REGION Network 4: Znacznik błedu komunikacji modbus
   RUNG wire#powerrail
      { S7_Templates := "SrcType := USInt" } EQ_Contact(in1 := "dbTags_master_Fal_1"."step", in2 := 1)
      wire#w1
      "MB_MASTER_DB".MB_MASTER(REQ := "dbTags_master_Fal_1".modbusMaster.req, MB_ADDR := "dbTags_master_Fal_1".modbusMaster.mbAddr, MODE := "dbTags_master_Fal_1".modbusMaster.mode, DATA_ADDR := "dbTags_master_Fal_1".modbusMaster.dataAddr, DATA_LEN := "dbTags_master_Fal_1".modbusMaster.dataLen, DATA_PTR := "dbMasterData".ID26_Inver_Control_word_416000_Fal, DONE => "dbTags_master_Fal_1".modbusMaster.done, BUSY => "dbTags_master_Fal_1".modbusMaster.busy, ERROR => "dbTags_master_Fal_1".modbusMaster.error, STATUS => "dbTags_master_Fal_1".modbusMaster.status)
   END_RUNG
   RUNG wire#powerrail
      { S7_Templates := "SrcType := USInt" } EQ_Contact(in1 := "dbTags_master_Fal_1"."step", in2 := 2)
   END_RUNG wire#w1
   RUNG wire#powerrail
      Contact( "dbTags_master_Fal_1".modbusMaster.error )
      wire#w2
      { S7_GenerateENO := "TRUE" } Move(in := "dbTags_master_Fal_1".modbusMaster.status, out1 => "dbTags_master_Fal_1".modbusMaster.errorStatus)
   END_RUNG
   RUNG wire#w2
      { S7_GenerateENO := "TRUE" } Move(in := 0, out1 => "dbModbusRTU_Reg".receivede26_Inver_Control_word_416000.typeDataInverter_int[0])
   END_RUNG
   // the same network as SCL:
   IF ("dbTags_master_Fal_1"."step" = 1) OR ("dbTags_master_Fal_1"."step" = 2) THEN
       "MB_MASTER_DB"(REQ := "dbTags_master_Fal_1".modbusMaster.req,   // MB_MASTER
                      MB_ADDR := "dbTags_master_Fal_1".modbusMaster.mbAddr,
                      MODE := "dbTags_master_Fal_1".modbusMaster.mode,
                      DATA_ADDR := "dbTags_master_Fal_1".modbusMaster.dataAddr,
                      DATA_LEN := "dbTags_master_Fal_1".modbusMaster.dataLen,
                      DATA_PTR := "dbMasterData".ID26_Inver_Control_word_416000_Fal,
                      DONE => "dbTags_master_Fal_1".modbusMaster.done,
                      BUSY => "dbTags_master_Fal_1".modbusMaster.busy,
                      ERROR => "dbTags_master_Fal_1".modbusMaster.error,
                      STATUS => "dbTags_master_Fal_1".modbusMaster.status);
   END_IF;
   IF "dbTags_master_Fal_1".modbusMaster.error THEN
       "dbTags_master_Fal_1".modbusMaster.errorStatus := "dbTags_master_Fal_1".modbusMaster.status;
       "dbModbusRTU_Reg".receivede26_Inver_Control_word_416000.typeDataInverter_int[0] := 0;
   END_IF;
END_REGION

REGION Network 5: step1: save received data 416000
   RUNG wire#powerrail
      { S7_Templates := "SrcType := USInt" } EQ_Contact(in1 := "dbTags_master_Fal_1"."step", in2 := 2)
      Contact( "dbTags_master_Fal_1".modbusMaster.done )
      wire#w1
      { S7_GenerateENO := "TRUE" } Move(in := "dbMasterData".ID26_Inver_Control_word_416000_Fal.typeDataInverter_int[0], out1 => "dbModbusRTU_Reg".receivede26_Inver_Control_word_416000.typeDataInverter_int[0])
      R_Coil( "dbTags_master_Fal_1".modbusMaster.req )
   END_RUNG
   RUNG wire#w1
      { S7_GenerateENO := "TRUE" } Move(in := 3, out1 => "dbTags_master_Fal_1"."step")
   END_RUNG
   // the same network as SCL:
   // ENO of a box is taken as its EN; it also drops when the box reports an error
   IF ("dbTags_master_Fal_1"."step" = 2) AND "dbTags_master_Fal_1".modbusMaster.done THEN
       "dbModbusRTU_Reg".receivede26_Inver_Control_word_416000.typeDataInverter_int[0] := "dbMasterData".ID26_Inver_Control_word_416000_Fal.typeDataInverter_int[0];
       "dbTags_master_Fal_1".modbusMaster.req := FALSE;
       "dbTags_master_Fal_1"."step" := 3;
   END_IF;
END_REGION

REGION Network 6: MODBUS RTU adress 26*****step 2: read from slave Inverter setpoint
   // Pobieranie wartości zadanej Hz
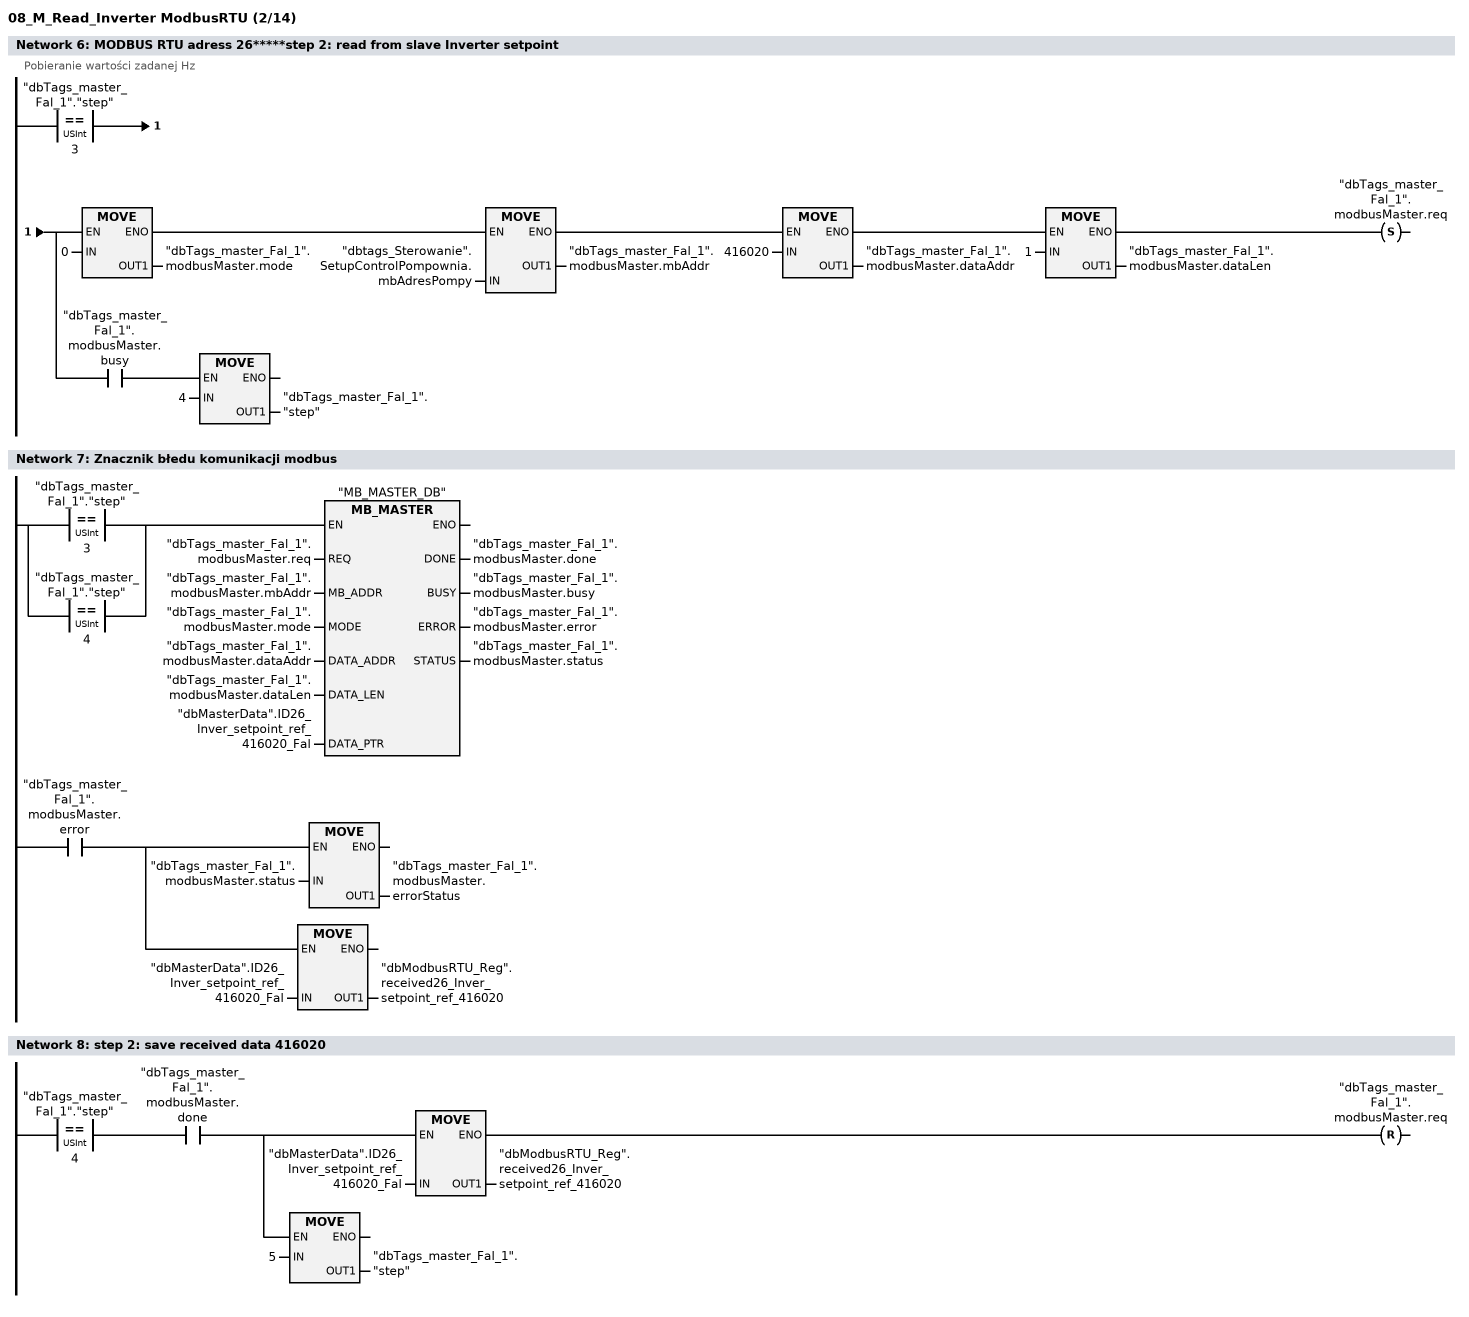
   RUNG wire#powerrail
      { S7_Templates := "SrcType := USInt" } EQ_Contact(in1 := "dbTags_master_Fal_1"."step", in2 := 3)
      wire#w1
      { S7_GenerateENO := "TRUE" } Move(in := 0, out1 => "dbTags_master_Fal_1".modbusMaster.mode)
      Move(in := "dbtags_Sterowanie".SetupControlPompownia.mbAdresPompy, out1 => "dbTags_master_Fal_1".modbusMaster.mbAddr)
      { S7_GenerateENO := "TRUE" } Move(in := 416020, out1 => "dbTags_master_Fal_1".modbusMaster.dataAddr)
      Move(in := 1, out1 => "dbTags_master_Fal_1".modbusMaster.dataLen)
      S_Coil( "dbTags_master_Fal_1".modbusMaster.req )
   END_RUNG
   RUNG wire#w1
      Contact( "dbTags_master_Fal_1".modbusMaster.busy )
      { S7_GenerateENO := "TRUE" } Move(in := 4, out1 => "dbTags_master_Fal_1"."step")
   END_RUNG
   // the same network as SCL:
   // ENO of a box is taken as its EN; it also drops when the box reports an error
   #_w1 := "dbTags_master_Fal_1"."step" = 3;
   IF #_w1 THEN
       "dbTags_master_Fal_1".modbusMaster.mode := 0;
       "dbTags_master_Fal_1".modbusMaster.mbAddr := "dbtags_Sterowanie".SetupControlPompownia.mbAdresPompy;
       "dbTags_master_Fal_1".modbusMaster.dataAddr := 416020;
       "dbTags_master_Fal_1".modbusMaster.dataLen := 1;
       "dbTags_master_Fal_1".modbusMaster.req := TRUE;
   END_IF;
   IF #_w1 AND "dbTags_master_Fal_1".modbusMaster.busy THEN "dbTags_master_Fal_1"."step" := 4; END_IF;
END_REGION

REGION Network 7: Znacznik błedu komunikacji modbus
   RUNG wire#powerrail
      { S7_Templates := "SrcType := USInt" } EQ_Contact(in1 := "dbTags_master_Fal_1"."step", in2 := 3)
      wire#w1
      "MB_MASTER_DB".MB_MASTER(REQ := "dbTags_master_Fal_1".modbusMaster.req, MB_ADDR := "dbTags_master_Fal_1".modbusMaster.mbAddr, MODE := "dbTags_master_Fal_1".modbusMaster.mode, DATA_ADDR := "dbTags_master_Fal_1".modbusMaster.dataAddr, DATA_LEN := "dbTags_master_Fal_1".modbusMaster.dataLen, DATA_PTR := "dbMasterData".ID26_Inver_setpoint_ref_416020_Fal, DONE => "dbTags_master_Fal_1".modbusMaster.done, BUSY => "dbTags_master_Fal_1".modbusMaster.busy, ERROR => "dbTags_master_Fal_1".modbusMaster.error, STATUS => "dbTags_master_Fal_1".modbusMaster.status)
   END_RUNG
   RUNG wire#powerrail
      { S7_Templates := "SrcType := USInt" } EQ_Contact(in1 := "dbTags_master_Fal_1"."step", in2 := 4)
   END_RUNG wire#w1
   RUNG wire#powerrail
      Contact( "dbTags_master_Fal_1".modbusMaster.error )
      wire#w2
      { S7_GenerateENO := "TRUE" } Move(in := "dbTags_master_Fal_1".modbusMaster.status, out1 => "dbTags_master_Fal_1".modbusMaster.errorStatus)
   END_RUNG
   RUNG wire#w2
      { S7_GenerateENO := "TRUE" } Move(in := "dbMasterData".ID26_Inver_setpoint_ref_416020_Fal, out1 => "dbModbusRTU_Reg".received26_Inver_setpoint_ref_416020)
   END_RUNG
   // the same network as SCL:
   IF ("dbTags_master_Fal_1"."step" = 3) OR ("dbTags_master_Fal_1"."step" = 4) THEN
       "MB_MASTER_DB"(REQ := "dbTags_master_Fal_1".modbusMaster.req,   // MB_MASTER
                      MB_ADDR := "dbTags_master_Fal_1".modbusMaster.mbAddr,
                      MODE := "dbTags_master_Fal_1".modbusMaster.mode,
                      DATA_ADDR := "dbTags_master_Fal_1".modbusMaster.dataAddr,
                      DATA_LEN := "dbTags_master_Fal_1".modbusMaster.dataLen,
                      DATA_PTR := "dbMasterData".ID26_Inver_setpoint_ref_416020_Fal,
                      DONE => "dbTags_master_Fal_1".modbusMaster.done,
                      BUSY => "dbTags_master_Fal_1".modbusMaster.busy,
                      ERROR => "dbTags_master_Fal_1".modbusMaster.error,
                      STATUS => "dbTags_master_Fal_1".modbusMaster.status);
   END_IF;
   IF "dbTags_master_Fal_1".modbusMaster.error THEN
       "dbTags_master_Fal_1".modbusMaster.errorStatus := "dbTags_master_Fal_1".modbusMaster.status;
       "dbModbusRTU_Reg".received26_Inver_setpoint_ref_416020 := "dbMasterData".ID26_Inver_setpoint_ref_416020_Fal;
   END_IF;
END_REGION

REGION Network 8: step 2: save received data 416020
   RUNG wire#powerrail
      { S7_Templates := "SrcType := USInt" } EQ_Contact(in1 := "dbTags_master_Fal_1"."step", in2 := 4)
      Contact( "dbTags_master_Fal_1".modbusMaster.done )
      wire#w1
      { S7_GenerateENO := "TRUE" } Move(in := "dbMasterData".ID26_Inver_setpoint_ref_416020_Fal, out1 => "dbModbusRTU_Reg".received26_Inver_setpoint_ref_416020)
      R_Coil( "dbTags_master_Fal_1".modbusMaster.req )
   END_RUNG
   RUNG wire#w1
      { S7_GenerateENO := "TRUE" } Move(in := 5, out1 => "dbTags_master_Fal_1"."step")
   END_RUNG
   // the same network as SCL:
   // ENO of a box is taken as its EN; it also drops when the box reports an error
   IF ("dbTags_master_Fal_1"."step" = 4) AND "dbTags_master_Fal_1".modbusMaster.done THEN
       "dbModbusRTU_Reg".received26_Inver_setpoint_ref_416020 := "dbMasterData".ID26_Inver_setpoint_ref_416020_Fal;
       "dbTags_master_Fal_1".modbusMaster.req := FALSE;
       "dbTags_master_Fal_1"."step" := 5;
   END_IF;
END_REGION

REGION Network 9: MODBUS RTU adress 26*****step 3: read from slave Inverter status word
   // Pobieramy status falownika
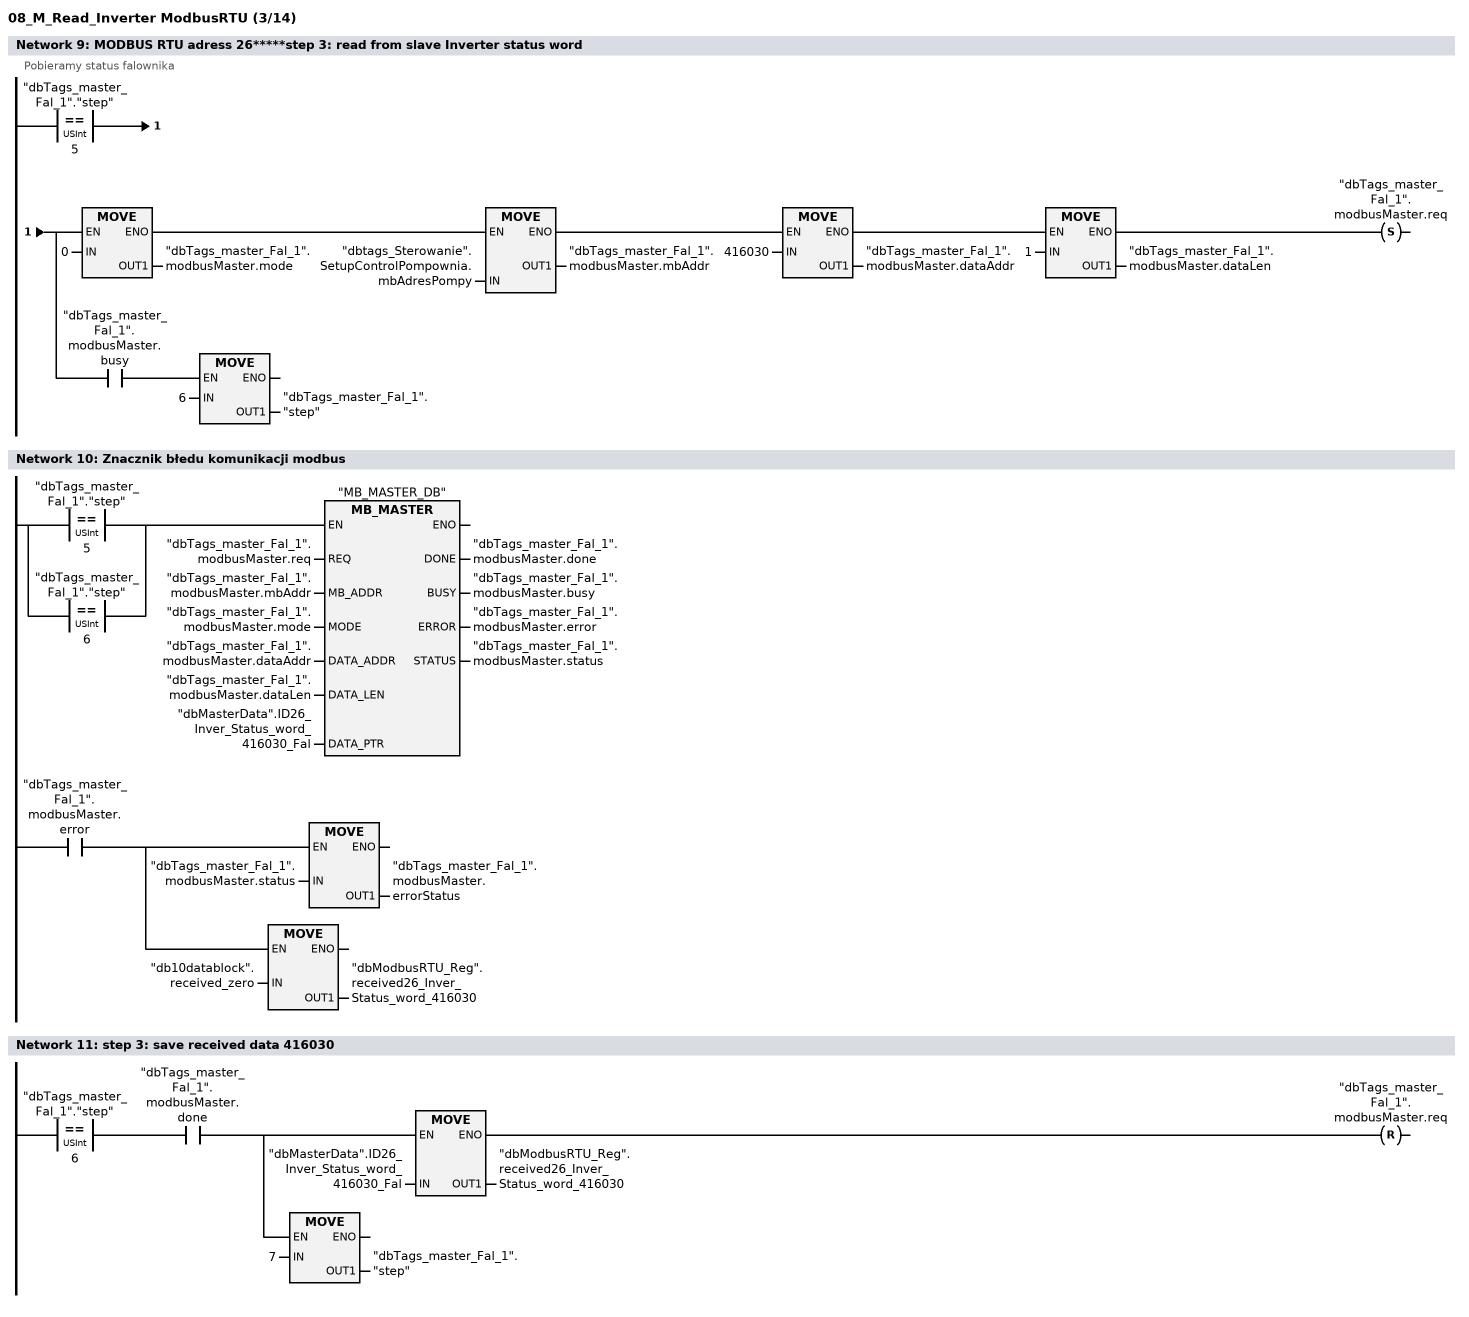
   RUNG wire#powerrail
      { S7_Templates := "SrcType := USInt" } EQ_Contact(in1 := "dbTags_master_Fal_1"."step", in2 := 5)
      wire#w1
      { S7_GenerateENO := "TRUE" } Move(in := 0, out1 => "dbTags_master_Fal_1".modbusMaster.mode)
      Move(in := "dbtags_Sterowanie".SetupControlPompownia.mbAdresPompy, out1 => "dbTags_master_Fal_1".modbusMaster.mbAddr)
      { S7_GenerateENO := "TRUE" } Move(in := 416030, out1 => "dbTags_master_Fal_1".modbusMaster.dataAddr)
      Move(in := 1, out1 => "dbTags_master_Fal_1".modbusMaster.dataLen)
      S_Coil( "dbTags_master_Fal_1".modbusMaster.req )
   END_RUNG
   RUNG wire#w1
      Contact( "dbTags_master_Fal_1".modbusMaster.busy )
      { S7_GenerateENO := "TRUE" } Move(in := 6, out1 => "dbTags_master_Fal_1"."step")
   END_RUNG
   // the same network as SCL:
   // ENO of a box is taken as its EN; it also drops when the box reports an error
   #_w1 := "dbTags_master_Fal_1"."step" = 5;
   IF #_w1 THEN
       "dbTags_master_Fal_1".modbusMaster.mode := 0;
       "dbTags_master_Fal_1".modbusMaster.mbAddr := "dbtags_Sterowanie".SetupControlPompownia.mbAdresPompy;
       "dbTags_master_Fal_1".modbusMaster.dataAddr := 416030;
       "dbTags_master_Fal_1".modbusMaster.dataLen := 1;
       "dbTags_master_Fal_1".modbusMaster.req := TRUE;
   END_IF;
   IF #_w1 AND "dbTags_master_Fal_1".modbusMaster.busy THEN "dbTags_master_Fal_1"."step" := 6; END_IF;
END_REGION

REGION Network 10: Znacznik błedu komunikacji modbus
   RUNG wire#powerrail
      { S7_Templates := "SrcType := USInt" } EQ_Contact(in1 := "dbTags_master_Fal_1"."step", in2 := 5)
      wire#w1
      "MB_MASTER_DB".MB_MASTER(REQ := "dbTags_master_Fal_1".modbusMaster.req, MB_ADDR := "dbTags_master_Fal_1".modbusMaster.mbAddr, MODE := "dbTags_master_Fal_1".modbusMaster.mode, DATA_ADDR := "dbTags_master_Fal_1".modbusMaster.dataAddr, DATA_LEN := "dbTags_master_Fal_1".modbusMaster.dataLen, DATA_PTR := "dbMasterData".ID26_Inver_Status_word_416030_Fal, DONE => "dbTags_master_Fal_1".modbusMaster.done, BUSY => "dbTags_master_Fal_1".modbusMaster.busy, ERROR => "dbTags_master_Fal_1".modbusMaster.error, STATUS => "dbTags_master_Fal_1".modbusMaster.status)
   END_RUNG
   RUNG wire#powerrail
      { S7_Templates := "SrcType := USInt" } EQ_Contact(in1 := "dbTags_master_Fal_1"."step", in2 := 6)
   END_RUNG wire#w1
   RUNG wire#powerrail
      Contact( "dbTags_master_Fal_1".modbusMaster.error )
      wire#w2
      { S7_GenerateENO := "TRUE" } Move(in := "dbTags_master_Fal_1".modbusMaster.status, out1 => "dbTags_master_Fal_1".modbusMaster.errorStatus)
   END_RUNG
   RUNG wire#w2
      { S7_GenerateENO := "TRUE" } Move(in := "db10datablock".received_zero, out1 => "dbModbusRTU_Reg".received26_Inver_Status_word_416030)
   END_RUNG
   // the same network as SCL:
   IF ("dbTags_master_Fal_1"."step" = 5) OR ("dbTags_master_Fal_1"."step" = 6) THEN
       "MB_MASTER_DB"(REQ := "dbTags_master_Fal_1".modbusMaster.req,   // MB_MASTER
                      MB_ADDR := "dbTags_master_Fal_1".modbusMaster.mbAddr,
                      MODE := "dbTags_master_Fal_1".modbusMaster.mode,
                      DATA_ADDR := "dbTags_master_Fal_1".modbusMaster.dataAddr,
                      DATA_LEN := "dbTags_master_Fal_1".modbusMaster.dataLen,
                      DATA_PTR := "dbMasterData".ID26_Inver_Status_word_416030_Fal,
                      DONE => "dbTags_master_Fal_1".modbusMaster.done,
                      BUSY => "dbTags_master_Fal_1".modbusMaster.busy,
                      ERROR => "dbTags_master_Fal_1".modbusMaster.error,
                      STATUS => "dbTags_master_Fal_1".modbusMaster.status);
   END_IF;
   IF "dbTags_master_Fal_1".modbusMaster.error THEN
       "dbTags_master_Fal_1".modbusMaster.errorStatus := "dbTags_master_Fal_1".modbusMaster.status;
       "dbModbusRTU_Reg".received26_Inver_Status_word_416030 := "db10datablock".received_zero;
   END_IF;
END_REGION

REGION Network 11: step 3: save received data 416030
   RUNG wire#powerrail
      { S7_Templates := "SrcType := USInt" } EQ_Contact(in1 := "dbTags_master_Fal_1"."step", in2 := 6)
      Contact( "dbTags_master_Fal_1".modbusMaster.done )
      wire#w1
      { S7_GenerateENO := "TRUE" } Move(in := "dbMasterData".ID26_Inver_Status_word_416030_Fal, out1 => "dbModbusRTU_Reg".received26_Inver_Status_word_416030)
      R_Coil( "dbTags_master_Fal_1".modbusMaster.req )
   END_RUNG
   RUNG wire#w1
      { S7_GenerateENO := "TRUE" } Move(in := 7, out1 => "dbTags_master_Fal_1"."step")
   END_RUNG
   // the same network as SCL:
   // ENO of a box is taken as its EN; it also drops when the box reports an error
   IF ("dbTags_master_Fal_1"."step" = 6) AND "dbTags_master_Fal_1".modbusMaster.done THEN
       "dbModbusRTU_Reg".received26_Inver_Status_word_416030 := "dbMasterData".ID26_Inver_Status_word_416030_Fal;
       "dbTags_master_Fal_1".modbusMaster.req := FALSE;
       "dbTags_master_Fal_1"."step" := 7;
   END_IF;
END_REGION

REGION Network 13: MODBUS RTU adress 26*****step 4: read from slave Inverter frequency
   // Pobieramy częstotliwość na silniku
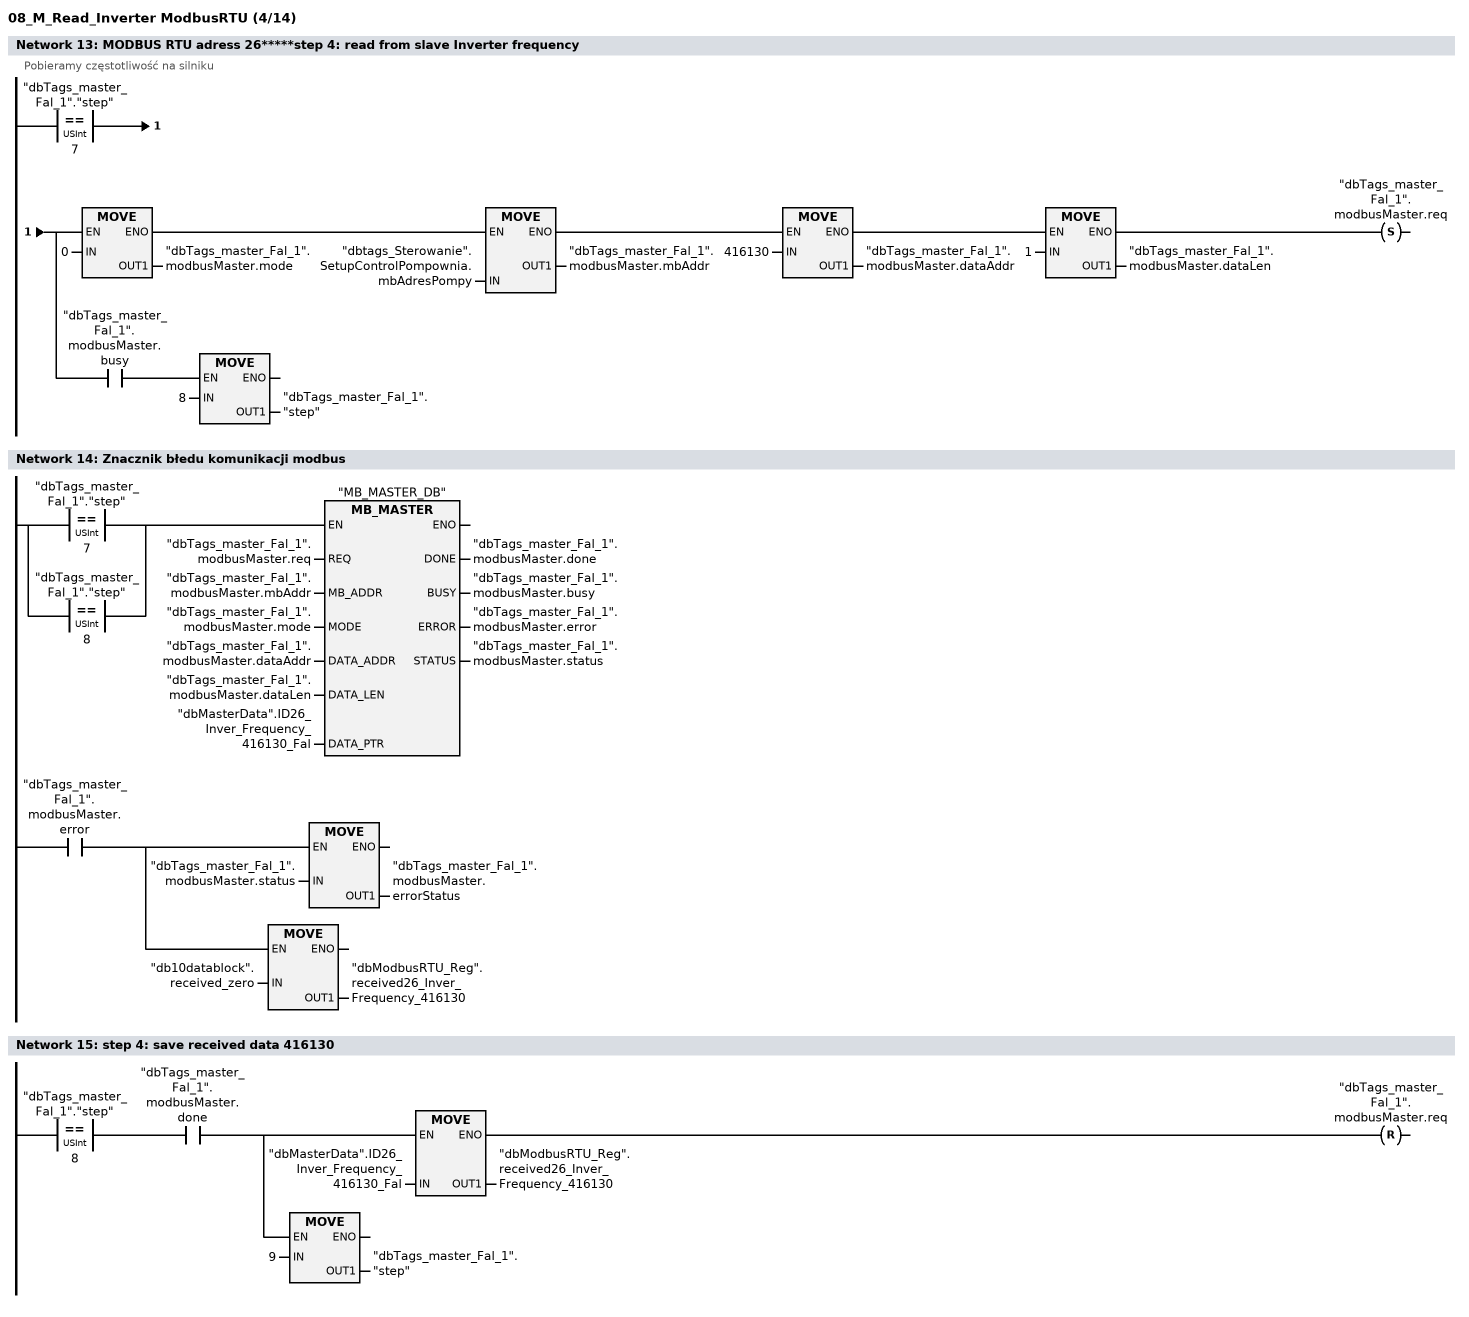
   RUNG wire#powerrail
      { S7_Templates := "SrcType := USInt" } EQ_Contact(in1 := "dbTags_master_Fal_1"."step", in2 := 7)
      wire#w1
      { S7_GenerateENO := "TRUE" } Move(in := 0, out1 => "dbTags_master_Fal_1".modbusMaster.mode)
      Move(in := "dbtags_Sterowanie".SetupControlPompownia.mbAdresPompy, out1 => "dbTags_master_Fal_1".modbusMaster.mbAddr)
      { S7_GenerateENO := "TRUE" } Move(in := 416130, out1 => "dbTags_master_Fal_1".modbusMaster.dataAddr)
      Move(in := 1, out1 => "dbTags_master_Fal_1".modbusMaster.dataLen)
      S_Coil( "dbTags_master_Fal_1".modbusMaster.req )
   END_RUNG
   RUNG wire#w1
      Contact( "dbTags_master_Fal_1".modbusMaster.busy )
      { S7_GenerateENO := "TRUE" } Move(in := 8, out1 => "dbTags_master_Fal_1"."step")
   END_RUNG
   // the same network as SCL:
   // ENO of a box is taken as its EN; it also drops when the box reports an error
   #_w1 := "dbTags_master_Fal_1"."step" = 7;
   IF #_w1 THEN
       "dbTags_master_Fal_1".modbusMaster.mode := 0;
       "dbTags_master_Fal_1".modbusMaster.mbAddr := "dbtags_Sterowanie".SetupControlPompownia.mbAdresPompy;
       "dbTags_master_Fal_1".modbusMaster.dataAddr := 416130;
       "dbTags_master_Fal_1".modbusMaster.dataLen := 1;
       "dbTags_master_Fal_1".modbusMaster.req := TRUE;
   END_IF;
   IF #_w1 AND "dbTags_master_Fal_1".modbusMaster.busy THEN "dbTags_master_Fal_1"."step" := 8; END_IF;
END_REGION

REGION Network 14: Znacznik błedu komunikacji modbus
   RUNG wire#powerrail
      { S7_Templates := "SrcType := USInt" } EQ_Contact(in1 := "dbTags_master_Fal_1"."step", in2 := 7)
      wire#w1
      "MB_MASTER_DB".MB_MASTER(REQ := "dbTags_master_Fal_1".modbusMaster.req, MB_ADDR := "dbTags_master_Fal_1".modbusMaster.mbAddr, MODE := "dbTags_master_Fal_1".modbusMaster.mode, DATA_ADDR := "dbTags_master_Fal_1".modbusMaster.dataAddr, DATA_LEN := "dbTags_master_Fal_1".modbusMaster.dataLen, DATA_PTR := "dbMasterData".ID26_Inver_Frequency_416130_Fal, DONE => "dbTags_master_Fal_1".modbusMaster.done, BUSY => "dbTags_master_Fal_1".modbusMaster.busy, ERROR => "dbTags_master_Fal_1".modbusMaster.error, STATUS => "dbTags_master_Fal_1".modbusMaster.status)
   END_RUNG
   RUNG wire#powerrail
      { S7_Templates := "SrcType := USInt" } EQ_Contact(in1 := "dbTags_master_Fal_1"."step", in2 := 8)
   END_RUNG wire#w1
   RUNG wire#powerrail
      Contact( "dbTags_master_Fal_1".modbusMaster.error )
      wire#w2
      { S7_GenerateENO := "TRUE" } Move(in := "dbTags_master_Fal_1".modbusMaster.status, out1 => "dbTags_master_Fal_1".modbusMaster.errorStatus)
   END_RUNG
   RUNG wire#w2
      { S7_GenerateENO := "TRUE" } Move(in := "db10datablock".received_zero, out1 => "dbModbusRTU_Reg".received26_Inver_Frequency_416130)
   END_RUNG
   // the same network as SCL:
   IF ("dbTags_master_Fal_1"."step" = 7) OR ("dbTags_master_Fal_1"."step" = 8) THEN
       "MB_MASTER_DB"(REQ := "dbTags_master_Fal_1".modbusMaster.req,   // MB_MASTER
                      MB_ADDR := "dbTags_master_Fal_1".modbusMaster.mbAddr,
                      MODE := "dbTags_master_Fal_1".modbusMaster.mode,
                      DATA_ADDR := "dbTags_master_Fal_1".modbusMaster.dataAddr,
                      DATA_LEN := "dbTags_master_Fal_1".modbusMaster.dataLen,
                      DATA_PTR := "dbMasterData".ID26_Inver_Frequency_416130_Fal,
                      DONE => "dbTags_master_Fal_1".modbusMaster.done,
                      BUSY => "dbTags_master_Fal_1".modbusMaster.busy,
                      ERROR => "dbTags_master_Fal_1".modbusMaster.error,
                      STATUS => "dbTags_master_Fal_1".modbusMaster.status);
   END_IF;
   IF "dbTags_master_Fal_1".modbusMaster.error THEN
       "dbTags_master_Fal_1".modbusMaster.errorStatus := "dbTags_master_Fal_1".modbusMaster.status;
       "dbModbusRTU_Reg".received26_Inver_Frequency_416130 := "db10datablock".received_zero;
   END_IF;
END_REGION

REGION Network 15: step 4: save received data 416130
   RUNG wire#powerrail
      { S7_Templates := "SrcType := USInt" } EQ_Contact(in1 := "dbTags_master_Fal_1"."step", in2 := 8)
      Contact( "dbTags_master_Fal_1".modbusMaster.done )
      wire#w1
      { S7_GenerateENO := "TRUE" } Move(in := "dbMasterData".ID26_Inver_Frequency_416130_Fal, out1 => "dbModbusRTU_Reg".received26_Inver_Frequency_416130)
      R_Coil( "dbTags_master_Fal_1".modbusMaster.req )
   END_RUNG
   RUNG wire#w1
      { S7_GenerateENO := "TRUE" } Move(in := 9, out1 => "dbTags_master_Fal_1"."step")
   END_RUNG
   // the same network as SCL:
   // ENO of a box is taken as its EN; it also drops when the box reports an error
   IF ("dbTags_master_Fal_1"."step" = 8) AND "dbTags_master_Fal_1".modbusMaster.done THEN
       "dbModbusRTU_Reg".received26_Inver_Frequency_416130 := "dbMasterData".ID26_Inver_Frequency_416130_Fal;
       "dbTags_master_Fal_1".modbusMaster.req := FALSE;
       "dbTags_master_Fal_1"."step" := 9;
   END_IF;
END_REGION

REGION Network 17: MODBUS RTU adress 26*****step 5: read from slave Motor Current
   // Pobieramy prąd silnika
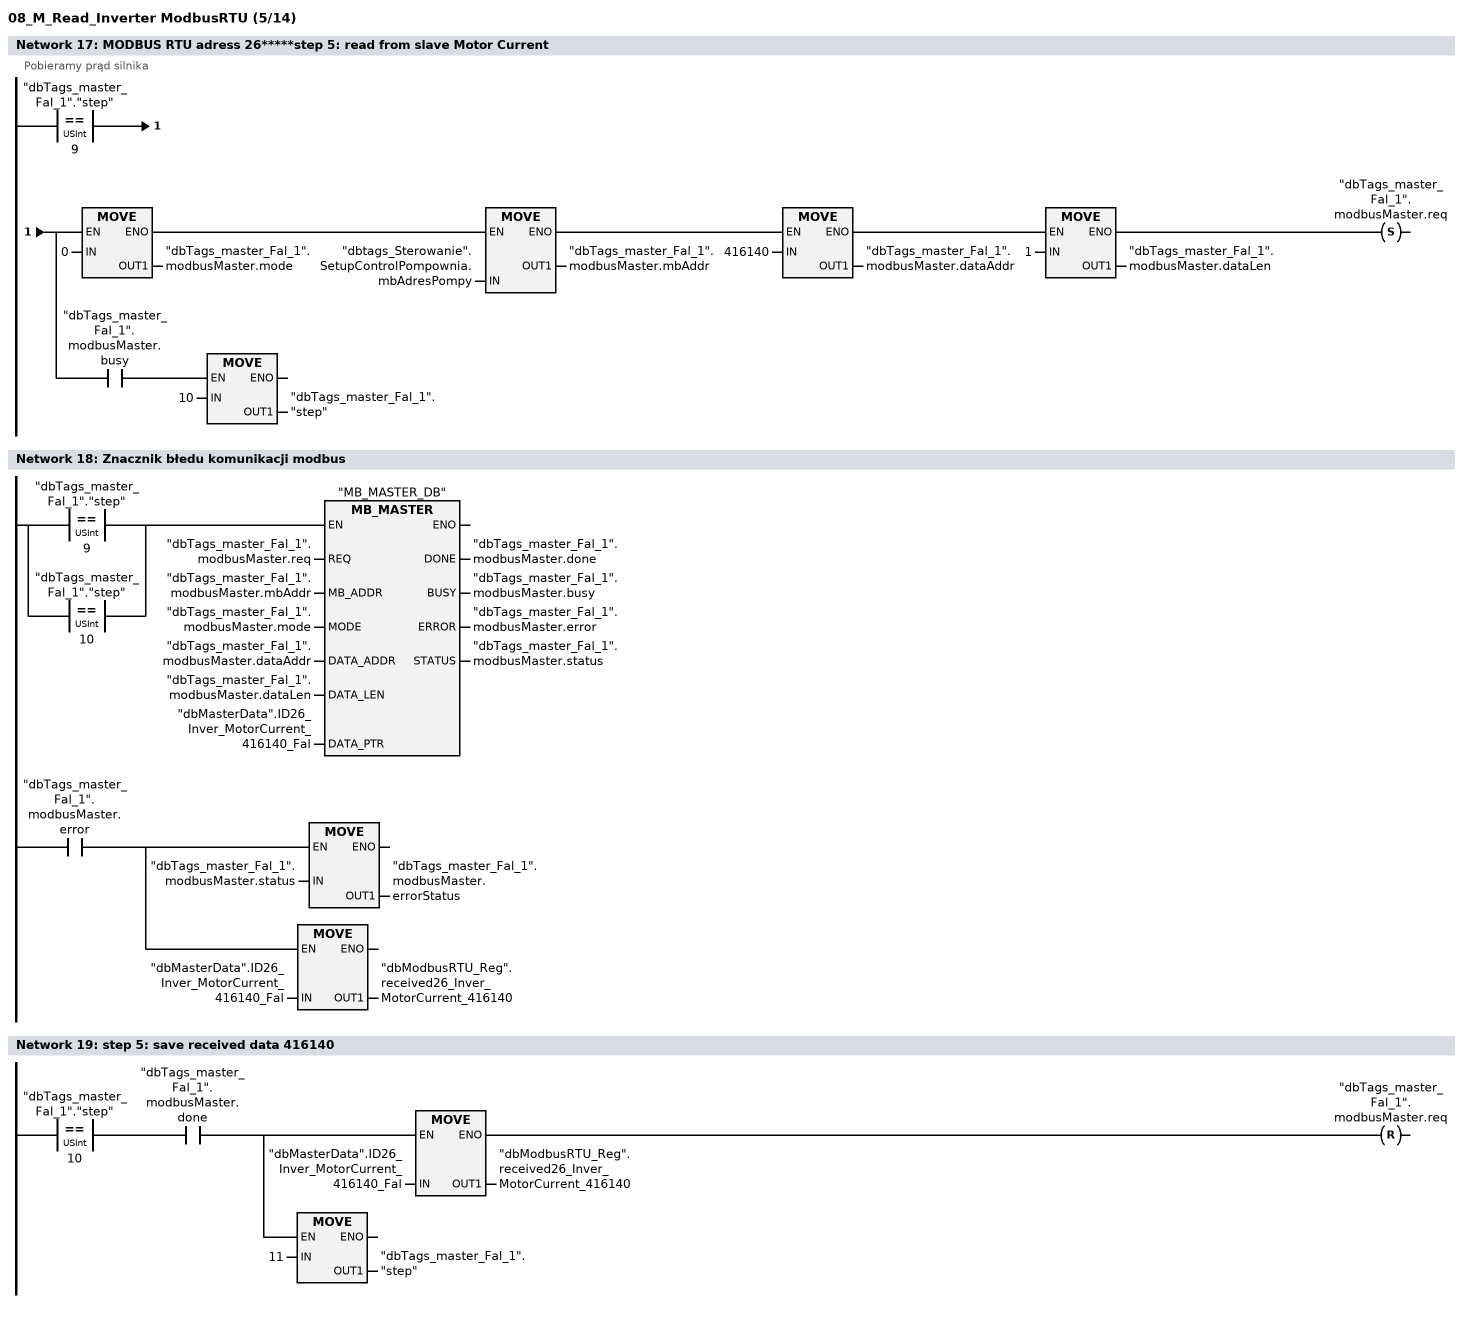
   RUNG wire#powerrail
      { S7_Templates := "SrcType := USInt" } EQ_Contact(in1 := "dbTags_master_Fal_1"."step", in2 := 9)
      wire#w1
      { S7_GenerateENO := "TRUE" } Move(in := 0, out1 => "dbTags_master_Fal_1".modbusMaster.mode)
      Move(in := "dbtags_Sterowanie".SetupControlPompownia.mbAdresPompy, out1 => "dbTags_master_Fal_1".modbusMaster.mbAddr)
      { S7_GenerateENO := "TRUE" } Move(in := 416140, out1 => "dbTags_master_Fal_1".modbusMaster.dataAddr)
      Move(in := 1, out1 => "dbTags_master_Fal_1".modbusMaster.dataLen)
      S_Coil( "dbTags_master_Fal_1".modbusMaster.req )
   END_RUNG
   RUNG wire#w1
      Contact( "dbTags_master_Fal_1".modbusMaster.busy )
      { S7_GenerateENO := "TRUE" } Move(in := 10, out1 => "dbTags_master_Fal_1"."step")
   END_RUNG
   // the same network as SCL:
   // ENO of a box is taken as its EN; it also drops when the box reports an error
   #_w1 := "dbTags_master_Fal_1"."step" = 9;
   IF #_w1 THEN
       "dbTags_master_Fal_1".modbusMaster.mode := 0;
       "dbTags_master_Fal_1".modbusMaster.mbAddr := "dbtags_Sterowanie".SetupControlPompownia.mbAdresPompy;
       "dbTags_master_Fal_1".modbusMaster.dataAddr := 416140;
       "dbTags_master_Fal_1".modbusMaster.dataLen := 1;
       "dbTags_master_Fal_1".modbusMaster.req := TRUE;
   END_IF;
   IF #_w1 AND "dbTags_master_Fal_1".modbusMaster.busy THEN "dbTags_master_Fal_1"."step" := 10; END_IF;
END_REGION

REGION Network 18: Znacznik błedu komunikacji modbus
   RUNG wire#powerrail
      { S7_Templates := "SrcType := USInt" } EQ_Contact(in1 := "dbTags_master_Fal_1"."step", in2 := 9)
      wire#w1
      "MB_MASTER_DB".MB_MASTER(REQ := "dbTags_master_Fal_1".modbusMaster.req, MB_ADDR := "dbTags_master_Fal_1".modbusMaster.mbAddr, MODE := "dbTags_master_Fal_1".modbusMaster.mode, DATA_ADDR := "dbTags_master_Fal_1".modbusMaster.dataAddr, DATA_LEN := "dbTags_master_Fal_1".modbusMaster.dataLen, DATA_PTR := "dbMasterData".ID26_Inver_MotorCurrent_416140_Fal, DONE => "dbTags_master_Fal_1".modbusMaster.done, BUSY => "dbTags_master_Fal_1".modbusMaster.busy, ERROR => "dbTags_master_Fal_1".modbusMaster.error, STATUS => "dbTags_master_Fal_1".modbusMaster.status)
   END_RUNG
   RUNG wire#powerrail
      { S7_Templates := "SrcType := USInt" } EQ_Contact(in1 := "dbTags_master_Fal_1"."step", in2 := 10)
   END_RUNG wire#w1
   RUNG wire#powerrail
      Contact( "dbTags_master_Fal_1".modbusMaster.error )
      wire#w2
      { S7_GenerateENO := "TRUE" } Move(in := "dbTags_master_Fal_1".modbusMaster.status, out1 => "dbTags_master_Fal_1".modbusMaster.errorStatus)
   END_RUNG
   RUNG wire#w2
      { S7_GenerateENO := "TRUE" } Move(in := "dbMasterData".ID26_Inver_MotorCurrent_416140_Fal, out1 => "dbModbusRTU_Reg".received26_Inver_MotorCurrent_416140)
   END_RUNG
   // the same network as SCL:
   IF ("dbTags_master_Fal_1"."step" = 9) OR ("dbTags_master_Fal_1"."step" = 10) THEN
       "MB_MASTER_DB"(REQ := "dbTags_master_Fal_1".modbusMaster.req,   // MB_MASTER
                      MB_ADDR := "dbTags_master_Fal_1".modbusMaster.mbAddr,
                      MODE := "dbTags_master_Fal_1".modbusMaster.mode,
                      DATA_ADDR := "dbTags_master_Fal_1".modbusMaster.dataAddr,
                      DATA_LEN := "dbTags_master_Fal_1".modbusMaster.dataLen,
                      DATA_PTR := "dbMasterData".ID26_Inver_MotorCurrent_416140_Fal,
                      DONE => "dbTags_master_Fal_1".modbusMaster.done,
                      BUSY => "dbTags_master_Fal_1".modbusMaster.busy,
                      ERROR => "dbTags_master_Fal_1".modbusMaster.error,
                      STATUS => "dbTags_master_Fal_1".modbusMaster.status);
   END_IF;
   IF "dbTags_master_Fal_1".modbusMaster.error THEN
       "dbTags_master_Fal_1".modbusMaster.errorStatus := "dbTags_master_Fal_1".modbusMaster.status;
       "dbModbusRTU_Reg".received26_Inver_MotorCurrent_416140 := "dbMasterData".ID26_Inver_MotorCurrent_416140_Fal;
   END_IF;
END_REGION

REGION Network 19: step 5: save received data 416140
   RUNG wire#powerrail
      { S7_Templates := "SrcType := USInt" } EQ_Contact(in1 := "dbTags_master_Fal_1"."step", in2 := 10)
      Contact( "dbTags_master_Fal_1".modbusMaster.done )
      wire#w1
      { S7_GenerateENO := "TRUE" } Move(in := "dbMasterData".ID26_Inver_MotorCurrent_416140_Fal, out1 => "dbModbusRTU_Reg".received26_Inver_MotorCurrent_416140)
      R_Coil( "dbTags_master_Fal_1".modbusMaster.req )
   END_RUNG
   RUNG wire#w1
      { S7_GenerateENO := "TRUE" } Move(in := 11, out1 => "dbTags_master_Fal_1"."step")
   END_RUNG
   // the same network as SCL:
   // ENO of a box is taken as its EN; it also drops when the box reports an error
   IF ("dbTags_master_Fal_1"."step" = 10) AND "dbTags_master_Fal_1".modbusMaster.done THEN
       "dbModbusRTU_Reg".received26_Inver_MotorCurrent_416140 := "dbMasterData".ID26_Inver_MotorCurrent_416140_Fal;
       "dbTags_master_Fal_1".modbusMaster.req := FALSE;
       "dbTags_master_Fal_1"."step" := 11;
   END_IF;
END_REGION

REGION Network 21: MODBUS RTU adress 26*****step 6: read from slave DC Voltage
   // Pobieramy napięcie na szynie DC
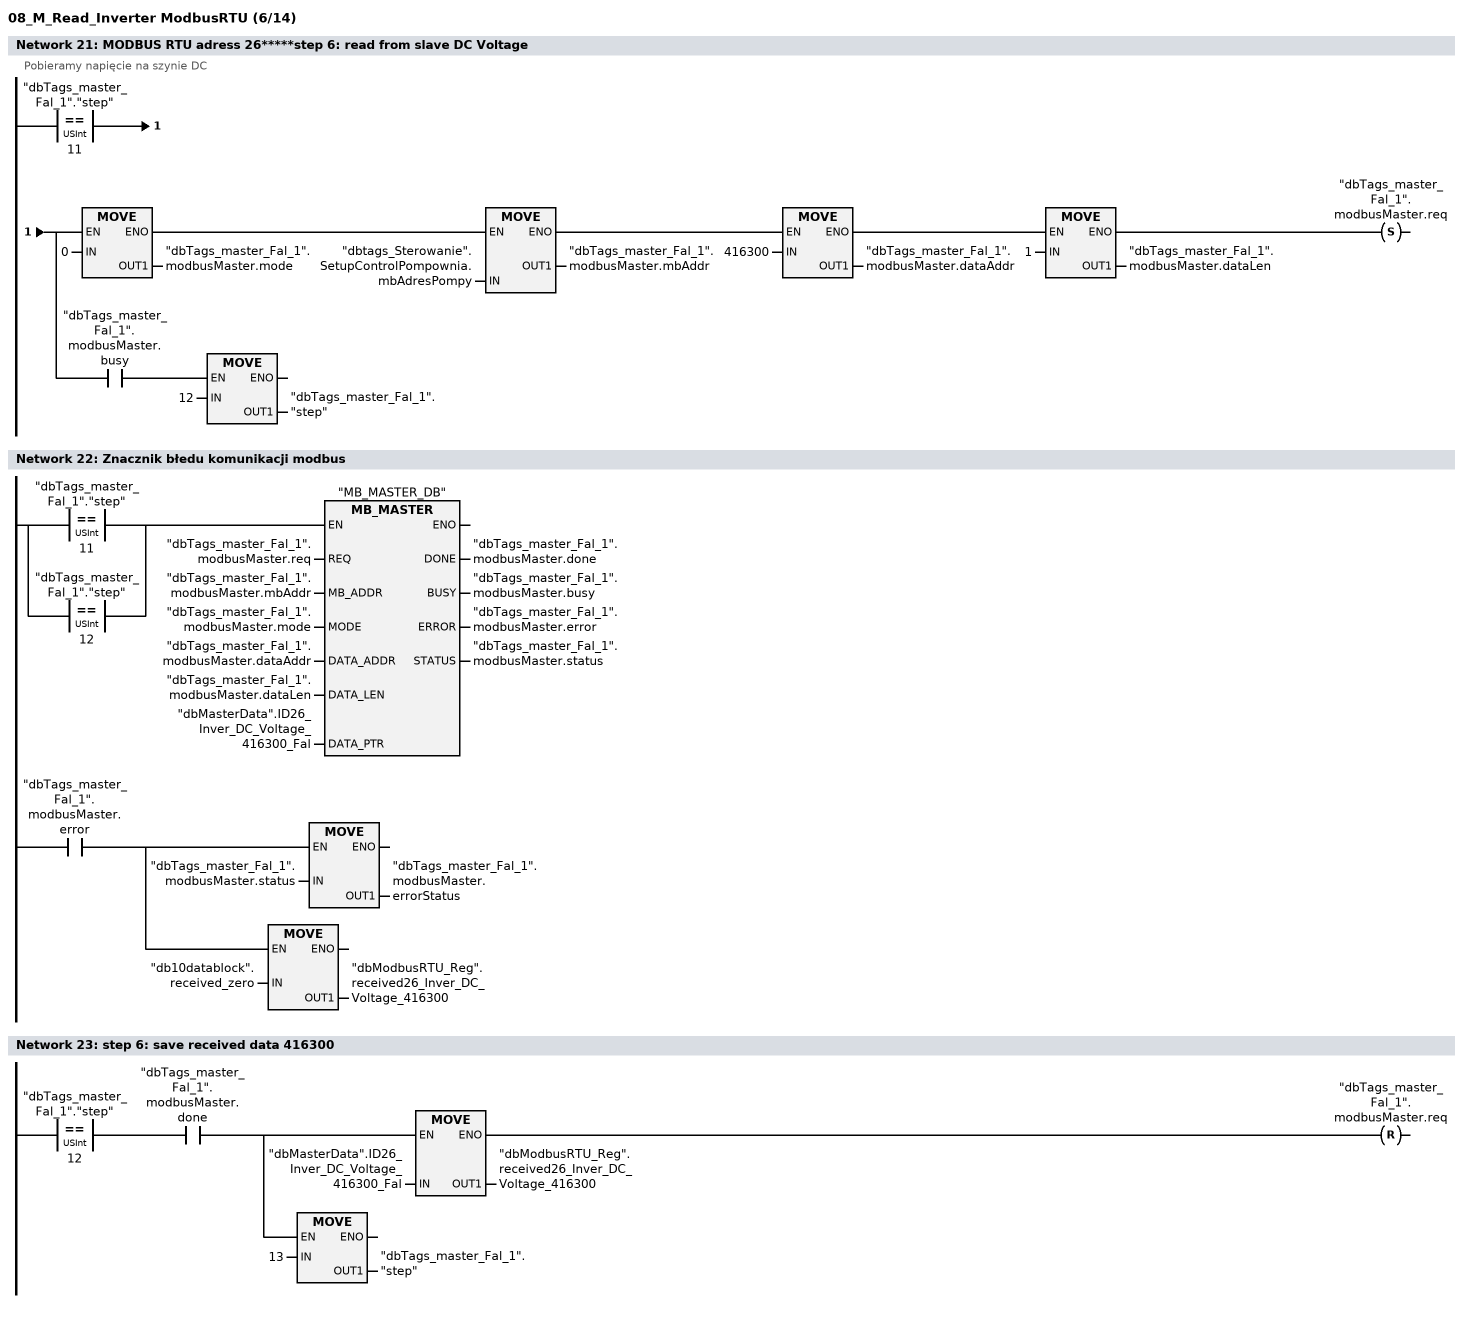
   RUNG wire#powerrail
      { S7_Templates := "SrcType := USInt" } EQ_Contact(in1 := "dbTags_master_Fal_1"."step", in2 := 11)
      wire#w1
      { S7_GenerateENO := "TRUE" } Move(in := 0, out1 => "dbTags_master_Fal_1".modbusMaster.mode)
      Move(in := "dbtags_Sterowanie".SetupControlPompownia.mbAdresPompy, out1 => "dbTags_master_Fal_1".modbusMaster.mbAddr)
      { S7_GenerateENO := "TRUE" } Move(in := 416300, out1 => "dbTags_master_Fal_1".modbusMaster.dataAddr)
      Move(in := 1, out1 => "dbTags_master_Fal_1".modbusMaster.dataLen)
      S_Coil( "dbTags_master_Fal_1".modbusMaster.req )
   END_RUNG
   RUNG wire#w1
      Contact( "dbTags_master_Fal_1".modbusMaster.busy )
      { S7_GenerateENO := "TRUE" } Move(in := 12, out1 => "dbTags_master_Fal_1"."step")
   END_RUNG
   // the same network as SCL:
   // ENO of a box is taken as its EN; it also drops when the box reports an error
   #_w1 := "dbTags_master_Fal_1"."step" = 11;
   IF #_w1 THEN
       "dbTags_master_Fal_1".modbusMaster.mode := 0;
       "dbTags_master_Fal_1".modbusMaster.mbAddr := "dbtags_Sterowanie".SetupControlPompownia.mbAdresPompy;
       "dbTags_master_Fal_1".modbusMaster.dataAddr := 416300;
       "dbTags_master_Fal_1".modbusMaster.dataLen := 1;
       "dbTags_master_Fal_1".modbusMaster.req := TRUE;
   END_IF;
   IF #_w1 AND "dbTags_master_Fal_1".modbusMaster.busy THEN "dbTags_master_Fal_1"."step" := 12; END_IF;
END_REGION

REGION Network 22: Znacznik błedu komunikacji modbus
   RUNG wire#powerrail
      { S7_Templates := "SrcType := USInt" } EQ_Contact(in1 := "dbTags_master_Fal_1"."step", in2 := 11)
      wire#w1
      "MB_MASTER_DB".MB_MASTER(REQ := "dbTags_master_Fal_1".modbusMaster.req, MB_ADDR := "dbTags_master_Fal_1".modbusMaster.mbAddr, MODE := "dbTags_master_Fal_1".modbusMaster.mode, DATA_ADDR := "dbTags_master_Fal_1".modbusMaster.dataAddr, DATA_LEN := "dbTags_master_Fal_1".modbusMaster.dataLen, DATA_PTR := "dbMasterData".ID26_Inver_DC_Voltage_416300_Fal, DONE => "dbTags_master_Fal_1".modbusMaster.done, BUSY => "dbTags_master_Fal_1".modbusMaster.busy, ERROR => "dbTags_master_Fal_1".modbusMaster.error, STATUS => "dbTags_master_Fal_1".modbusMaster.status)
   END_RUNG
   RUNG wire#powerrail
      { S7_Templates := "SrcType := USInt" } EQ_Contact(in1 := "dbTags_master_Fal_1"."step", in2 := 12)
   END_RUNG wire#w1
   RUNG wire#powerrail
      Contact( "dbTags_master_Fal_1".modbusMaster.error )
      wire#w2
      { S7_GenerateENO := "TRUE" } Move(in := "dbTags_master_Fal_1".modbusMaster.status, out1 => "dbTags_master_Fal_1".modbusMaster.errorStatus)
   END_RUNG
   RUNG wire#w2
      { S7_GenerateENO := "TRUE" } Move(in := "db10datablock".received_zero, out1 => "dbModbusRTU_Reg".received26_Inver_DC_Voltage_416300)
   END_RUNG
   // the same network as SCL:
   IF ("dbTags_master_Fal_1"."step" = 11) OR ("dbTags_master_Fal_1"."step" = 12) THEN
       "MB_MASTER_DB"(REQ := "dbTags_master_Fal_1".modbusMaster.req,   // MB_MASTER
                      MB_ADDR := "dbTags_master_Fal_1".modbusMaster.mbAddr,
                      MODE := "dbTags_master_Fal_1".modbusMaster.mode,
                      DATA_ADDR := "dbTags_master_Fal_1".modbusMaster.dataAddr,
                      DATA_LEN := "dbTags_master_Fal_1".modbusMaster.dataLen,
                      DATA_PTR := "dbMasterData".ID26_Inver_DC_Voltage_416300_Fal,
                      DONE => "dbTags_master_Fal_1".modbusMaster.done,
                      BUSY => "dbTags_master_Fal_1".modbusMaster.busy,
                      ERROR => "dbTags_master_Fal_1".modbusMaster.error,
                      STATUS => "dbTags_master_Fal_1".modbusMaster.status);
   END_IF;
   IF "dbTags_master_Fal_1".modbusMaster.error THEN
       "dbTags_master_Fal_1".modbusMaster.errorStatus := "dbTags_master_Fal_1".modbusMaster.status;
       "dbModbusRTU_Reg".received26_Inver_DC_Voltage_416300 := "db10datablock".received_zero;
   END_IF;
END_REGION

REGION Network 23: step 6: save received data 416300
   RUNG wire#powerrail
      { S7_Templates := "SrcType := USInt" } EQ_Contact(in1 := "dbTags_master_Fal_1"."step", in2 := 12)
      Contact( "dbTags_master_Fal_1".modbusMaster.done )
      wire#w1
      { S7_GenerateENO := "TRUE" } Move(in := "dbMasterData".ID26_Inver_DC_Voltage_416300_Fal, out1 => "dbModbusRTU_Reg".received26_Inver_DC_Voltage_416300)
      R_Coil( "dbTags_master_Fal_1".modbusMaster.req )
   END_RUNG
   RUNG wire#w1
      { S7_GenerateENO := "TRUE" } Move(in := 13, out1 => "dbTags_master_Fal_1"."step")
   END_RUNG
   // the same network as SCL:
   // ENO of a box is taken as its EN; it also drops when the box reports an error
   IF ("dbTags_master_Fal_1"."step" = 12) AND "dbTags_master_Fal_1".modbusMaster.done THEN
       "dbModbusRTU_Reg".received26_Inver_DC_Voltage_416300 := "dbMasterData".ID26_Inver_DC_Voltage_416300_Fal;
       "dbTags_master_Fal_1".modbusMaster.req := FALSE;
       "dbTags_master_Fal_1"."step" := 13;
   END_IF;
END_REGION

REGION Network 25: MODBUS RTU adress 26*****step 7: read from slave temperature inverter
   // Pobieramy tęperaturę falownika
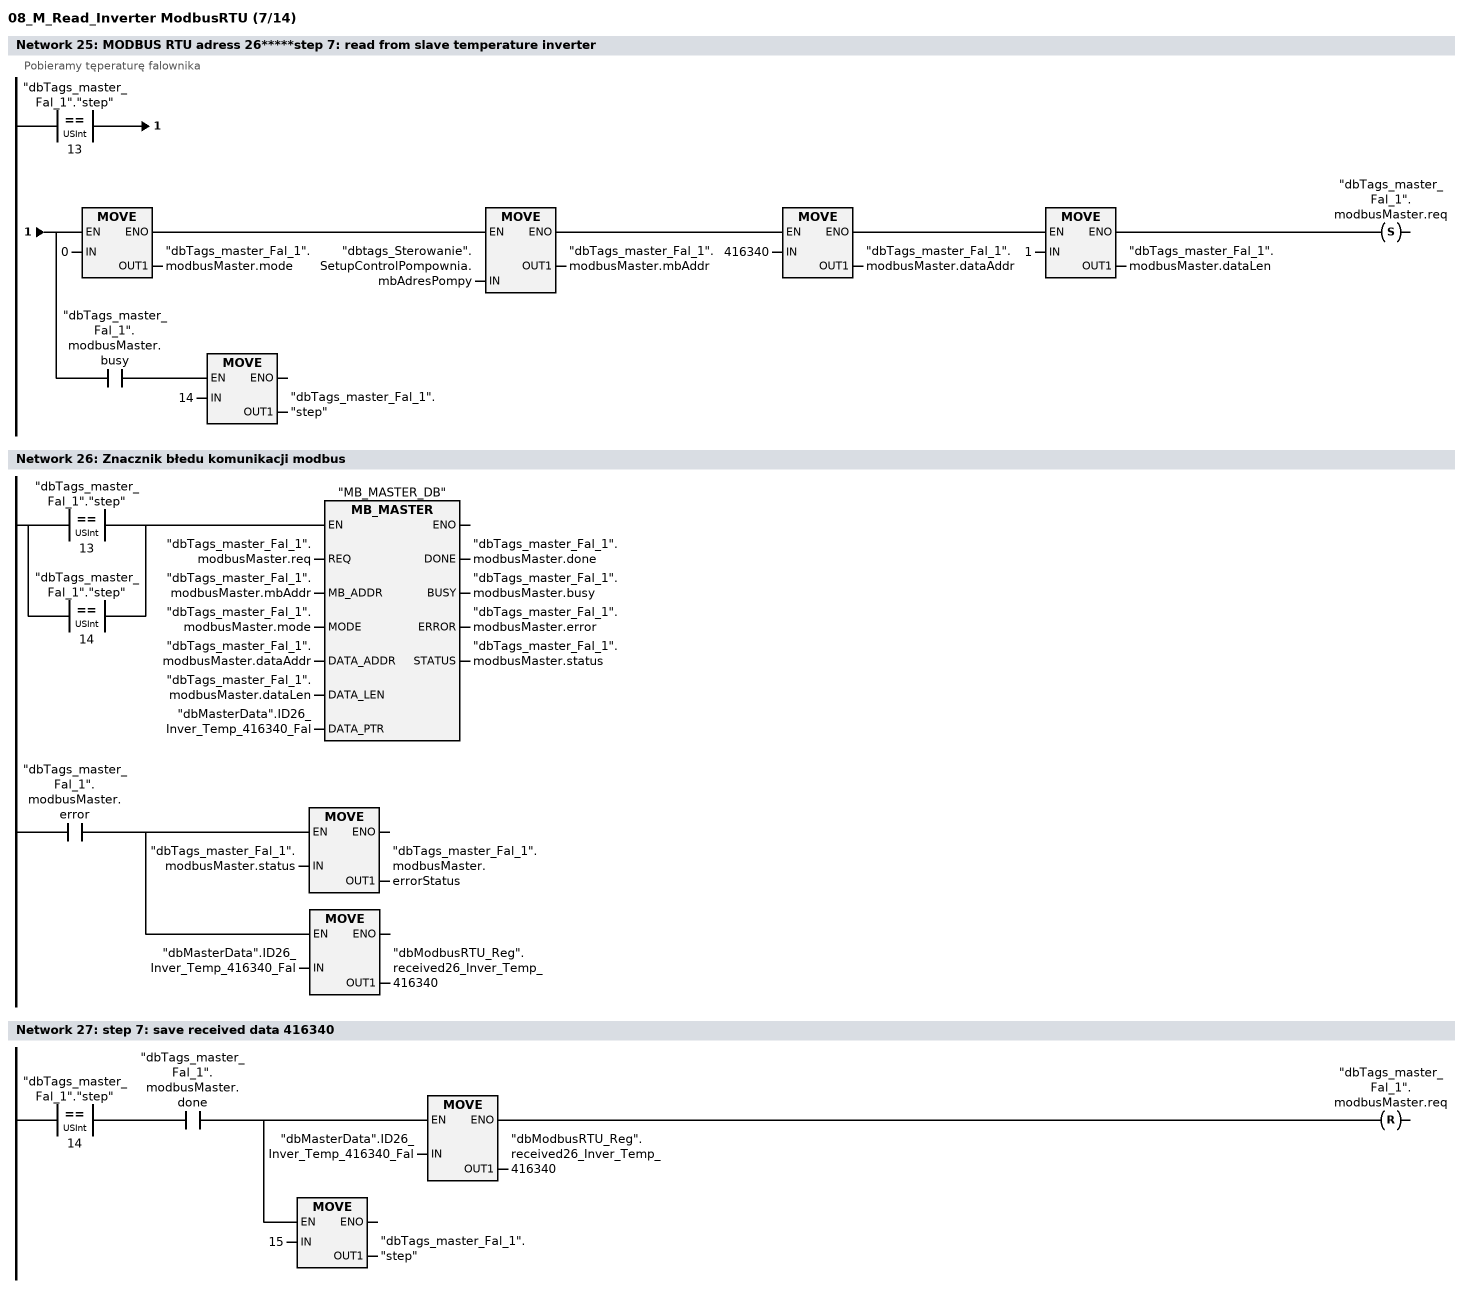
   RUNG wire#powerrail
      { S7_Templates := "SrcType := USInt" } EQ_Contact(in1 := "dbTags_master_Fal_1"."step", in2 := 13)
      wire#w1
      { S7_GenerateENO := "TRUE" } Move(in := 0, out1 => "dbTags_master_Fal_1".modbusMaster.mode)
      Move(in := "dbtags_Sterowanie".SetupControlPompownia.mbAdresPompy, out1 => "dbTags_master_Fal_1".modbusMaster.mbAddr)
      { S7_GenerateENO := "TRUE" } Move(in := 416340, out1 => "dbTags_master_Fal_1".modbusMaster.dataAddr)
      Move(in := 1, out1 => "dbTags_master_Fal_1".modbusMaster.dataLen)
      S_Coil( "dbTags_master_Fal_1".modbusMaster.req )
   END_RUNG
   RUNG wire#w1
      Contact( "dbTags_master_Fal_1".modbusMaster.busy )
      { S7_GenerateENO := "TRUE" } Move(in := 14, out1 => "dbTags_master_Fal_1"."step")
   END_RUNG
   // the same network as SCL:
   // ENO of a box is taken as its EN; it also drops when the box reports an error
   #_w1 := "dbTags_master_Fal_1"."step" = 13;
   IF #_w1 THEN
       "dbTags_master_Fal_1".modbusMaster.mode := 0;
       "dbTags_master_Fal_1".modbusMaster.mbAddr := "dbtags_Sterowanie".SetupControlPompownia.mbAdresPompy;
       "dbTags_master_Fal_1".modbusMaster.dataAddr := 416340;
       "dbTags_master_Fal_1".modbusMaster.dataLen := 1;
       "dbTags_master_Fal_1".modbusMaster.req := TRUE;
   END_IF;
   IF #_w1 AND "dbTags_master_Fal_1".modbusMaster.busy THEN "dbTags_master_Fal_1"."step" := 14; END_IF;
END_REGION

REGION Network 26: Znacznik błedu komunikacji modbus
   RUNG wire#powerrail
      { S7_Templates := "SrcType := USInt" } EQ_Contact(in1 := "dbTags_master_Fal_1"."step", in2 := 13)
      wire#w1
      "MB_MASTER_DB".MB_MASTER(REQ := "dbTags_master_Fal_1".modbusMaster.req, MB_ADDR := "dbTags_master_Fal_1".modbusMaster.mbAddr, MODE := "dbTags_master_Fal_1".modbusMaster.mode, DATA_ADDR := "dbTags_master_Fal_1".modbusMaster.dataAddr, DATA_LEN := "dbTags_master_Fal_1".modbusMaster.dataLen, DATA_PTR := "dbMasterData".ID26_Inver_Temp_416340_Fal, DONE => "dbTags_master_Fal_1".modbusMaster.done, BUSY => "dbTags_master_Fal_1".modbusMaster.busy, ERROR => "dbTags_master_Fal_1".modbusMaster.error, STATUS => "dbTags_master_Fal_1".modbusMaster.status)
   END_RUNG
   RUNG wire#powerrail
      { S7_Templates := "SrcType := USInt" } EQ_Contact(in1 := "dbTags_master_Fal_1"."step", in2 := 14)
   END_RUNG wire#w1
   RUNG wire#powerrail
      Contact( "dbTags_master_Fal_1".modbusMaster.error )
      wire#w2
      { S7_GenerateENO := "TRUE" } Move(in := "dbTags_master_Fal_1".modbusMaster.status, out1 => "dbTags_master_Fal_1".modbusMaster.errorStatus)
   END_RUNG
   RUNG wire#w2
      { S7_GenerateENO := "TRUE" } Move(in := "dbMasterData".ID26_Inver_Temp_416340_Fal, out1 => "dbModbusRTU_Reg".received26_Inver_Temp_416340)
   END_RUNG
   // the same network as SCL:
   IF ("dbTags_master_Fal_1"."step" = 13) OR ("dbTags_master_Fal_1"."step" = 14) THEN
       "MB_MASTER_DB"(REQ := "dbTags_master_Fal_1".modbusMaster.req,   // MB_MASTER
                      MB_ADDR := "dbTags_master_Fal_1".modbusMaster.mbAddr,
                      MODE := "dbTags_master_Fal_1".modbusMaster.mode,
                      DATA_ADDR := "dbTags_master_Fal_1".modbusMaster.dataAddr,
                      DATA_LEN := "dbTags_master_Fal_1".modbusMaster.dataLen,
                      DATA_PTR := "dbMasterData".ID26_Inver_Temp_416340_Fal,
                      DONE => "dbTags_master_Fal_1".modbusMaster.done,
                      BUSY => "dbTags_master_Fal_1".modbusMaster.busy,
                      ERROR => "dbTags_master_Fal_1".modbusMaster.error,
                      STATUS => "dbTags_master_Fal_1".modbusMaster.status);
   END_IF;
   IF "dbTags_master_Fal_1".modbusMaster.error THEN
       "dbTags_master_Fal_1".modbusMaster.errorStatus := "dbTags_master_Fal_1".modbusMaster.status;
       "dbModbusRTU_Reg".received26_Inver_Temp_416340 := "dbMasterData".ID26_Inver_Temp_416340_Fal;
   END_IF;
END_REGION

REGION Network 27: step 7: save received data 416340
   RUNG wire#powerrail
      { S7_Templates := "SrcType := USInt" } EQ_Contact(in1 := "dbTags_master_Fal_1"."step", in2 := 14)
      Contact( "dbTags_master_Fal_1".modbusMaster.done )
      wire#w1
      { S7_GenerateENO := "TRUE" } Move(in := "dbMasterData".ID26_Inver_Temp_416340_Fal, out1 => "dbModbusRTU_Reg".received26_Inver_Temp_416340)
      R_Coil( "dbTags_master_Fal_1".modbusMaster.req )
   END_RUNG
   RUNG wire#w1
      { S7_GenerateENO := "TRUE" } Move(in := 15, out1 => "dbTags_master_Fal_1"."step")
   END_RUNG
   // the same network as SCL:
   // ENO of a box is taken as its EN; it also drops when the box reports an error
   IF ("dbTags_master_Fal_1"."step" = 14) AND "dbTags_master_Fal_1".modbusMaster.done THEN
       "dbModbusRTU_Reg".received26_Inver_Temp_416340 := "dbMasterData".ID26_Inver_Temp_416340_Fal;
       "dbTags_master_Fal_1".modbusMaster.req := FALSE;
       "dbTags_master_Fal_1"."step" := 15;
   END_IF;
END_REGION

REGION Network 29: MODBUS RTU adress 26*****step 8: read from slave Normal Current
   // Pobieramy nominalną wartość prądu falownika (znamionowa ustawiona)
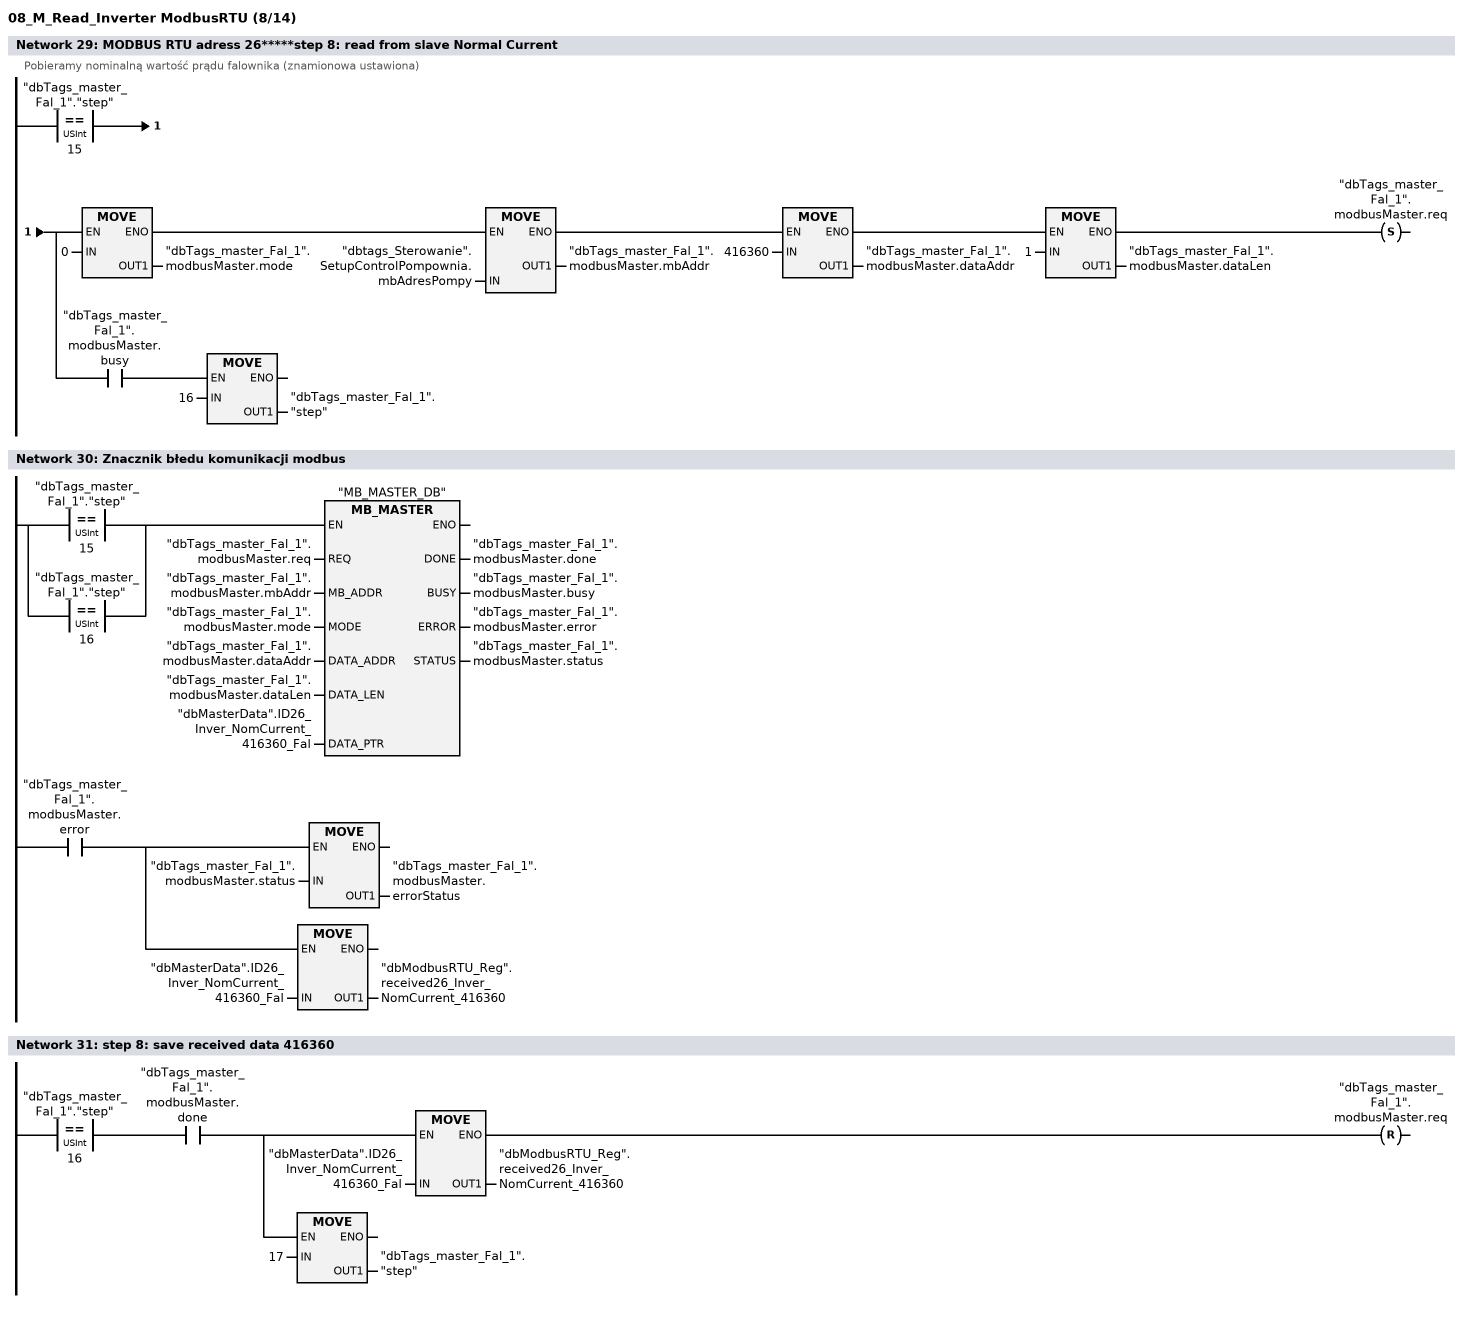
   RUNG wire#powerrail
      { S7_Templates := "SrcType := USInt" } EQ_Contact(in1 := "dbTags_master_Fal_1"."step", in2 := 15)
      wire#w1
      { S7_GenerateENO := "TRUE" } Move(in := 0, out1 => "dbTags_master_Fal_1".modbusMaster.mode)
      Move(in := "dbtags_Sterowanie".SetupControlPompownia.mbAdresPompy, out1 => "dbTags_master_Fal_1".modbusMaster.mbAddr)
      { S7_GenerateENO := "TRUE" } Move(in := 416360, out1 => "dbTags_master_Fal_1".modbusMaster.dataAddr)
      Move(in := 1, out1 => "dbTags_master_Fal_1".modbusMaster.dataLen)
      S_Coil( "dbTags_master_Fal_1".modbusMaster.req )
   END_RUNG
   RUNG wire#w1
      Contact( "dbTags_master_Fal_1".modbusMaster.busy )
      { S7_GenerateENO := "TRUE" } Move(in := 16, out1 => "dbTags_master_Fal_1"."step")
   END_RUNG
   // the same network as SCL:
   // ENO of a box is taken as its EN; it also drops when the box reports an error
   #_w1 := "dbTags_master_Fal_1"."step" = 15;
   IF #_w1 THEN
       "dbTags_master_Fal_1".modbusMaster.mode := 0;
       "dbTags_master_Fal_1".modbusMaster.mbAddr := "dbtags_Sterowanie".SetupControlPompownia.mbAdresPompy;
       "dbTags_master_Fal_1".modbusMaster.dataAddr := 416360;
       "dbTags_master_Fal_1".modbusMaster.dataLen := 1;
       "dbTags_master_Fal_1".modbusMaster.req := TRUE;
   END_IF;
   IF #_w1 AND "dbTags_master_Fal_1".modbusMaster.busy THEN "dbTags_master_Fal_1"."step" := 16; END_IF;
END_REGION

REGION Network 30: Znacznik błedu komunikacji modbus
   RUNG wire#powerrail
      { S7_Templates := "SrcType := USInt" } EQ_Contact(in1 := "dbTags_master_Fal_1"."step", in2 := 15)
      wire#w1
      "MB_MASTER_DB".MB_MASTER(REQ := "dbTags_master_Fal_1".modbusMaster.req, MB_ADDR := "dbTags_master_Fal_1".modbusMaster.mbAddr, MODE := "dbTags_master_Fal_1".modbusMaster.mode, DATA_ADDR := "dbTags_master_Fal_1".modbusMaster.dataAddr, DATA_LEN := "dbTags_master_Fal_1".modbusMaster.dataLen, DATA_PTR := "dbMasterData".ID26_Inver_NomCurrent_416360_Fal, DONE => "dbTags_master_Fal_1".modbusMaster.done, BUSY => "dbTags_master_Fal_1".modbusMaster.busy, ERROR => "dbTags_master_Fal_1".modbusMaster.error, STATUS => "dbTags_master_Fal_1".modbusMaster.status)
   END_RUNG
   RUNG wire#powerrail
      { S7_Templates := "SrcType := USInt" } EQ_Contact(in1 := "dbTags_master_Fal_1"."step", in2 := 16)
   END_RUNG wire#w1
   RUNG wire#powerrail
      Contact( "dbTags_master_Fal_1".modbusMaster.error )
      wire#w2
      { S7_GenerateENO := "TRUE" } Move(in := "dbTags_master_Fal_1".modbusMaster.status, out1 => "dbTags_master_Fal_1".modbusMaster.errorStatus)
   END_RUNG
   RUNG wire#w2
      { S7_GenerateENO := "TRUE" } Move(in := "dbMasterData".ID26_Inver_NomCurrent_416360_Fal, out1 => "dbModbusRTU_Reg".received26_Inver_NomCurrent_416360)
   END_RUNG
   // the same network as SCL:
   IF ("dbTags_master_Fal_1"."step" = 15) OR ("dbTags_master_Fal_1"."step" = 16) THEN
       "MB_MASTER_DB"(REQ := "dbTags_master_Fal_1".modbusMaster.req,   // MB_MASTER
                      MB_ADDR := "dbTags_master_Fal_1".modbusMaster.mbAddr,
                      MODE := "dbTags_master_Fal_1".modbusMaster.mode,
                      DATA_ADDR := "dbTags_master_Fal_1".modbusMaster.dataAddr,
                      DATA_LEN := "dbTags_master_Fal_1".modbusMaster.dataLen,
                      DATA_PTR := "dbMasterData".ID26_Inver_NomCurrent_416360_Fal,
                      DONE => "dbTags_master_Fal_1".modbusMaster.done,
                      BUSY => "dbTags_master_Fal_1".modbusMaster.busy,
                      ERROR => "dbTags_master_Fal_1".modbusMaster.error,
                      STATUS => "dbTags_master_Fal_1".modbusMaster.status);
   END_IF;
   IF "dbTags_master_Fal_1".modbusMaster.error THEN
       "dbTags_master_Fal_1".modbusMaster.errorStatus := "dbTags_master_Fal_1".modbusMaster.status;
       "dbModbusRTU_Reg".received26_Inver_NomCurrent_416360 := "dbMasterData".ID26_Inver_NomCurrent_416360_Fal;
   END_IF;
END_REGION

REGION Network 31: step 8: save received data 416360
   RUNG wire#powerrail
      { S7_Templates := "SrcType := USInt" } EQ_Contact(in1 := "dbTags_master_Fal_1"."step", in2 := 16)
      Contact( "dbTags_master_Fal_1".modbusMaster.done )
      wire#w1
      { S7_GenerateENO := "TRUE" } Move(in := "dbMasterData".ID26_Inver_NomCurrent_416360_Fal, out1 => "dbModbusRTU_Reg".received26_Inver_NomCurrent_416360)
      R_Coil( "dbTags_master_Fal_1".modbusMaster.req )
   END_RUNG
   RUNG wire#w1
      { S7_GenerateENO := "TRUE" } Move(in := 17, out1 => "dbTags_master_Fal_1"."step")
   END_RUNG
   // the same network as SCL:
   // ENO of a box is taken as its EN; it also drops when the box reports an error
   IF ("dbTags_master_Fal_1"."step" = 16) AND "dbTags_master_Fal_1".modbusMaster.done THEN
       "dbModbusRTU_Reg".received26_Inver_NomCurrent_416360 := "dbMasterData".ID26_Inver_NomCurrent_416360_Fal;
       "dbTags_master_Fal_1".modbusMaster.req := FALSE;
       "dbTags_master_Fal_1"."step" := 17;
   END_IF;
END_REGION

REGION Network 33: MODBUS RTU adress 26*****step 9: read from slave Max Current
   // Pobieramy dopuszczalnu maxymalny krótkotrwały
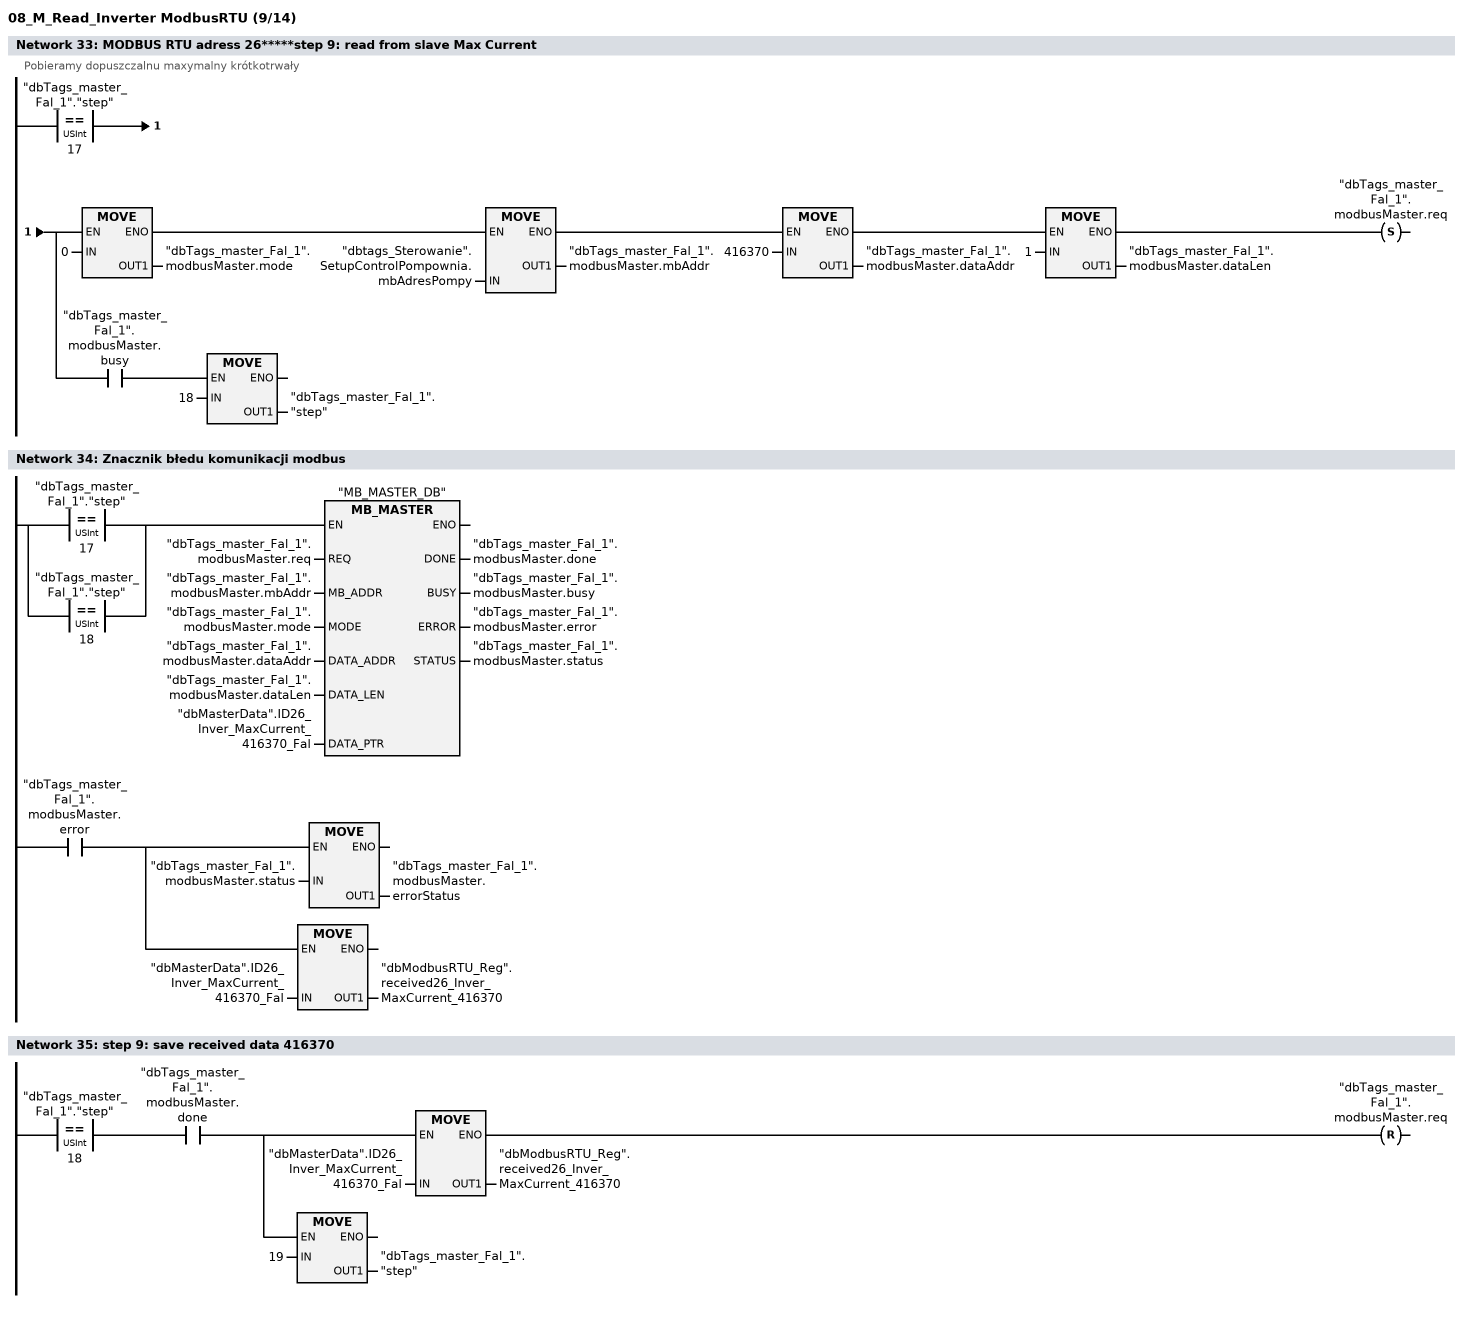
   RUNG wire#powerrail
      { S7_Templates := "SrcType := USInt" } EQ_Contact(in1 := "dbTags_master_Fal_1"."step", in2 := 17)
      wire#w1
      { S7_GenerateENO := "TRUE" } Move(in := 0, out1 => "dbTags_master_Fal_1".modbusMaster.mode)
      Move(in := "dbtags_Sterowanie".SetupControlPompownia.mbAdresPompy, out1 => "dbTags_master_Fal_1".modbusMaster.mbAddr)
      { S7_GenerateENO := "TRUE" } Move(in := 416370, out1 => "dbTags_master_Fal_1".modbusMaster.dataAddr)
      Move(in := 1, out1 => "dbTags_master_Fal_1".modbusMaster.dataLen)
      S_Coil( "dbTags_master_Fal_1".modbusMaster.req )
   END_RUNG
   RUNG wire#w1
      Contact( "dbTags_master_Fal_1".modbusMaster.busy )
      { S7_GenerateENO := "TRUE" } Move(in := 18, out1 => "dbTags_master_Fal_1"."step")
   END_RUNG
   // the same network as SCL:
   // ENO of a box is taken as its EN; it also drops when the box reports an error
   #_w1 := "dbTags_master_Fal_1"."step" = 17;
   IF #_w1 THEN
       "dbTags_master_Fal_1".modbusMaster.mode := 0;
       "dbTags_master_Fal_1".modbusMaster.mbAddr := "dbtags_Sterowanie".SetupControlPompownia.mbAdresPompy;
       "dbTags_master_Fal_1".modbusMaster.dataAddr := 416370;
       "dbTags_master_Fal_1".modbusMaster.dataLen := 1;
       "dbTags_master_Fal_1".modbusMaster.req := TRUE;
   END_IF;
   IF #_w1 AND "dbTags_master_Fal_1".modbusMaster.busy THEN "dbTags_master_Fal_1"."step" := 18; END_IF;
END_REGION

REGION Network 34: Znacznik błedu komunikacji modbus
   RUNG wire#powerrail
      { S7_Templates := "SrcType := USInt" } EQ_Contact(in1 := "dbTags_master_Fal_1"."step", in2 := 17)
      wire#w1
      "MB_MASTER_DB".MB_MASTER(REQ := "dbTags_master_Fal_1".modbusMaster.req, MB_ADDR := "dbTags_master_Fal_1".modbusMaster.mbAddr, MODE := "dbTags_master_Fal_1".modbusMaster.mode, DATA_ADDR := "dbTags_master_Fal_1".modbusMaster.dataAddr, DATA_LEN := "dbTags_master_Fal_1".modbusMaster.dataLen, DATA_PTR := "dbMasterData".ID26_Inver_MaxCurrent_416370_Fal, DONE => "dbTags_master_Fal_1".modbusMaster.done, BUSY => "dbTags_master_Fal_1".modbusMaster.busy, ERROR => "dbTags_master_Fal_1".modbusMaster.error, STATUS => "dbTags_master_Fal_1".modbusMaster.status)
   END_RUNG
   RUNG wire#powerrail
      { S7_Templates := "SrcType := USInt" } EQ_Contact(in1 := "dbTags_master_Fal_1"."step", in2 := 18)
   END_RUNG wire#w1
   RUNG wire#powerrail
      Contact( "dbTags_master_Fal_1".modbusMaster.error )
      wire#w2
      { S7_GenerateENO := "TRUE" } Move(in := "dbTags_master_Fal_1".modbusMaster.status, out1 => "dbTags_master_Fal_1".modbusMaster.errorStatus)
   END_RUNG
   RUNG wire#w2
      { S7_GenerateENO := "TRUE" } Move(in := "dbMasterData".ID26_Inver_MaxCurrent_416370_Fal, out1 => "dbModbusRTU_Reg".received26_Inver_MaxCurrent_416370)
   END_RUNG
   // the same network as SCL:
   IF ("dbTags_master_Fal_1"."step" = 17) OR ("dbTags_master_Fal_1"."step" = 18) THEN
       "MB_MASTER_DB"(REQ := "dbTags_master_Fal_1".modbusMaster.req,   // MB_MASTER
                      MB_ADDR := "dbTags_master_Fal_1".modbusMaster.mbAddr,
                      MODE := "dbTags_master_Fal_1".modbusMaster.mode,
                      DATA_ADDR := "dbTags_master_Fal_1".modbusMaster.dataAddr,
                      DATA_LEN := "dbTags_master_Fal_1".modbusMaster.dataLen,
                      DATA_PTR := "dbMasterData".ID26_Inver_MaxCurrent_416370_Fal,
                      DONE => "dbTags_master_Fal_1".modbusMaster.done,
                      BUSY => "dbTags_master_Fal_1".modbusMaster.busy,
                      ERROR => "dbTags_master_Fal_1".modbusMaster.error,
                      STATUS => "dbTags_master_Fal_1".modbusMaster.status);
   END_IF;
   IF "dbTags_master_Fal_1".modbusMaster.error THEN
       "dbTags_master_Fal_1".modbusMaster.errorStatus := "dbTags_master_Fal_1".modbusMaster.status;
       "dbModbusRTU_Reg".received26_Inver_MaxCurrent_416370 := "dbMasterData".ID26_Inver_MaxCurrent_416370_Fal;
   END_IF;
END_REGION

REGION Network 35: step 9: save received data 416370
   RUNG wire#powerrail
      { S7_Templates := "SrcType := USInt" } EQ_Contact(in1 := "dbTags_master_Fal_1"."step", in2 := 18)
      Contact( "dbTags_master_Fal_1".modbusMaster.done )
      wire#w1
      { S7_GenerateENO := "TRUE" } Move(in := "dbMasterData".ID26_Inver_MaxCurrent_416370_Fal, out1 => "dbModbusRTU_Reg".received26_Inver_MaxCurrent_416370)
      R_Coil( "dbTags_master_Fal_1".modbusMaster.req )
   END_RUNG
   RUNG wire#w1
      { S7_GenerateENO := "TRUE" } Move(in := 19, out1 => "dbTags_master_Fal_1"."step")
   END_RUNG
   // the same network as SCL:
   // ENO of a box is taken as its EN; it also drops when the box reports an error
   IF ("dbTags_master_Fal_1"."step" = 18) AND "dbTags_master_Fal_1".modbusMaster.done THEN
       "dbModbusRTU_Reg".received26_Inver_MaxCurrent_416370 := "dbMasterData".ID26_Inver_MaxCurrent_416370_Fal;
       "dbTags_master_Fal_1".modbusMaster.req := FALSE;
       "dbTags_master_Fal_1"."step" := 19;
   END_IF;
END_REGION

REGION Network 37: MODBUS RTU adress 26*****step 10: read from slave Input digital 18, 19,27,33
   // Pobieramy sygnał z wejść cyfrowych wej 18 Strat inverter =1
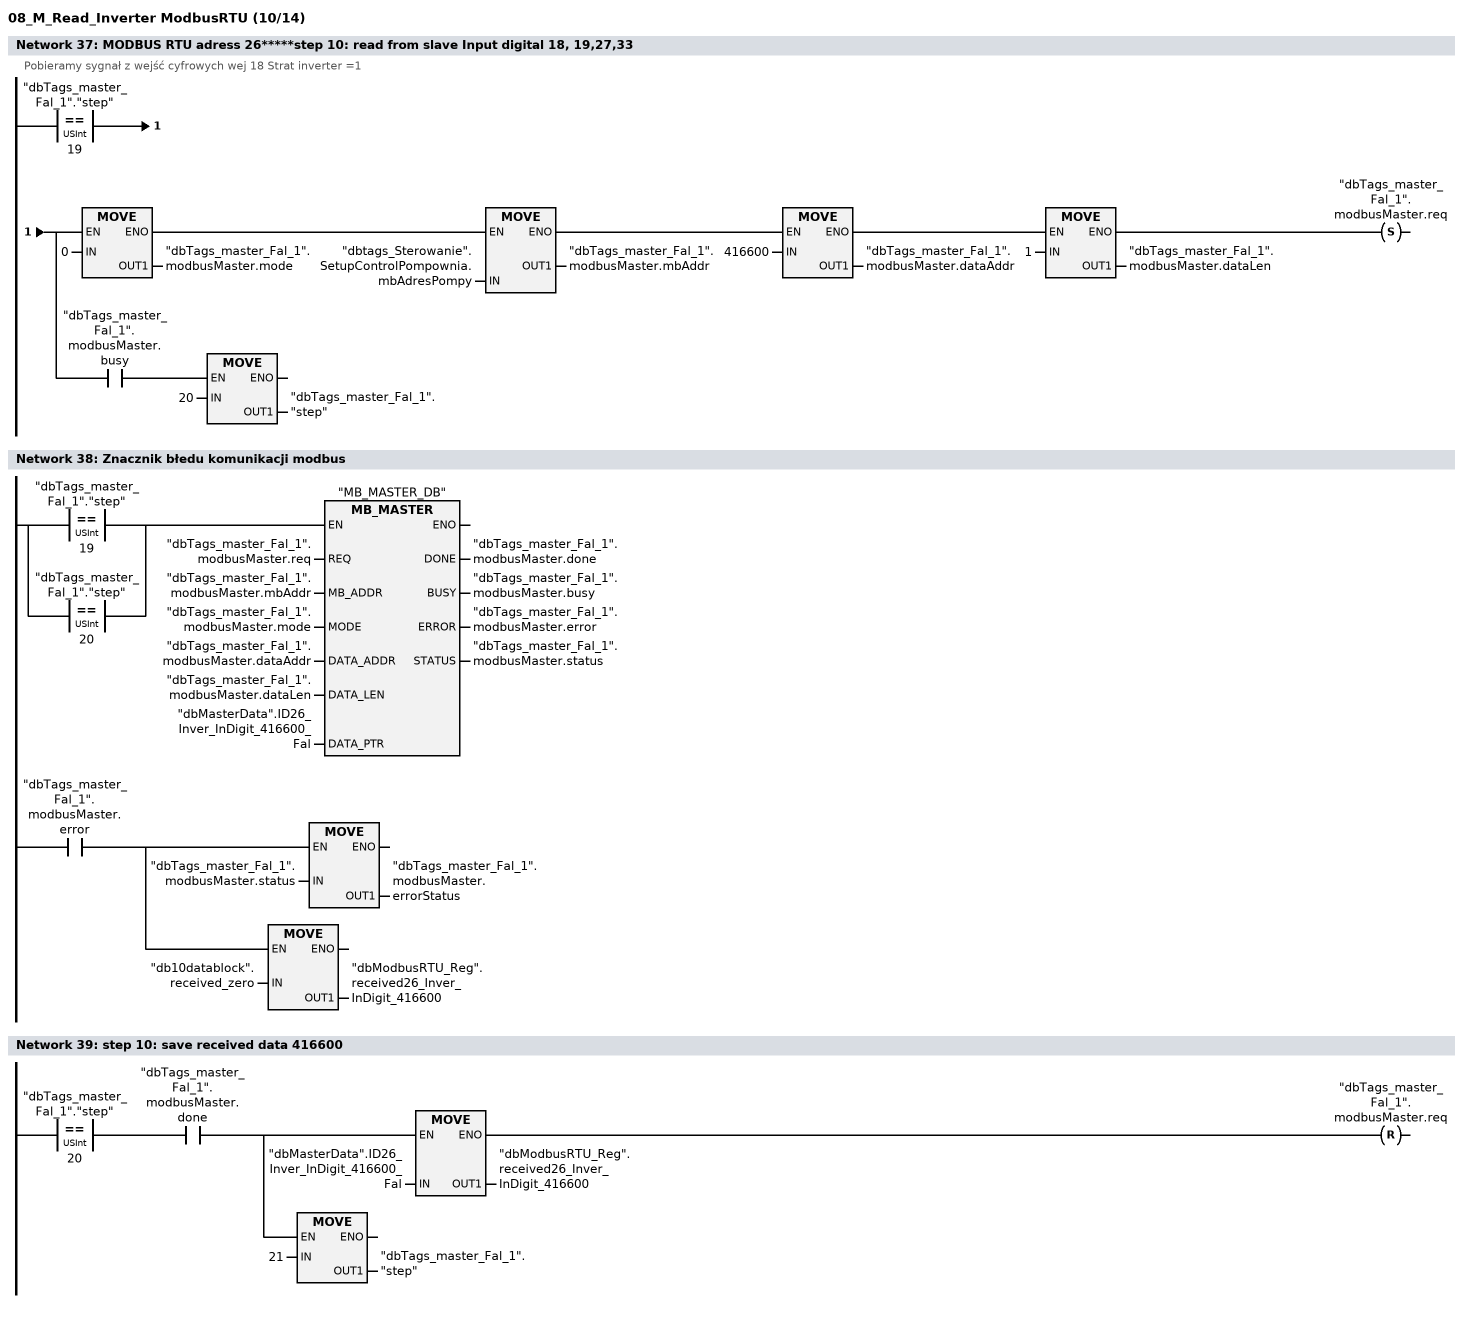
   RUNG wire#powerrail
      { S7_Templates := "SrcType := USInt" } EQ_Contact(in1 := "dbTags_master_Fal_1"."step", in2 := 19)
      wire#w1
      { S7_GenerateENO := "TRUE" } Move(in := 0, out1 => "dbTags_master_Fal_1".modbusMaster.mode)
      Move(in := "dbtags_Sterowanie".SetupControlPompownia.mbAdresPompy, out1 => "dbTags_master_Fal_1".modbusMaster.mbAddr)
      { S7_GenerateENO := "TRUE" } Move(in := 416600, out1 => "dbTags_master_Fal_1".modbusMaster.dataAddr)
      Move(in := 1, out1 => "dbTags_master_Fal_1".modbusMaster.dataLen)
      S_Coil( "dbTags_master_Fal_1".modbusMaster.req )
   END_RUNG
   RUNG wire#w1
      Contact( "dbTags_master_Fal_1".modbusMaster.busy )
      { S7_GenerateENO := "TRUE" } Move(in := 20, out1 => "dbTags_master_Fal_1"."step")
   END_RUNG
   // the same network as SCL:
   // ENO of a box is taken as its EN; it also drops when the box reports an error
   #_w1 := "dbTags_master_Fal_1"."step" = 19;
   IF #_w1 THEN
       "dbTags_master_Fal_1".modbusMaster.mode := 0;
       "dbTags_master_Fal_1".modbusMaster.mbAddr := "dbtags_Sterowanie".SetupControlPompownia.mbAdresPompy;
       "dbTags_master_Fal_1".modbusMaster.dataAddr := 416600;
       "dbTags_master_Fal_1".modbusMaster.dataLen := 1;
       "dbTags_master_Fal_1".modbusMaster.req := TRUE;
   END_IF;
   IF #_w1 AND "dbTags_master_Fal_1".modbusMaster.busy THEN "dbTags_master_Fal_1"."step" := 20; END_IF;
END_REGION

REGION Network 38: Znacznik błedu komunikacji modbus
   RUNG wire#powerrail
      { S7_Templates := "SrcType := USInt" } EQ_Contact(in1 := "dbTags_master_Fal_1"."step", in2 := 19)
      wire#w1
      "MB_MASTER_DB".MB_MASTER(REQ := "dbTags_master_Fal_1".modbusMaster.req, MB_ADDR := "dbTags_master_Fal_1".modbusMaster.mbAddr, MODE := "dbTags_master_Fal_1".modbusMaster.mode, DATA_ADDR := "dbTags_master_Fal_1".modbusMaster.dataAddr, DATA_LEN := "dbTags_master_Fal_1".modbusMaster.dataLen, DATA_PTR := "dbMasterData".ID26_Inver_InDigit_416600_Fal, DONE => "dbTags_master_Fal_1".modbusMaster.done, BUSY => "dbTags_master_Fal_1".modbusMaster.busy, ERROR => "dbTags_master_Fal_1".modbusMaster.error, STATUS => "dbTags_master_Fal_1".modbusMaster.status)
   END_RUNG
   RUNG wire#powerrail
      { S7_Templates := "SrcType := USInt" } EQ_Contact(in1 := "dbTags_master_Fal_1"."step", in2 := 20)
   END_RUNG wire#w1
   RUNG wire#powerrail
      Contact( "dbTags_master_Fal_1".modbusMaster.error )
      wire#w2
      { S7_GenerateENO := "TRUE" } Move(in := "dbTags_master_Fal_1".modbusMaster.status, out1 => "dbTags_master_Fal_1".modbusMaster.errorStatus)
   END_RUNG
   RUNG wire#w2
      { S7_GenerateENO := "TRUE" } Move(in := "db10datablock".received_zero, out1 => "dbModbusRTU_Reg".received26_Inver_InDigit_416600)
   END_RUNG
   // the same network as SCL:
   IF ("dbTags_master_Fal_1"."step" = 19) OR ("dbTags_master_Fal_1"."step" = 20) THEN
       "MB_MASTER_DB"(REQ := "dbTags_master_Fal_1".modbusMaster.req,   // MB_MASTER
                      MB_ADDR := "dbTags_master_Fal_1".modbusMaster.mbAddr,
                      MODE := "dbTags_master_Fal_1".modbusMaster.mode,
                      DATA_ADDR := "dbTags_master_Fal_1".modbusMaster.dataAddr,
                      DATA_LEN := "dbTags_master_Fal_1".modbusMaster.dataLen,
                      DATA_PTR := "dbMasterData".ID26_Inver_InDigit_416600_Fal,
                      DONE => "dbTags_master_Fal_1".modbusMaster.done,
                      BUSY => "dbTags_master_Fal_1".modbusMaster.busy,
                      ERROR => "dbTags_master_Fal_1".modbusMaster.error,
                      STATUS => "dbTags_master_Fal_1".modbusMaster.status);
   END_IF;
   IF "dbTags_master_Fal_1".modbusMaster.error THEN
       "dbTags_master_Fal_1".modbusMaster.errorStatus := "dbTags_master_Fal_1".modbusMaster.status;
       "dbModbusRTU_Reg".received26_Inver_InDigit_416600 := "db10datablock".received_zero;
   END_IF;
END_REGION

REGION Network 39: step 10: save received data 416600
   RUNG wire#powerrail
      { S7_Templates := "SrcType := USInt" } EQ_Contact(in1 := "dbTags_master_Fal_1"."step", in2 := 20)
      Contact( "dbTags_master_Fal_1".modbusMaster.done )
      wire#w1
      { S7_GenerateENO := "TRUE" } Move(in := "dbMasterData".ID26_Inver_InDigit_416600_Fal, out1 => "dbModbusRTU_Reg".received26_Inver_InDigit_416600)
      R_Coil( "dbTags_master_Fal_1".modbusMaster.req )
   END_RUNG
   RUNG wire#w1
      { S7_GenerateENO := "TRUE" } Move(in := 21, out1 => "dbTags_master_Fal_1"."step")
   END_RUNG
   // the same network as SCL:
   // ENO of a box is taken as its EN; it also drops when the box reports an error
   IF ("dbTags_master_Fal_1"."step" = 20) AND "dbTags_master_Fal_1".modbusMaster.done THEN
       "dbModbusRTU_Reg".received26_Inver_InDigit_416600 := "dbMasterData".ID26_Inver_InDigit_416600_Fal;
       "dbTags_master_Fal_1".modbusMaster.req := FALSE;
       "dbTags_master_Fal_1"."step" := 21;
   END_IF;
END_REGION

REGION Network 40: MODBUS RTU adress 26*****step 11: read from slave Over Temperature
   // Pobieramy rejestr przekroczenia temperatury silnika wyliczany przez falownik
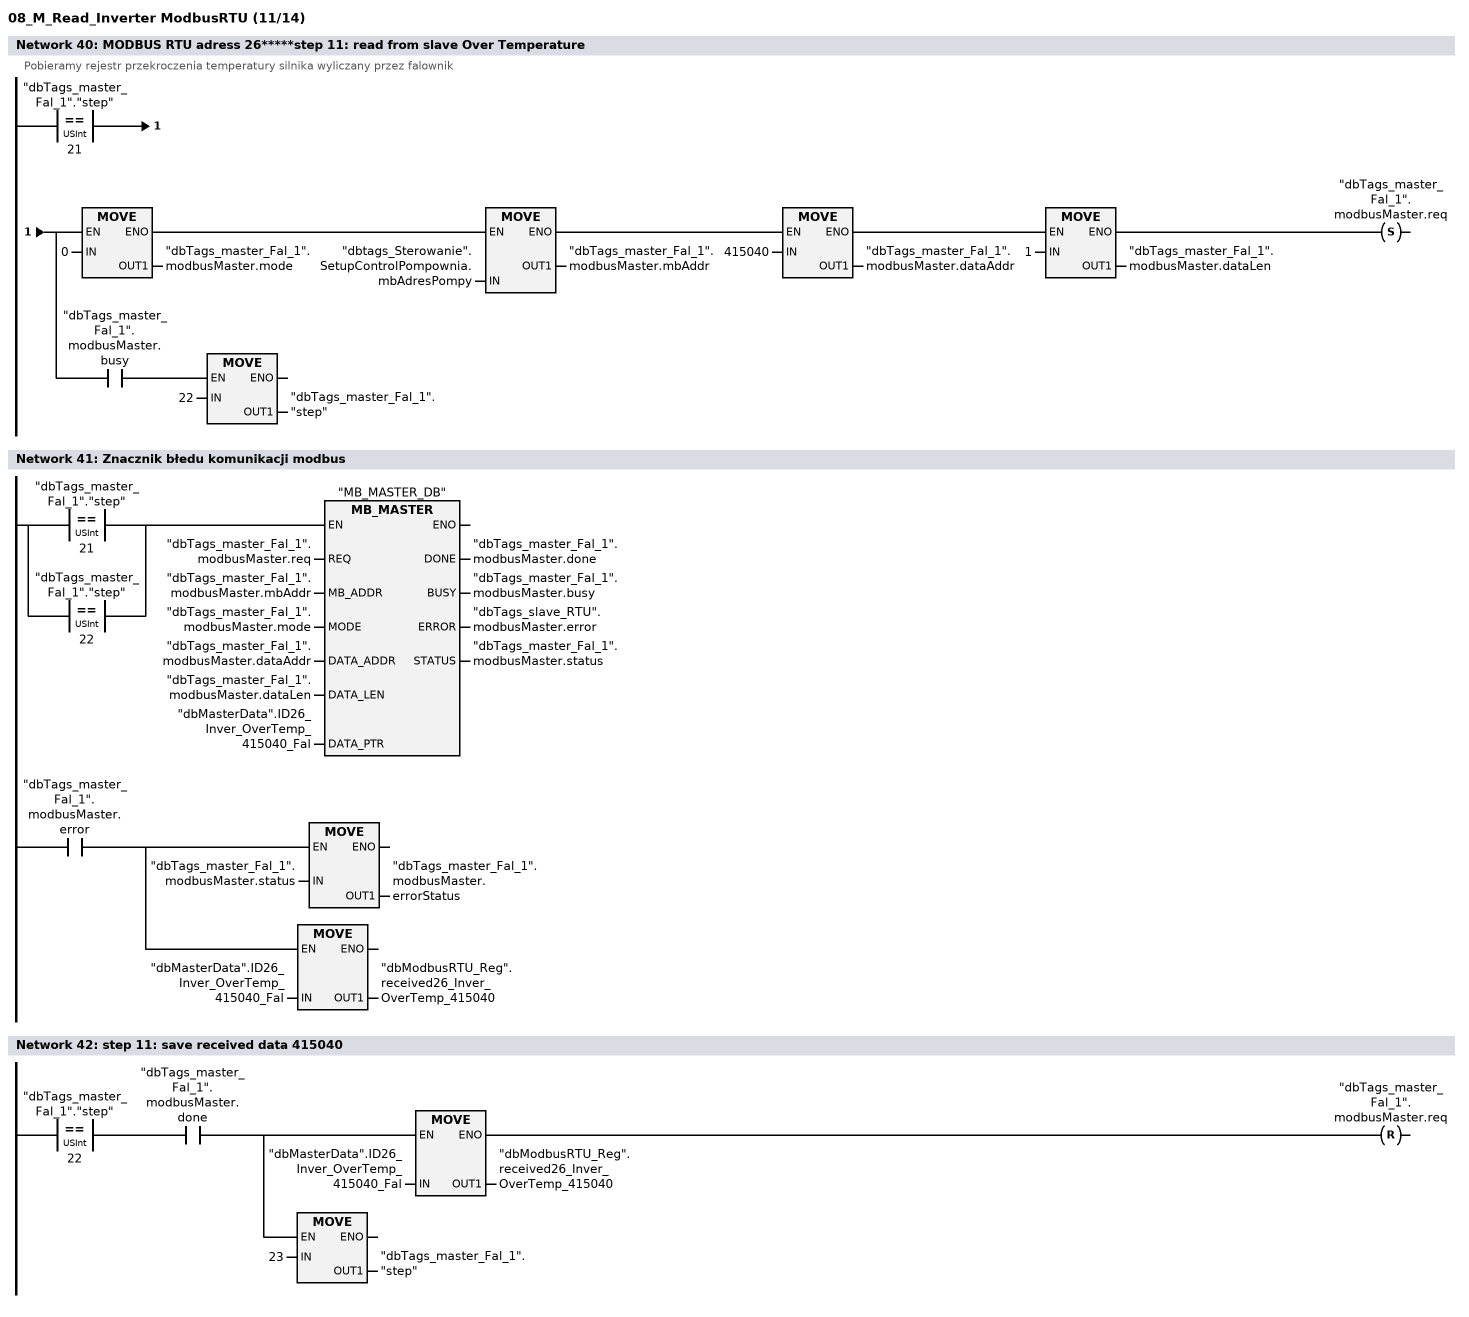
   RUNG wire#powerrail
      { S7_Templates := "SrcType := USInt" } EQ_Contact(in1 := "dbTags_master_Fal_1"."step", in2 := 21)
      wire#w1
      { S7_GenerateENO := "TRUE" } Move(in := 0, out1 => "dbTags_master_Fal_1".modbusMaster.mode)
      Move(in := "dbtags_Sterowanie".SetupControlPompownia.mbAdresPompy, out1 => "dbTags_master_Fal_1".modbusMaster.mbAddr)
      { S7_GenerateENO := "TRUE" } Move(in := 415040, out1 => "dbTags_master_Fal_1".modbusMaster.dataAddr)
      Move(in := 1, out1 => "dbTags_master_Fal_1".modbusMaster.dataLen)
      S_Coil( "dbTags_master_Fal_1".modbusMaster.req )
   END_RUNG
   RUNG wire#w1
      Contact( "dbTags_master_Fal_1".modbusMaster.busy )
      { S7_GenerateENO := "TRUE" } Move(in := 22, out1 => "dbTags_master_Fal_1"."step")
   END_RUNG
   // the same network as SCL:
   // ENO of a box is taken as its EN; it also drops when the box reports an error
   #_w1 := "dbTags_master_Fal_1"."step" = 21;
   IF #_w1 THEN
       "dbTags_master_Fal_1".modbusMaster.mode := 0;
       "dbTags_master_Fal_1".modbusMaster.mbAddr := "dbtags_Sterowanie".SetupControlPompownia.mbAdresPompy;
       "dbTags_master_Fal_1".modbusMaster.dataAddr := 415040;
       "dbTags_master_Fal_1".modbusMaster.dataLen := 1;
       "dbTags_master_Fal_1".modbusMaster.req := TRUE;
   END_IF;
   IF #_w1 AND "dbTags_master_Fal_1".modbusMaster.busy THEN "dbTags_master_Fal_1"."step" := 22; END_IF;
END_REGION

REGION Network 41: Znacznik błedu komunikacji modbus
   RUNG wire#powerrail
      { S7_Templates := "SrcType := USInt" } EQ_Contact(in1 := "dbTags_master_Fal_1"."step", in2 := 21)
      wire#w1
      "MB_MASTER_DB".MB_MASTER(REQ := "dbTags_master_Fal_1".modbusMaster.req, MB_ADDR := "dbTags_master_Fal_1".modbusMaster.mbAddr, MODE := "dbTags_master_Fal_1".modbusMaster.mode, DATA_ADDR := "dbTags_master_Fal_1".modbusMaster.dataAddr, DATA_LEN := "dbTags_master_Fal_1".modbusMaster.dataLen, DATA_PTR := "dbMasterData".ID26_Inver_OverTemp_415040_Fal, DONE => "dbTags_master_Fal_1".modbusMaster.done, BUSY => "dbTags_master_Fal_1".modbusMaster.busy, ERROR => "dbTags_slave_RTU".modbusMaster.error, STATUS => "dbTags_master_Fal_1".modbusMaster.status)
   END_RUNG
   RUNG wire#powerrail
      { S7_Templates := "SrcType := USInt" } EQ_Contact(in1 := "dbTags_master_Fal_1"."step", in2 := 22)
   END_RUNG wire#w1
   RUNG wire#powerrail
      Contact( "dbTags_master_Fal_1".modbusMaster.error )
      wire#w2
      { S7_GenerateENO := "TRUE" } Move(in := "dbTags_master_Fal_1".modbusMaster.status, out1 => "dbTags_master_Fal_1".modbusMaster.errorStatus)
   END_RUNG
   RUNG wire#w2
      { S7_GenerateENO := "TRUE" } Move(in := "dbMasterData".ID26_Inver_OverTemp_415040_Fal, out1 => "dbModbusRTU_Reg".received26_Inver_OverTemp_415040)
   END_RUNG
   // the same network as SCL:
   IF ("dbTags_master_Fal_1"."step" = 21) OR ("dbTags_master_Fal_1"."step" = 22) THEN
       "MB_MASTER_DB"(REQ := "dbTags_master_Fal_1".modbusMaster.req,   // MB_MASTER
                      MB_ADDR := "dbTags_master_Fal_1".modbusMaster.mbAddr,
                      MODE := "dbTags_master_Fal_1".modbusMaster.mode,
                      DATA_ADDR := "dbTags_master_Fal_1".modbusMaster.dataAddr,
                      DATA_LEN := "dbTags_master_Fal_1".modbusMaster.dataLen,
                      DATA_PTR := "dbMasterData".ID26_Inver_OverTemp_415040_Fal,
                      DONE => "dbTags_master_Fal_1".modbusMaster.done,
                      BUSY => "dbTags_master_Fal_1".modbusMaster.busy,
                      ERROR => "dbTags_slave_RTU".modbusMaster.error,
                      STATUS => "dbTags_master_Fal_1".modbusMaster.status);
   END_IF;
   IF "dbTags_master_Fal_1".modbusMaster.error THEN
       "dbTags_master_Fal_1".modbusMaster.errorStatus := "dbTags_master_Fal_1".modbusMaster.status;
       "dbModbusRTU_Reg".received26_Inver_OverTemp_415040 := "dbMasterData".ID26_Inver_OverTemp_415040_Fal;
   END_IF;
END_REGION

REGION Network 42: step 11: save received data 415040
   RUNG wire#powerrail
      { S7_Templates := "SrcType := USInt" } EQ_Contact(in1 := "dbTags_master_Fal_1"."step", in2 := 22)
      Contact( "dbTags_master_Fal_1".modbusMaster.done )
      wire#w1
      { S7_GenerateENO := "TRUE" } Move(in := "dbMasterData".ID26_Inver_OverTemp_415040_Fal, out1 => "dbModbusRTU_Reg".received26_Inver_OverTemp_415040)
      R_Coil( "dbTags_master_Fal_1".modbusMaster.req )
   END_RUNG
   RUNG wire#w1
      { S7_GenerateENO := "TRUE" } Move(in := 23, out1 => "dbTags_master_Fal_1"."step")
   END_RUNG
   // the same network as SCL:
   // ENO of a box is taken as its EN; it also drops when the box reports an error
   IF ("dbTags_master_Fal_1"."step" = 22) AND "dbTags_master_Fal_1".modbusMaster.done THEN
       "dbModbusRTU_Reg".received26_Inver_OverTemp_415040 := "dbMasterData".ID26_Inver_OverTemp_415040_Fal;
       "dbTags_master_Fal_1".modbusMaster.req := FALSE;
       "dbTags_master_Fal_1"."step" := 23;
   END_IF;
END_REGION

REGION Network 44: MODBUS RTU adress 26*****step 12: read from slave Over Voltage
   // Pobieramy rejestr przekroczenia napięcia maxymalnego
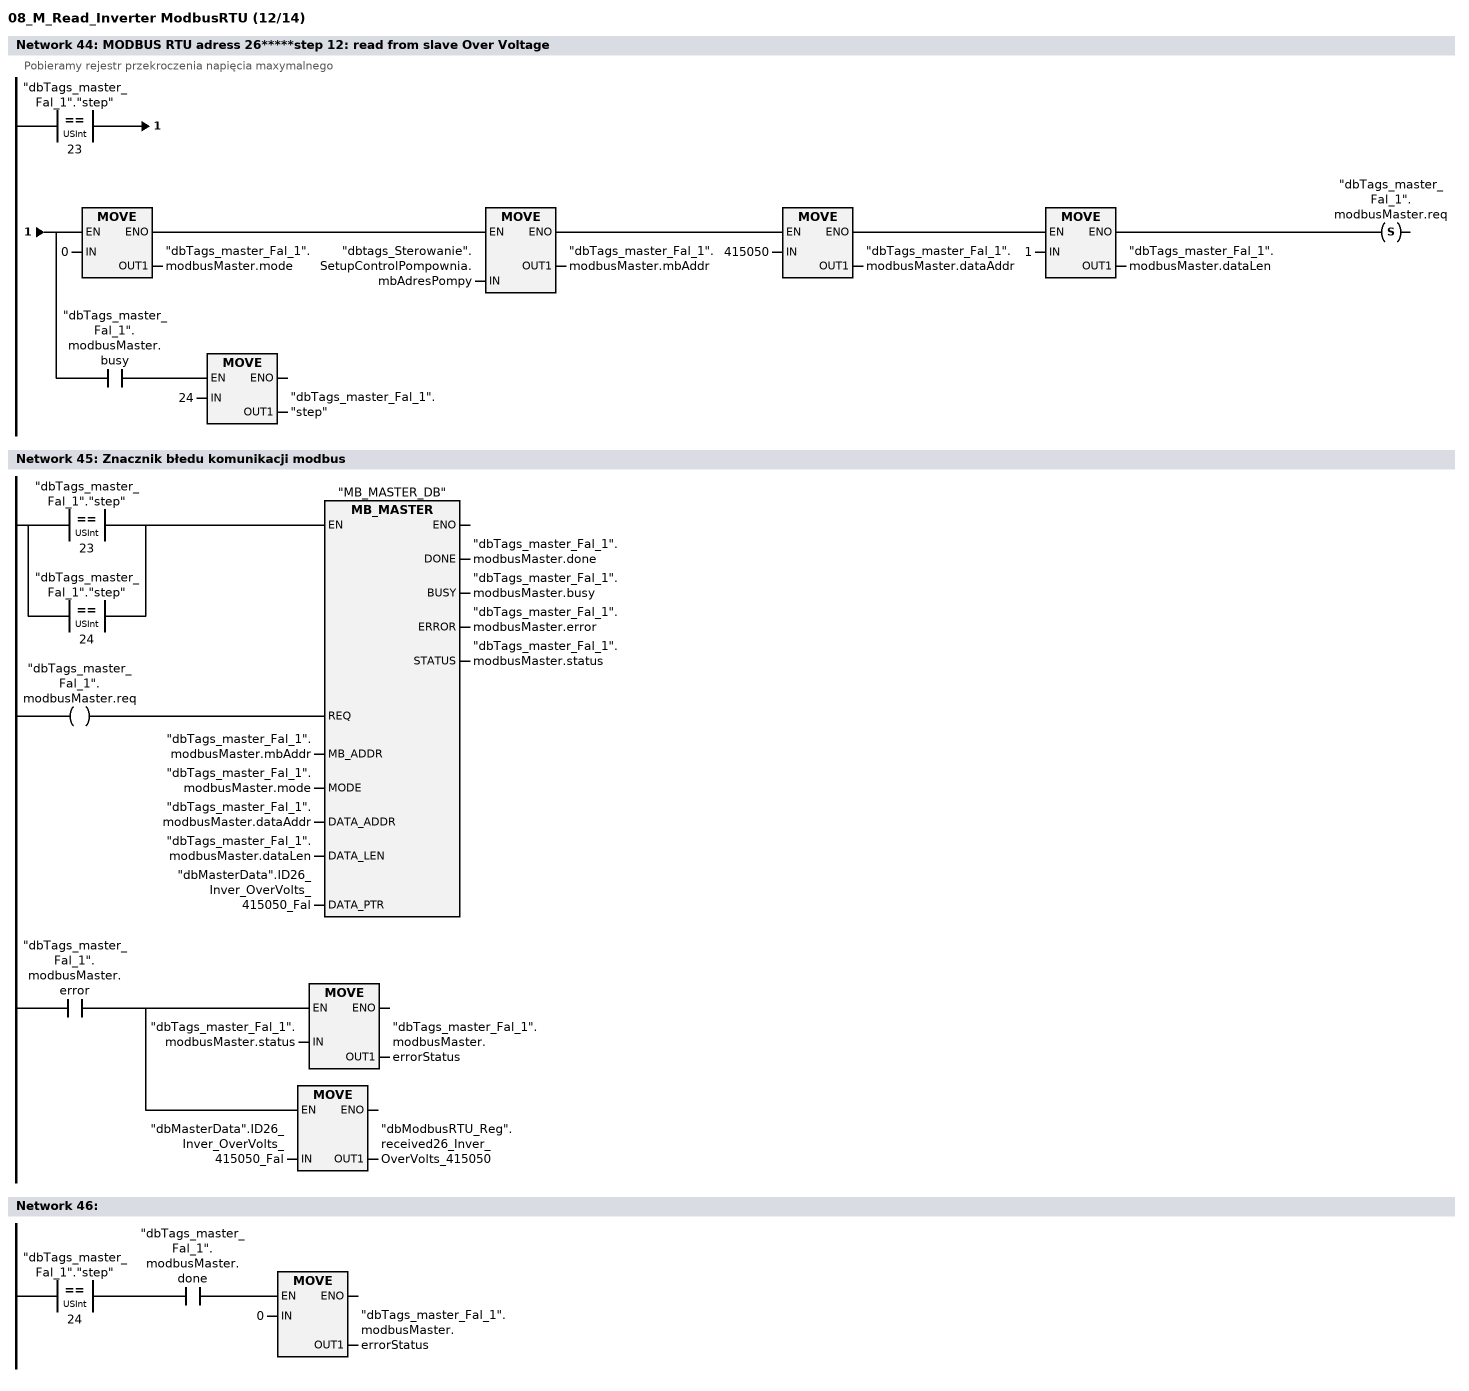
   RUNG wire#powerrail
      { S7_Templates := "SrcType := USInt" } EQ_Contact(in1 := "dbTags_master_Fal_1"."step", in2 := 23)
      wire#w1
      { S7_GenerateENO := "TRUE" } Move(in := 0, out1 => "dbTags_master_Fal_1".modbusMaster.mode)
      Move(in := "dbtags_Sterowanie".SetupControlPompownia.mbAdresPompy, out1 => "dbTags_master_Fal_1".modbusMaster.mbAddr)
      { S7_GenerateENO := "TRUE" } Move(in := 415050, out1 => "dbTags_master_Fal_1".modbusMaster.dataAddr)
      Move(in := 1, out1 => "dbTags_master_Fal_1".modbusMaster.dataLen)
      S_Coil( "dbTags_master_Fal_1".modbusMaster.req )
   END_RUNG
   RUNG wire#w1
      Contact( "dbTags_master_Fal_1".modbusMaster.busy )
      { S7_GenerateENO := "TRUE" } Move(in := 24, out1 => "dbTags_master_Fal_1"."step")
   END_RUNG
   // the same network as SCL:
   // ENO of a box is taken as its EN; it also drops when the box reports an error
   #_w1 := "dbTags_master_Fal_1"."step" = 23;
   IF #_w1 THEN
       "dbTags_master_Fal_1".modbusMaster.mode := 0;
       "dbTags_master_Fal_1".modbusMaster.mbAddr := "dbtags_Sterowanie".SetupControlPompownia.mbAdresPompy;
       "dbTags_master_Fal_1".modbusMaster.dataAddr := 415050;
       "dbTags_master_Fal_1".modbusMaster.dataLen := 1;
       "dbTags_master_Fal_1".modbusMaster.req := TRUE;
   END_IF;
   IF #_w1 AND "dbTags_master_Fal_1".modbusMaster.busy THEN "dbTags_master_Fal_1"."step" := 24; END_IF;
END_REGION

REGION Network 45: Znacznik błedu komunikacji modbus
   RUNG wire#powerrail
      { S7_Templates := "SrcType := USInt" } EQ_Contact(in1 := "dbTags_master_Fal_1"."step", in2 := 23)
      wire#w1
      "MB_MASTER_DB".MB_MASTER(REQ := wire#w2, MB_ADDR := "dbTags_master_Fal_1".modbusMaster.mbAddr, MODE := "dbTags_master_Fal_1".modbusMaster.mode, DATA_ADDR := "dbTags_master_Fal_1".modbusMaster.dataAddr, DATA_LEN := "dbTags_master_Fal_1".modbusMaster.dataLen, DATA_PTR := "dbMasterData".ID26_Inver_OverVolts_415050_Fal, DONE => "dbTags_master_Fal_1".modbusMaster.done, BUSY => "dbTags_master_Fal_1".modbusMaster.busy, ERROR => "dbTags_master_Fal_1".modbusMaster.error, STATUS => "dbTags_master_Fal_1".modbusMaster.status)
   END_RUNG
   RUNG wire#powerrail
      { S7_Templates := "SrcType := USInt" } EQ_Contact(in1 := "dbTags_master_Fal_1"."step", in2 := 24)
   END_RUNG wire#w1
   RUNG wire#powerrail
      Coil( "dbTags_master_Fal_1".modbusMaster.req )
   END_RUNG wire#w2
   RUNG wire#powerrail
      Contact( "dbTags_master_Fal_1".modbusMaster.error )
      wire#w3
      { S7_GenerateENO := "TRUE" } Move(in := "dbTags_master_Fal_1".modbusMaster.status, out1 => "dbTags_master_Fal_1".modbusMaster.errorStatus)
   END_RUNG
   RUNG wire#w3
      { S7_GenerateENO := "TRUE" } Move(in := "dbMasterData".ID26_Inver_OverVolts_415050_Fal, out1 => "dbModbusRTU_Reg".received26_Inver_OverVolts_415050)
   END_RUNG
   // the same network as SCL:
   "dbTags_master_Fal_1".modbusMaster.req := TRUE;
   IF ("dbTags_master_Fal_1"."step" = 23) OR ("dbTags_master_Fal_1"."step" = 24) THEN
       "MB_MASTER_DB"(REQ := TRUE,   // MB_MASTER
                      MB_ADDR := "dbTags_master_Fal_1".modbusMaster.mbAddr,
                      MODE := "dbTags_master_Fal_1".modbusMaster.mode,
                      DATA_ADDR := "dbTags_master_Fal_1".modbusMaster.dataAddr,
                      DATA_LEN := "dbTags_master_Fal_1".modbusMaster.dataLen,
                      DATA_PTR := "dbMasterData".ID26_Inver_OverVolts_415050_Fal,
                      DONE => "dbTags_master_Fal_1".modbusMaster.done,
                      BUSY => "dbTags_master_Fal_1".modbusMaster.busy,
                      ERROR => "dbTags_master_Fal_1".modbusMaster.error,
                      STATUS => "dbTags_master_Fal_1".modbusMaster.status);
   END_IF;
   IF "dbTags_master_Fal_1".modbusMaster.error THEN
       "dbTags_master_Fal_1".modbusMaster.errorStatus := "dbTags_master_Fal_1".modbusMaster.status;
       "dbModbusRTU_Reg".received26_Inver_OverVolts_415050 := "dbMasterData".ID26_Inver_OverVolts_415050_Fal;
   END_IF;
END_REGION

REGION Network 46
   RUNG wire#powerrail
      { S7_Templates := "SrcType := USInt" } EQ_Contact(in1 := "dbTags_master_Fal_1"."step", in2 := 24)
      Contact( "dbTags_master_Fal_1".modbusMaster.done )
      { S7_GenerateENO := "TRUE" } Move(in := 0, out1 => "dbTags_master_Fal_1".modbusMaster.errorStatus)
   END_RUNG
   // the same network as SCL:
   IF ("dbTags_master_Fal_1"."step" = 24) AND "dbTags_master_Fal_1".modbusMaster.done THEN
       "dbTags_master_Fal_1".modbusMaster.errorStatus := 0;
   END_IF;
END_REGION

REGION Network 47: step 12: save received data 415050
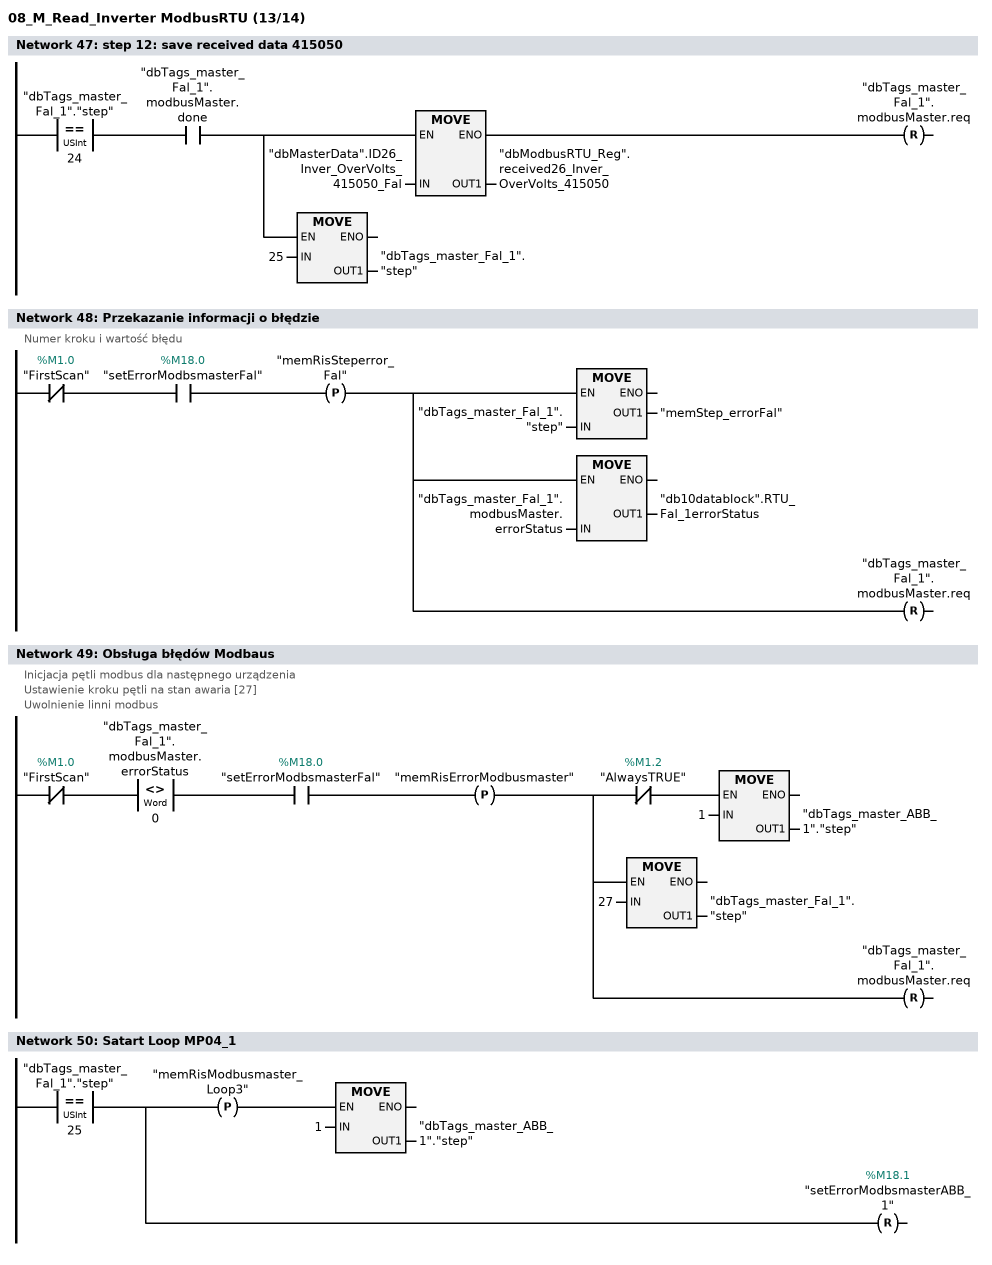
   RUNG wire#powerrail
      { S7_Templates := "SrcType := USInt" } EQ_Contact(in1 := "dbTags_master_Fal_1"."step", in2 := 24)
      Contact( "dbTags_master_Fal_1".modbusMaster.done )
      wire#w1
      { S7_GenerateENO := "TRUE" } Move(in := "dbMasterData".ID26_Inver_OverVolts_415050_Fal, out1 => "dbModbusRTU_Reg".received26_Inver_OverVolts_415050)
      R_Coil( "dbTags_master_Fal_1".modbusMaster.req )
   END_RUNG
   RUNG wire#w1
      { S7_GenerateENO := "TRUE" } Move(in := 25, out1 => "dbTags_master_Fal_1"."step")
   END_RUNG
   // the same network as SCL:
   // ENO of a box is taken as its EN; it also drops when the box reports an error
   IF ("dbTags_master_Fal_1"."step" = 24) AND "dbTags_master_Fal_1".modbusMaster.done THEN
       "dbModbusRTU_Reg".received26_Inver_OverVolts_415050 := "dbMasterData".ID26_Inver_OverVolts_415050_Fal;
       "dbTags_master_Fal_1".modbusMaster.req := FALSE;
       "dbTags_master_Fal_1"."step" := 25;
   END_IF;
END_REGION

REGION Network 48: Przekazanie informacji o błędzie
   // Numer kroku i wartość błędu
   RUNG wire#powerrail
      I_Contact( "FirstScan" )
      Contact( "setErrorModbsmasterFal" )
      P_Trig( "memRisSteperror_Fal" )
      wire#w1
      Move(in := "dbTags_master_Fal_1"."step", out1 => "memStep_errorFal")
   END_RUNG
   RUNG wire#w1
      { S7_GenerateENO := "TRUE" } Move(in := "dbTags_master_Fal_1".modbusMaster.errorStatus, out1 => "db10datablock".RTU_Fal_1errorStatus)
   END_RUNG
   RUNG wire#w1
      R_Coil( "dbTags_master_Fal_1".modbusMaster.req )
   END_RUNG
   // the same network as SCL:
   #_w1 := NOT "FirstScan" AND "setErrorModbsmasterFal";
   #_w2 := #_w1 AND NOT "memRisSteperror_Fal";   // rising edge
   "memRisSteperror_Fal" := #_w1;
   IF #_w2 THEN
       "memStep_errorFal" := "dbTags_master_Fal_1"."step";
       "db10datablock".RTU_Fal_1errorStatus := "dbTags_master_Fal_1".modbusMaster.errorStatus;
       "dbTags_master_Fal_1".modbusMaster.req := FALSE;
   END_IF;
END_REGION

REGION Network 49: Obsługa błędów Modbaus
   // Inicjacja pętli modbus dla następnego urządzenia
   // Ustawienie kroku pętli na stan awaria [27]
   // Uwolnienie linni modbus
   RUNG wire#powerrail
      I_Contact( "FirstScan" )
      { S7_Templates := "SrcType := Word" } NE_Contact(in1 := "dbTags_master_Fal_1".modbusMaster.errorStatus, in2 := 0)
      Contact( "setErrorModbsmasterFal" )
      P_Trig( "memRisErrorModbusmaster" )
      wire#w1
      I_Contact( "AlwaysTRUE" )
      { S7_GenerateENO := "TRUE" } Move(in := 1, out1 => "dbTags_master_ABB_1"."step")
   END_RUNG
   RUNG wire#w1
      { S7_GenerateENO := "TRUE" } Move(in := 27, out1 => "dbTags_master_Fal_1"."step")
   END_RUNG
   RUNG wire#w1
      R_Coil( "dbTags_master_Fal_1".modbusMaster.req )
   END_RUNG
   // the same network as SCL:
   #_w1 := NOT "FirstScan" AND ("dbTags_master_Fal_1".modbusMaster.errorStatus <> 0) AND "setErrorModbsmasterFal";
   #_w2 := #_w1 AND NOT "memRisErrorModbusmaster";   // rising edge
   "memRisErrorModbusmaster" := #_w1;
   IF #_w2 AND NOT "AlwaysTRUE" THEN "dbTags_master_ABB_1"."step" := 1; END_IF;
   IF #_w2 THEN
       "dbTags_master_Fal_1"."step" := 27;
       "dbTags_master_Fal_1".modbusMaster.req := FALSE;
   END_IF;
END_REGION

REGION Network 50: Satart Loop MP04_1
   RUNG wire#powerrail
      { S7_Templates := "SrcType := USInt" } EQ_Contact(in1 := "dbTags_master_Fal_1"."step", in2 := 25)
      wire#w1
      P_Trig( "memRisModbusmaster_Loop3" )
      { S7_GenerateENO := "TRUE" } Move(in := 1, out1 => "dbTags_master_ABB_1"."step")
   END_RUNG
   RUNG wire#w1
      R_Coil( "setErrorModbsmasterABB_1" )
   END_RUNG
   // the same network as SCL:
   #_w1 := "dbTags_master_Fal_1"."step" = 25;
   #_w2 := #_w1 AND NOT "memRisModbusmaster_Loop3";   // rising edge
   "memRisModbusmaster_Loop3" := #_w1;
   IF #_w2 THEN "dbTags_master_ABB_1"."step" := 1; END_IF;
   IF #_w1 THEN "setErrorModbsmasterABB_1" := FALSE; END_IF;
END_REGION

REGION Network 52: Reset error mdbus staus
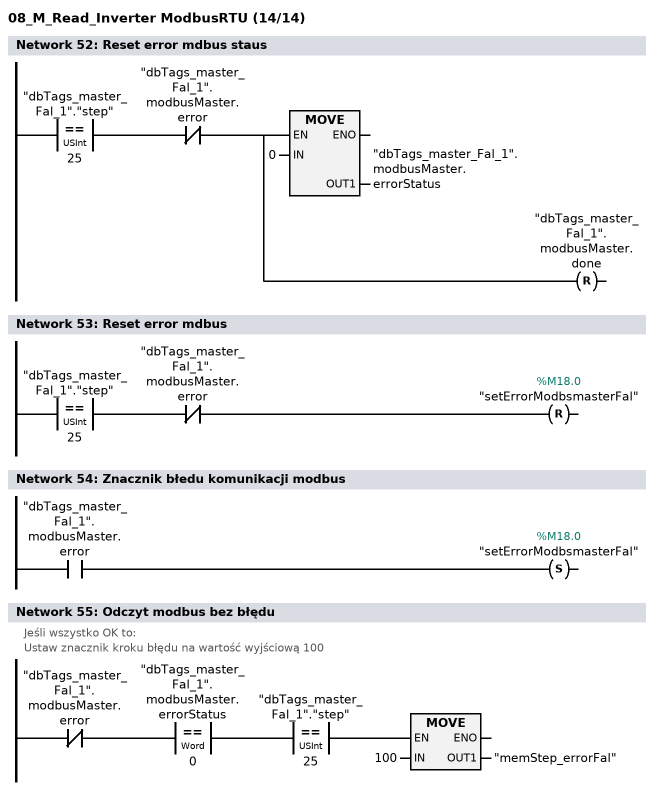
   RUNG wire#powerrail
      { S7_Templates := "SrcType := USInt" } EQ_Contact(in1 := "dbTags_master_Fal_1"."step", in2 := 25)
      I_Contact( "dbTags_master_Fal_1".modbusMaster.error )
      wire#w1
      { S7_GenerateENO := "TRUE" } Move(in := 0, out1 => "dbTags_master_Fal_1".modbusMaster.errorStatus)
   END_RUNG
   RUNG wire#w1
      R_Coil( "dbTags_master_Fal_1".modbusMaster.done )
   END_RUNG
   // the same network as SCL:
   IF ("dbTags_master_Fal_1"."step" = 25) AND NOT "dbTags_master_Fal_1".modbusMaster.error THEN
       "dbTags_master_Fal_1".modbusMaster.errorStatus := 0;
       "dbTags_master_Fal_1".modbusMaster.done := FALSE;
   END_IF;
END_REGION

REGION Network 53: Reset error mdbus
   RUNG wire#powerrail
      { S7_Templates := "SrcType := USInt" } EQ_Contact(in1 := "dbTags_master_Fal_1"."step", in2 := 25)
      I_Contact( "dbTags_master_Fal_1".modbusMaster.error )
      R_Coil( "setErrorModbsmasterFal" )
   END_RUNG
   // the same network as SCL:
   IF ("dbTags_master_Fal_1"."step" = 25) AND NOT "dbTags_master_Fal_1".modbusMaster.error THEN
       "setErrorModbsmasterFal" := FALSE;
   END_IF;
END_REGION

REGION Network 54: Znacznik błedu komunikacji modbus
   RUNG wire#powerrail
      Contact( "dbTags_master_Fal_1".modbusMaster.error )
      S_Coil( "setErrorModbsmasterFal" )
   END_RUNG
   // the same network as SCL:
   IF "dbTags_master_Fal_1".modbusMaster.error THEN "setErrorModbsmasterFal" := TRUE; END_IF;
END_REGION

REGION Network 55: Odczyt modbus bez błędu
   // Jeśli wszystko OK to:
   // Ustaw znacznik kroku błędu na wartość wyjściową 100
   RUNG wire#powerrail
      I_Contact( "dbTags_master_Fal_1".modbusMaster.error )
      { S7_Templates := "SrcType := Word" } EQ_Contact(in1 := "dbTags_master_Fal_1".modbusMaster.errorStatus, in2 := 0)
      { S7_Templates := "SrcType := USInt" } EQ_Contact(in1 := "dbTags_master_Fal_1"."step", in2 := 25)
      Move(in := 100, out1 => "memStep_errorFal")
   END_RUNG
   // the same network as SCL:
   IF NOT "dbTags_master_Fal_1".modbusMaster.error AND ("dbTags_master_Fal_1".modbusMaster.errorStatus = 0) AND ("dbTags_master_Fal_1"."step" = 25) THEN
       "memStep_errorFal" := 100;
   END_IF;
END_REGION
END_FUNCTION

FUNCTION "08_M_Read_MPP04_1_ModbusRTU" : Void   // FC23, LAD
TITLE = Read data from SC100
{ S7_Optimized_Access := 'TRUE' }
AUTHOR : rtecmer
VERSION : 0.1
// Czytanie z ABB 
// Obsługa protokołu Master Modbus RTU.  Odczyt pomiarów  przepływomierza ABB
// stored: AutoNumber true, IsIECCheckEnabled false, SetENOAutomatically false, UDAEnableTagReadback false
   VAR_TEMP   // added for the SCL form of the ladder/FBD networks
      _w1 : Bool;
      _w2 : Bool;
   END_VAR
BEGIN

REGION Network 1
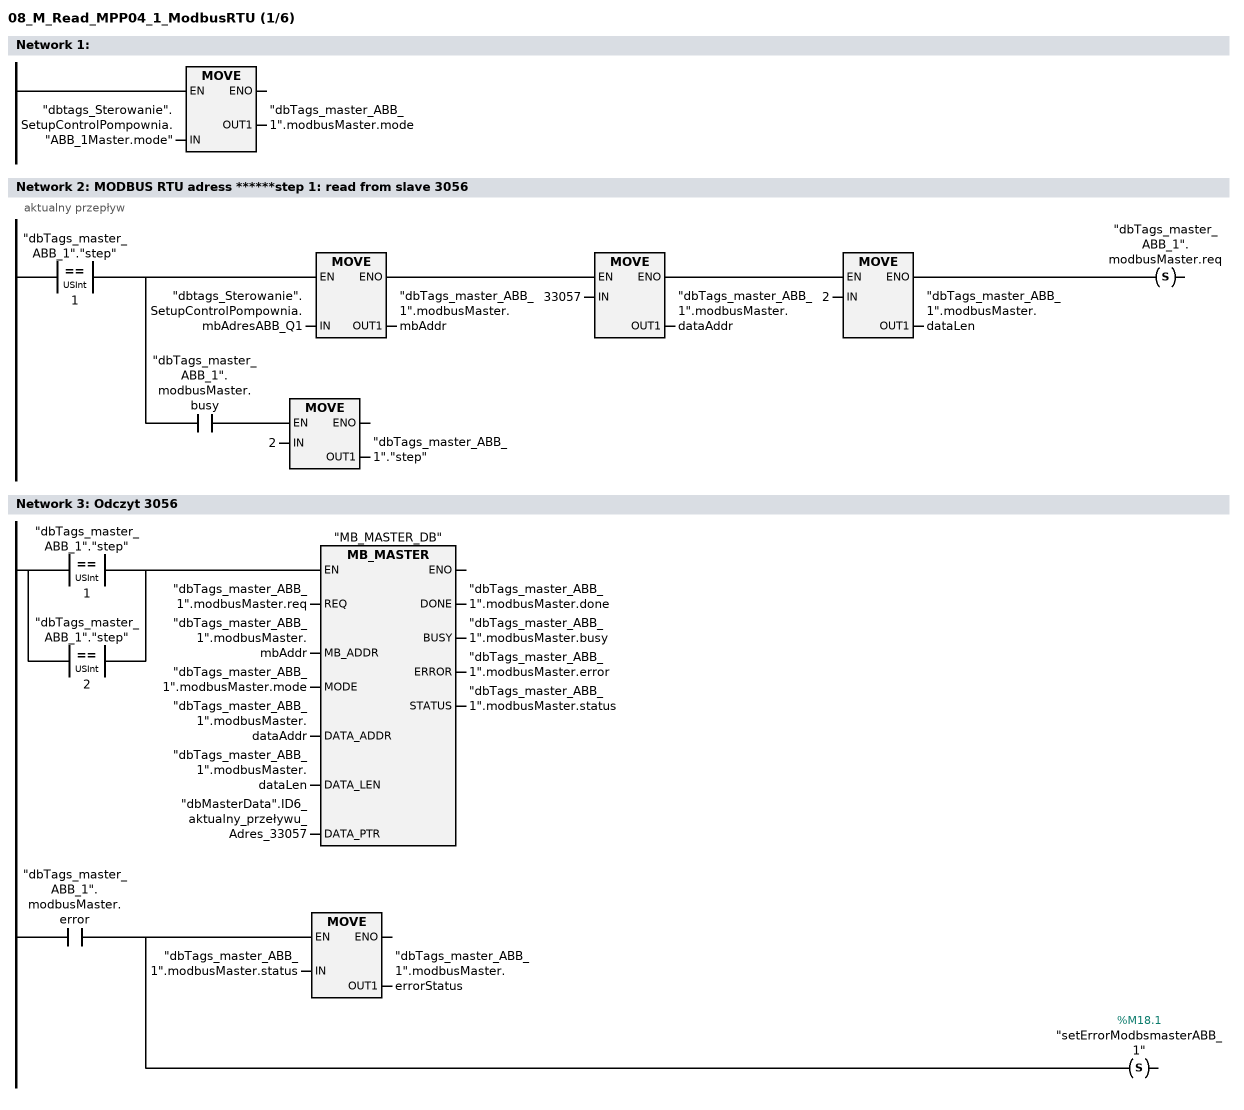
   RUNG wire#powerrail
      { S7_GenerateENO := "TRUE" } Move(in := "dbtags_Sterowanie".SetupControlPompownia."ABB_1Master.mode", out1 => "dbTags_master_ABB_1".modbusMaster.mode)
   END_RUNG
   // the same network as SCL:
   "dbTags_master_ABB_1".modbusMaster.mode := "dbtags_Sterowanie".SetupControlPompownia."ABB_1Master.mode";
END_REGION

REGION Network 2: MODBUS RTU adress ******step 1: read from slave 3056
   // aktualny przepływ
   RUNG wire#powerrail
      { S7_Templates := "SrcType := USInt" } EQ_Contact(in1 := "dbTags_master_ABB_1"."step", in2 := 1)
      wire#w1
      Move(in := "dbtags_Sterowanie".SetupControlPompownia.mbAdresABB_Q1, out1 => "dbTags_master_ABB_1".modbusMaster.mbAddr)
      { S7_GenerateENO := "TRUE" } Move(in := 33057, out1 => "dbTags_master_ABB_1".modbusMaster.dataAddr)
      Move(in := 2, out1 => "dbTags_master_ABB_1".modbusMaster.dataLen)
      S_Coil( "dbTags_master_ABB_1".modbusMaster.req )
   END_RUNG
   RUNG wire#w1
      Contact( "dbTags_master_ABB_1".modbusMaster.busy )
      { S7_GenerateENO := "TRUE" } Move(in := 2, out1 => "dbTags_master_ABB_1"."step")
   END_RUNG
   // the same network as SCL:
   // ENO of a box is taken as its EN; it also drops when the box reports an error
   #_w1 := "dbTags_master_ABB_1"."step" = 1;
   IF #_w1 THEN
       "dbTags_master_ABB_1".modbusMaster.mbAddr := "dbtags_Sterowanie".SetupControlPompownia.mbAdresABB_Q1;
       "dbTags_master_ABB_1".modbusMaster.dataAddr := 33057;
       "dbTags_master_ABB_1".modbusMaster.dataLen := 2;
       "dbTags_master_ABB_1".modbusMaster.req := TRUE;
   END_IF;
   IF #_w1 AND "dbTags_master_ABB_1".modbusMaster.busy THEN "dbTags_master_ABB_1"."step" := 2; END_IF;
END_REGION

REGION Network 3: Odczyt 3056
   RUNG wire#powerrail
      { S7_Templates := "SrcType := USInt" } EQ_Contact(in1 := "dbTags_master_ABB_1"."step", in2 := 1)
      wire#w1
      "MB_MASTER_DB".MB_MASTER(REQ := "dbTags_master_ABB_1".modbusMaster.req, MB_ADDR := "dbTags_master_ABB_1".modbusMaster.mbAddr, MODE := "dbTags_master_ABB_1".modbusMaster.mode, DATA_ADDR := "dbTags_master_ABB_1".modbusMaster.dataAddr, DATA_LEN := "dbTags_master_ABB_1".modbusMaster.dataLen, DATA_PTR := "dbMasterData".ID6_aktualny_przeływu_Adres_33057, DONE => "dbTags_master_ABB_1".modbusMaster.done, BUSY => "dbTags_master_ABB_1".modbusMaster.busy, ERROR => "dbTags_master_ABB_1".modbusMaster.error, STATUS => "dbTags_master_ABB_1".modbusMaster.status)
   END_RUNG
   RUNG wire#powerrail
      { S7_Templates := "SrcType := USInt" } EQ_Contact(in1 := "dbTags_master_ABB_1"."step", in2 := 2)
   END_RUNG wire#w1
   RUNG wire#powerrail
      Contact( "dbTags_master_ABB_1".modbusMaster.error )
      wire#w2
      { S7_GenerateENO := "TRUE" } Move(in := "dbTags_master_ABB_1".modbusMaster.status, out1 => "dbTags_master_ABB_1".modbusMaster.errorStatus)
   END_RUNG
   RUNG wire#w2
      S_Coil( "setErrorModbsmasterABB_1" )
   END_RUNG
   // the same network as SCL:
   IF ("dbTags_master_ABB_1"."step" = 1) OR ("dbTags_master_ABB_1"."step" = 2) THEN
       "MB_MASTER_DB"(REQ := "dbTags_master_ABB_1".modbusMaster.req,   // MB_MASTER
                      MB_ADDR := "dbTags_master_ABB_1".modbusMaster.mbAddr,
                      MODE := "dbTags_master_ABB_1".modbusMaster.mode,
                      DATA_ADDR := "dbTags_master_ABB_1".modbusMaster.dataAddr,
                      DATA_LEN := "dbTags_master_ABB_1".modbusMaster.dataLen,
                      DATA_PTR := "dbMasterData".ID6_aktualny_przeływu_Adres_33057,
                      DONE => "dbTags_master_ABB_1".modbusMaster.done,
                      BUSY => "dbTags_master_ABB_1".modbusMaster.busy,
                      ERROR => "dbTags_master_ABB_1".modbusMaster.error,
                      STATUS => "dbTags_master_ABB_1".modbusMaster.status);
   END_IF;
   IF "dbTags_master_ABB_1".modbusMaster.error THEN
       "dbTags_master_ABB_1".modbusMaster.errorStatus := "dbTags_master_ABB_1".modbusMaster.status;
       "setErrorModbsmasterABB_1" := TRUE;
   END_IF;
END_REGION

REGION Network 4: step 2: save received data 3056
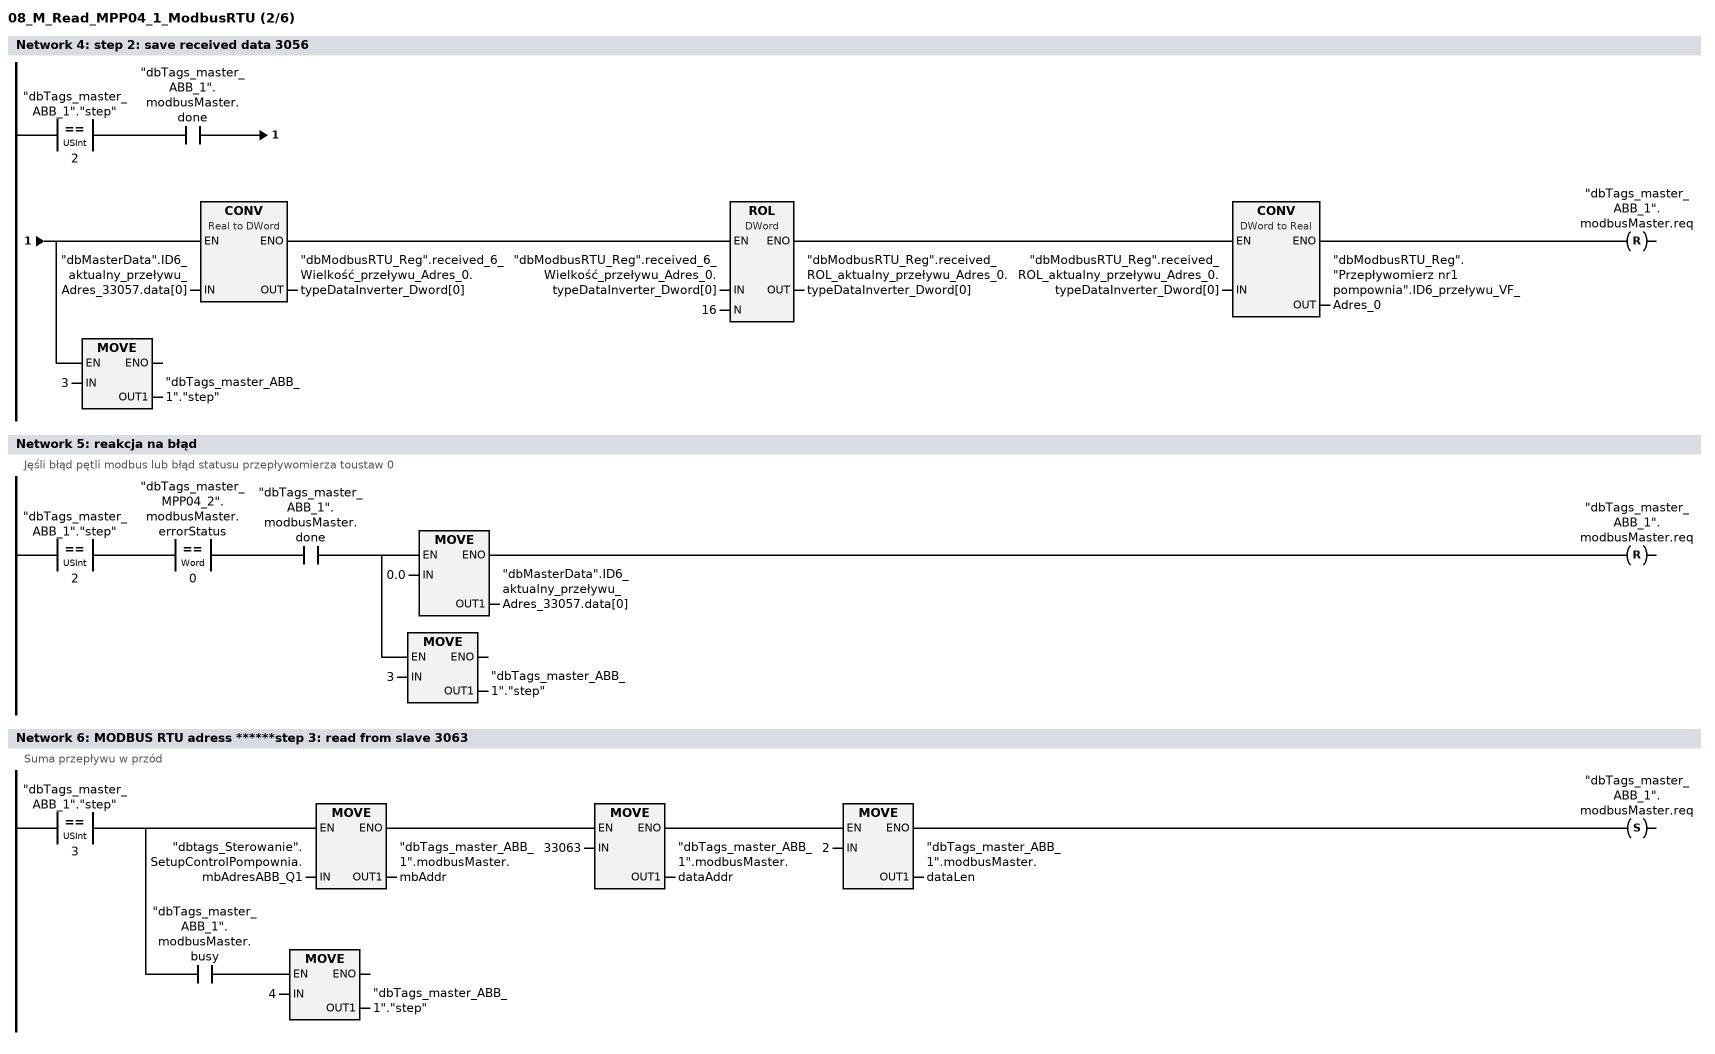
   IF ("dbTags_master_ABB_1"."step" = 2) AND "dbTags_master_ABB_1".modbusMaster.done THEN
       "dbModbusRTU_Reg".received_6_Wielkość_przeływu_Adres_0.typeDataInverter_Dword[0] := REAL_TO_DWORD("dbMasterData".ID6_aktualny_przeływu_Adres_33057.data[0]);
       "dbModbusRTU_Reg".received_ROL_aktualny_przeływu_Adres_0.typeDataInverter_Dword[0] := ROL(IN := "dbModbusRTU_Reg".received_6_Wielkość_przeływu_Adres_0.typeDataInverter_Dword[0], N := 16);
       "dbModbusRTU_Reg"."Przepływomierz nr1 pompownia".ID6_przeływu_VF_Adres_0 := DWORD_TO_REAL("dbModbusRTU_Reg".received_ROL_aktualny_przeływu_Adres_0.typeDataInverter_Dword[0]);
       "dbTags_master_ABB_1".modbusMaster.req := FALSE;
       "dbTags_master_ABB_1"."step" := 3;
   END_IF;
END_REGION

REGION Network 5: reakcja na błąd
   // Jęśli błąd pętli modbus lub błąd statusu przepływomierza toustaw 0
   RUNG wire#powerrail
      { S7_Templates := "SrcType := USInt" } EQ_Contact(in1 := "dbTags_master_ABB_1"."step", in2 := 2)
      { S7_Templates := "SrcType := Word" } EQ_Contact(in1 := "dbTags_master_MPP04_2".modbusMaster.errorStatus, in2 := 0)
      Contact( "dbTags_master_ABB_1".modbusMaster.done )
      wire#w1
      { S7_GenerateENO := "TRUE" } Move(in := 0.0, out1 => "dbMasterData".ID6_aktualny_przeływu_Adres_33057.data[0])
      R_Coil( "dbTags_master_ABB_1".modbusMaster.req )
   END_RUNG
   RUNG wire#w1
      { S7_GenerateENO := "TRUE" } Move(in := 3, out1 => "dbTags_master_ABB_1"."step")
   END_RUNG
   // the same network as SCL:
   // ENO of a box is taken as its EN; it also drops when the box reports an error
   IF ("dbTags_master_ABB_1"."step" = 2) AND ("dbTags_master_MPP04_2".modbusMaster.errorStatus = 0) AND "dbTags_master_ABB_1".modbusMaster.done THEN
       "dbMasterData".ID6_aktualny_przeływu_Adres_33057.data[0] := 0.0;
       "dbTags_master_ABB_1".modbusMaster.req := FALSE;
       "dbTags_master_ABB_1"."step" := 3;
   END_IF;
END_REGION

REGION Network 6: MODBUS RTU adress ******step 3: read from slave 3063
   // Suma przepływu w przód
   RUNG wire#powerrail
      { S7_Templates := "SrcType := USInt" } EQ_Contact(in1 := "dbTags_master_ABB_1"."step", in2 := 3)
      wire#w1
      Move(in := "dbtags_Sterowanie".SetupControlPompownia.mbAdresABB_Q1, out1 => "dbTags_master_ABB_1".modbusMaster.mbAddr)
      { S7_GenerateENO := "TRUE" } Move(in := 33063, out1 => "dbTags_master_ABB_1".modbusMaster.dataAddr)
      Move(in := 2, out1 => "dbTags_master_ABB_1".modbusMaster.dataLen)
      S_Coil( "dbTags_master_ABB_1".modbusMaster.req )
   END_RUNG
   RUNG wire#w1
      Contact( "dbTags_master_ABB_1".modbusMaster.busy )
      { S7_GenerateENO := "TRUE" } Move(in := 4, out1 => "dbTags_master_ABB_1"."step")
   END_RUNG
   // the same network as SCL:
   // ENO of a box is taken as its EN; it also drops when the box reports an error
   #_w1 := "dbTags_master_ABB_1"."step" = 3;
   IF #_w1 THEN
       "dbTags_master_ABB_1".modbusMaster.mbAddr := "dbtags_Sterowanie".SetupControlPompownia.mbAdresABB_Q1;
       "dbTags_master_ABB_1".modbusMaster.dataAddr := 33063;
       "dbTags_master_ABB_1".modbusMaster.dataLen := 2;
       "dbTags_master_ABB_1".modbusMaster.req := TRUE;
   END_IF;
   IF #_w1 AND "dbTags_master_ABB_1".modbusMaster.busy THEN "dbTags_master_ABB_1"."step" := 4; END_IF;
END_REGION

REGION Network 7: Odczyt 3062
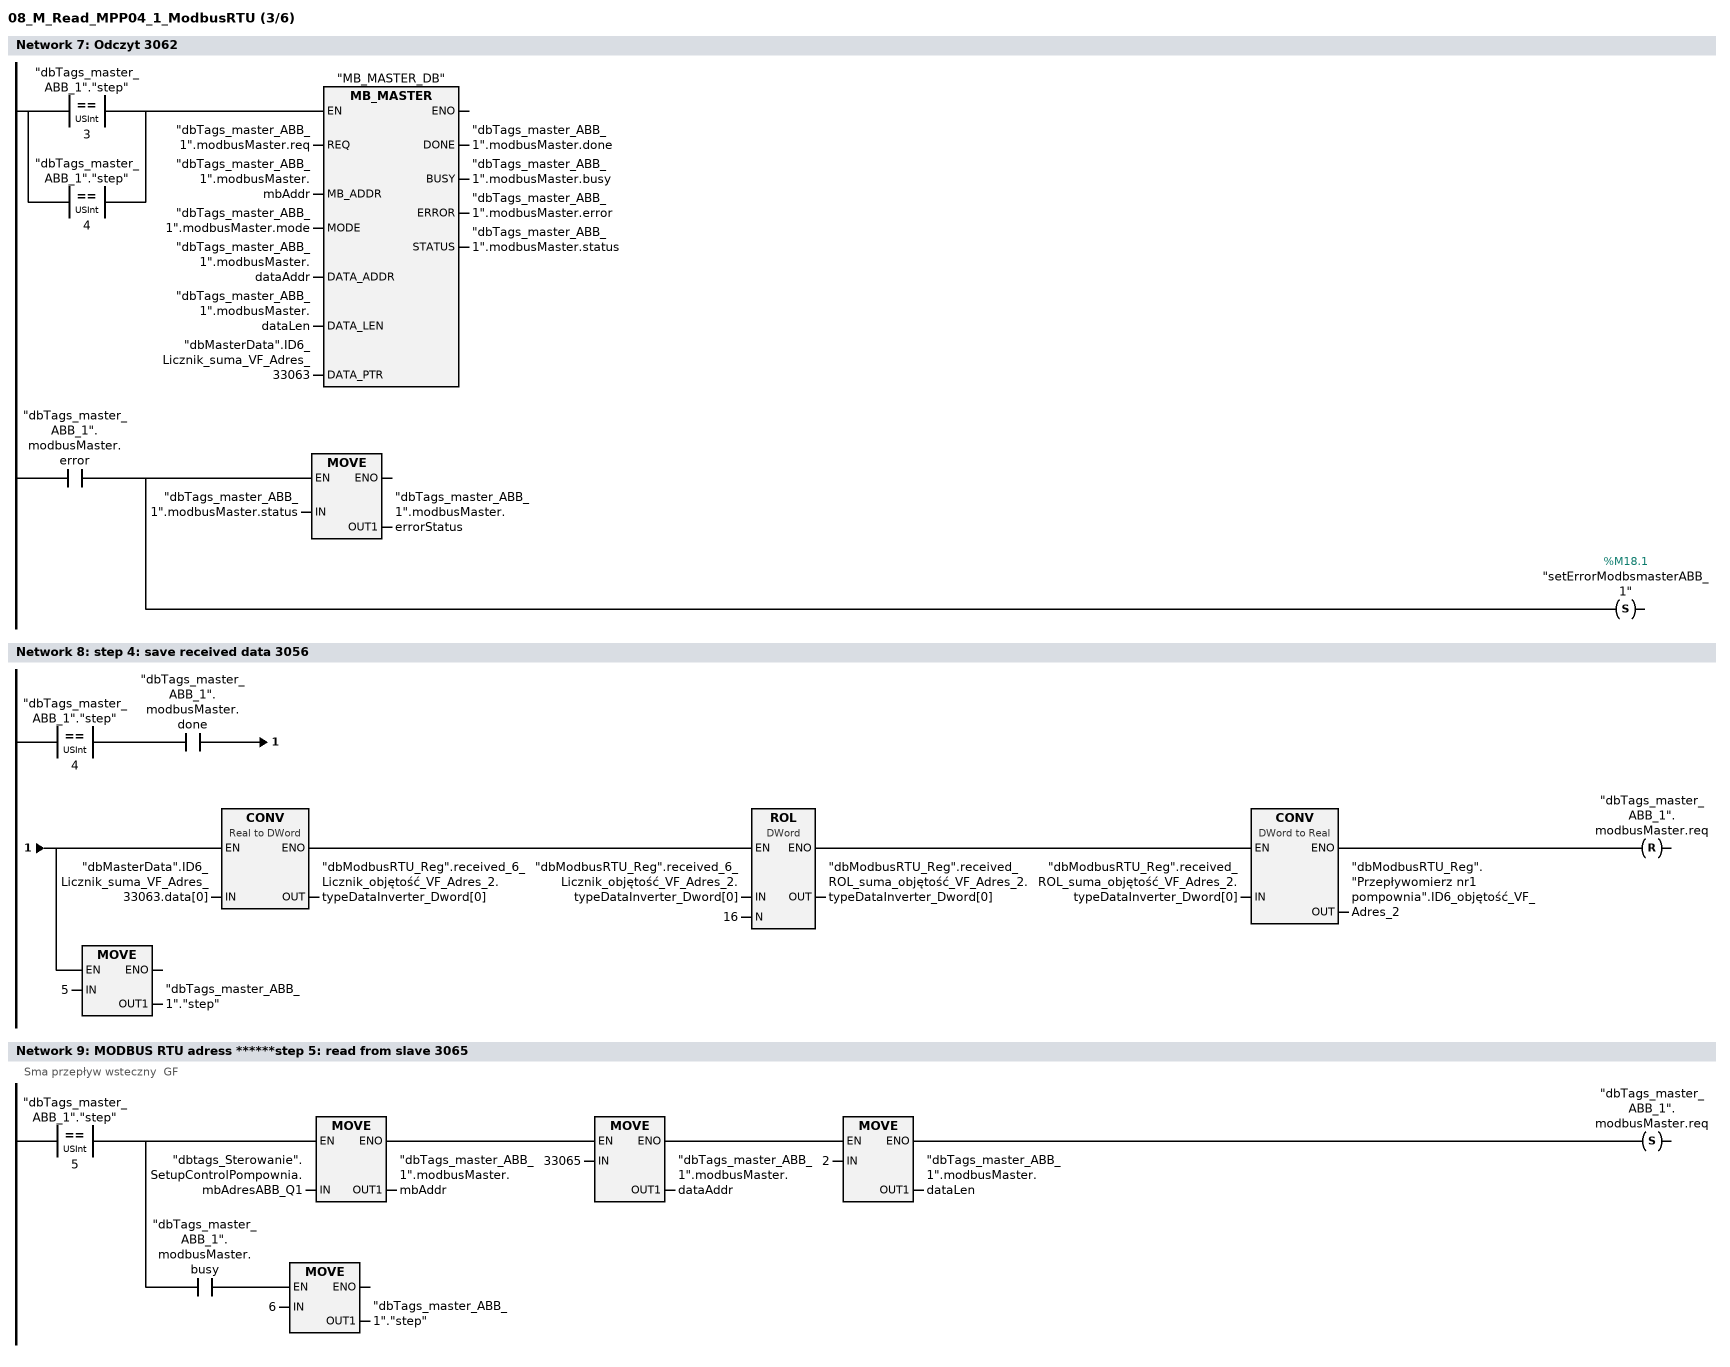
   RUNG wire#powerrail
      { S7_Templates := "SrcType := USInt" } EQ_Contact(in1 := "dbTags_master_ABB_1"."step", in2 := 3)
      wire#w1
      "MB_MASTER_DB".MB_MASTER(REQ := "dbTags_master_ABB_1".modbusMaster.req, MB_ADDR := "dbTags_master_ABB_1".modbusMaster.mbAddr, MODE := "dbTags_master_ABB_1".modbusMaster.mode, DATA_ADDR := "dbTags_master_ABB_1".modbusMaster.dataAddr, DATA_LEN := "dbTags_master_ABB_1".modbusMaster.dataLen, DATA_PTR := "dbMasterData".ID6_Licznik_suma_VF_Adres_33063, DONE => "dbTags_master_ABB_1".modbusMaster.done, BUSY => "dbTags_master_ABB_1".modbusMaster.busy, ERROR => "dbTags_master_ABB_1".modbusMaster.error, STATUS => "dbTags_master_ABB_1".modbusMaster.status)
   END_RUNG
   RUNG wire#powerrail
      { S7_Templates := "SrcType := USInt" } EQ_Contact(in1 := "dbTags_master_ABB_1"."step", in2 := 4)
   END_RUNG wire#w1
   RUNG wire#powerrail
      Contact( "dbTags_master_ABB_1".modbusMaster.error )
      wire#w2
      { S7_GenerateENO := "TRUE" } Move(in := "dbTags_master_ABB_1".modbusMaster.status, out1 => "dbTags_master_ABB_1".modbusMaster.errorStatus)
   END_RUNG
   RUNG wire#w2
      S_Coil( "setErrorModbsmasterABB_1" )
   END_RUNG
   // the same network as SCL:
   IF ("dbTags_master_ABB_1"."step" = 3) OR ("dbTags_master_ABB_1"."step" = 4) THEN
       "MB_MASTER_DB"(REQ := "dbTags_master_ABB_1".modbusMaster.req,   // MB_MASTER
                      MB_ADDR := "dbTags_master_ABB_1".modbusMaster.mbAddr,
                      MODE := "dbTags_master_ABB_1".modbusMaster.mode,
                      DATA_ADDR := "dbTags_master_ABB_1".modbusMaster.dataAddr,
                      DATA_LEN := "dbTags_master_ABB_1".modbusMaster.dataLen,
                      DATA_PTR := "dbMasterData".ID6_Licznik_suma_VF_Adres_33063,
                      DONE => "dbTags_master_ABB_1".modbusMaster.done,
                      BUSY => "dbTags_master_ABB_1".modbusMaster.busy,
                      ERROR => "dbTags_master_ABB_1".modbusMaster.error,
                      STATUS => "dbTags_master_ABB_1".modbusMaster.status);
   END_IF;
   IF "dbTags_master_ABB_1".modbusMaster.error THEN
       "dbTags_master_ABB_1".modbusMaster.errorStatus := "dbTags_master_ABB_1".modbusMaster.status;
       "setErrorModbsmasterABB_1" := TRUE;
   END_IF;
END_REGION

REGION Network 8: step 4: save received data 3056
   IF ("dbTags_master_ABB_1"."step" = 4) AND "dbTags_master_ABB_1".modbusMaster.done THEN
       "dbModbusRTU_Reg".received_6_Licznik_objętość_VF_Adres_2.typeDataInverter_Dword[0] := REAL_TO_DWORD("dbMasterData".ID6_Licznik_suma_VF_Adres_33063.data[0]);
       "dbModbusRTU_Reg".received_ROL_suma_objętość_VF_Adres_2.typeDataInverter_Dword[0] := ROL(IN := "dbModbusRTU_Reg".received_6_Licznik_objętość_VF_Adres_2.typeDataInverter_Dword[0], N := 16);
       "dbModbusRTU_Reg"."Przepływomierz nr1 pompownia".ID6_objętość_VF_Adres_2 := DWORD_TO_REAL("dbModbusRTU_Reg".received_ROL_suma_objętość_VF_Adres_2.typeDataInverter_Dword[0]);
       "dbTags_master_ABB_1".modbusMaster.req := FALSE;
       "dbTags_master_ABB_1"."step" := 5;
   END_IF;
END_REGION

REGION Network 9: MODBUS RTU adress ******step 5: read from slave 3065
   // Sma przepływ wsteczny  GF
   RUNG wire#powerrail
      { S7_Templates := "SrcType := USInt" } EQ_Contact(in1 := "dbTags_master_ABB_1"."step", in2 := 5)
      wire#w1
      Move(in := "dbtags_Sterowanie".SetupControlPompownia.mbAdresABB_Q1, out1 => "dbTags_master_ABB_1".modbusMaster.mbAddr)
      { S7_GenerateENO := "TRUE" } Move(in := 33065, out1 => "dbTags_master_ABB_1".modbusMaster.dataAddr)
      Move(in := 2, out1 => "dbTags_master_ABB_1".modbusMaster.dataLen)
      S_Coil( "dbTags_master_ABB_1".modbusMaster.req )
   END_RUNG
   RUNG wire#w1
      Contact( "dbTags_master_ABB_1".modbusMaster.busy )
      { S7_GenerateENO := "TRUE" } Move(in := 6, out1 => "dbTags_master_ABB_1"."step")
   END_RUNG
   // the same network as SCL:
   // ENO of a box is taken as its EN; it also drops when the box reports an error
   #_w1 := "dbTags_master_ABB_1"."step" = 5;
   IF #_w1 THEN
       "dbTags_master_ABB_1".modbusMaster.mbAddr := "dbtags_Sterowanie".SetupControlPompownia.mbAdresABB_Q1;
       "dbTags_master_ABB_1".modbusMaster.dataAddr := 33065;
       "dbTags_master_ABB_1".modbusMaster.dataLen := 2;
       "dbTags_master_ABB_1".modbusMaster.req := TRUE;
   END_IF;
   IF #_w1 AND "dbTags_master_ABB_1".modbusMaster.busy THEN "dbTags_master_ABB_1"."step" := 6; END_IF;
END_REGION

REGION Network 10: Odczyt 3065
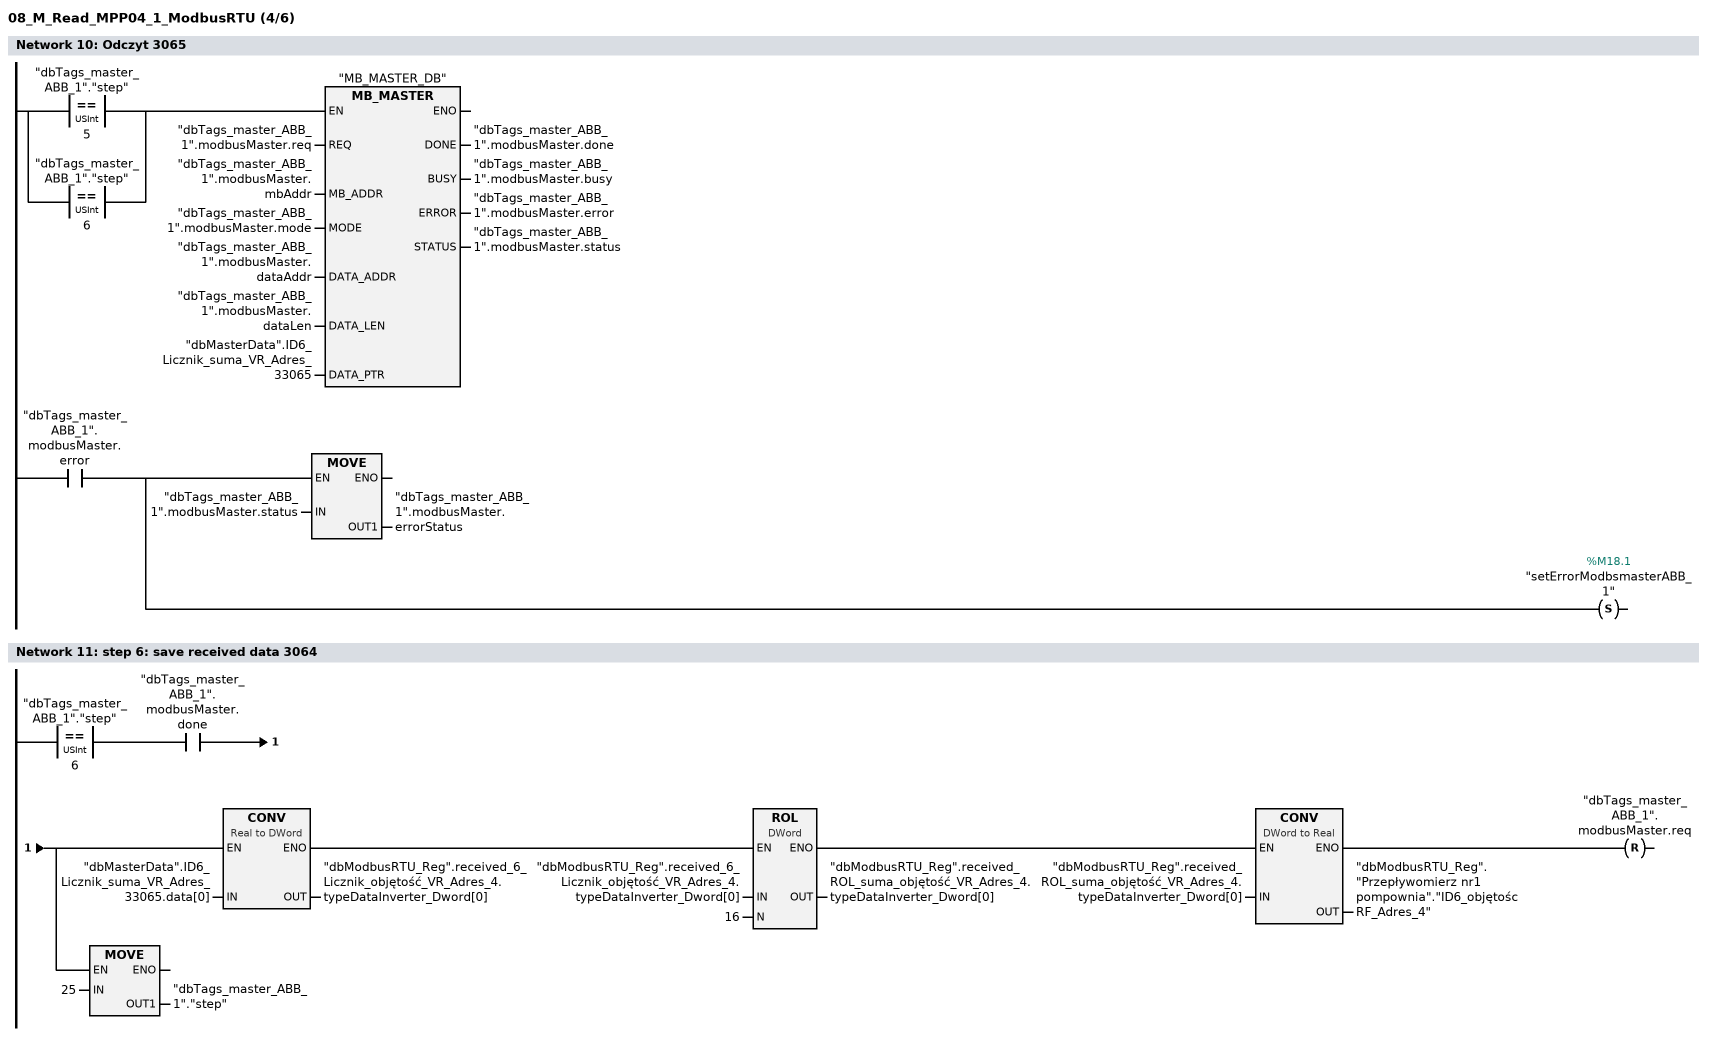
   RUNG wire#powerrail
      { S7_Templates := "SrcType := USInt" } EQ_Contact(in1 := "dbTags_master_ABB_1"."step", in2 := 5)
      wire#w1
      "MB_MASTER_DB".MB_MASTER(REQ := "dbTags_master_ABB_1".modbusMaster.req, MB_ADDR := "dbTags_master_ABB_1".modbusMaster.mbAddr, MODE := "dbTags_master_ABB_1".modbusMaster.mode, DATA_ADDR := "dbTags_master_ABB_1".modbusMaster.dataAddr, DATA_LEN := "dbTags_master_ABB_1".modbusMaster.dataLen, DATA_PTR := "dbMasterData".ID6_Licznik_suma_VR_Adres_33065, DONE => "dbTags_master_ABB_1".modbusMaster.done, BUSY => "dbTags_master_ABB_1".modbusMaster.busy, ERROR => "dbTags_master_ABB_1".modbusMaster.error, STATUS => "dbTags_master_ABB_1".modbusMaster.status)
   END_RUNG
   RUNG wire#powerrail
      { S7_Templates := "SrcType := USInt" } EQ_Contact(in1 := "dbTags_master_ABB_1"."step", in2 := 6)
   END_RUNG wire#w1
   RUNG wire#powerrail
      Contact( "dbTags_master_ABB_1".modbusMaster.error )
      wire#w2
      { S7_GenerateENO := "TRUE" } Move(in := "dbTags_master_ABB_1".modbusMaster.status, out1 => "dbTags_master_ABB_1".modbusMaster.errorStatus)
   END_RUNG
   RUNG wire#w2
      S_Coil( "setErrorModbsmasterABB_1" )
   END_RUNG
   // the same network as SCL:
   IF ("dbTags_master_ABB_1"."step" = 5) OR ("dbTags_master_ABB_1"."step" = 6) THEN
       "MB_MASTER_DB"(REQ := "dbTags_master_ABB_1".modbusMaster.req,   // MB_MASTER
                      MB_ADDR := "dbTags_master_ABB_1".modbusMaster.mbAddr,
                      MODE := "dbTags_master_ABB_1".modbusMaster.mode,
                      DATA_ADDR := "dbTags_master_ABB_1".modbusMaster.dataAddr,
                      DATA_LEN := "dbTags_master_ABB_1".modbusMaster.dataLen,
                      DATA_PTR := "dbMasterData".ID6_Licznik_suma_VR_Adres_33065,
                      DONE => "dbTags_master_ABB_1".modbusMaster.done,
                      BUSY => "dbTags_master_ABB_1".modbusMaster.busy,
                      ERROR => "dbTags_master_ABB_1".modbusMaster.error,
                      STATUS => "dbTags_master_ABB_1".modbusMaster.status);
   END_IF;
   IF "dbTags_master_ABB_1".modbusMaster.error THEN
       "dbTags_master_ABB_1".modbusMaster.errorStatus := "dbTags_master_ABB_1".modbusMaster.status;
       "setErrorModbsmasterABB_1" := TRUE;
   END_IF;
END_REGION

REGION Network 11: step 6: save received data 3064
   IF ("dbTags_master_ABB_1"."step" = 6) AND "dbTags_master_ABB_1".modbusMaster.done THEN
       "dbModbusRTU_Reg".received_6_Licznik_objętość_VR_Adres_4.typeDataInverter_Dword[0] := REAL_TO_DWORD("dbMasterData".ID6_Licznik_suma_VR_Adres_33065.data[0]);
       "dbModbusRTU_Reg".received_ROL_suma_objętość_VR_Adres_4.typeDataInverter_Dword[0] := ROL(IN := "dbModbusRTU_Reg".received_6_Licznik_objętość_VR_Adres_4.typeDataInverter_Dword[0], N := 16);
       "dbModbusRTU_Reg"."Przepływomierz nr1 pompownia"."ID6_objętośc RF_Adres_4" := DWORD_TO_REAL("dbModbusRTU_Reg".received_ROL_suma_objętość_VR_Adres_4.typeDataInverter_Dword[0]);
       "dbTags_master_ABB_1".modbusMaster.req := FALSE;
       "dbTags_master_ABB_1"."step" := 25;
   END_IF;
END_REGION

REGION Network 12: Przekazanie informacji o błędzie
   // Numer kroku i wartość błędu
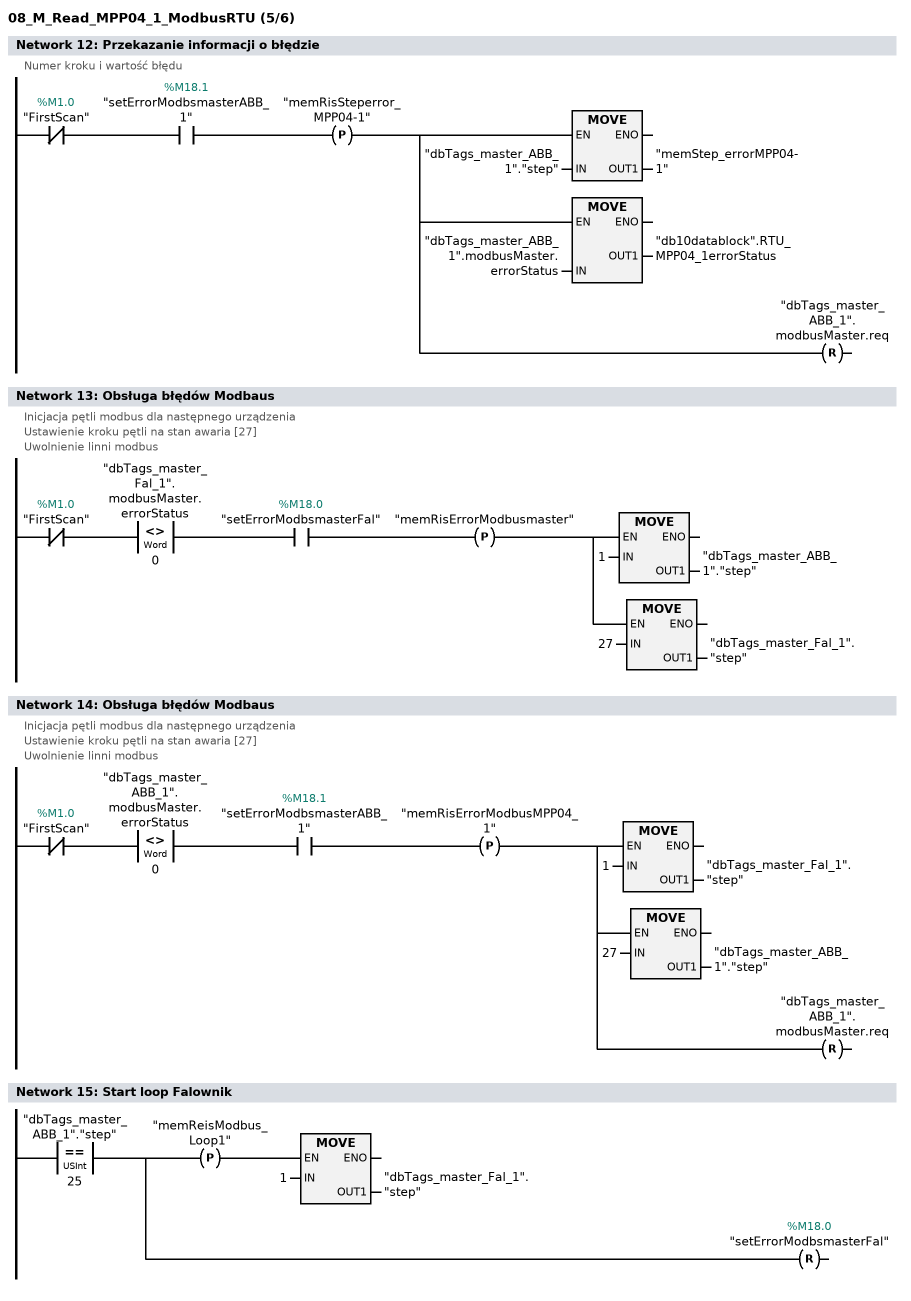
   RUNG wire#powerrail
      I_Contact( "FirstScan" )
      Contact( "setErrorModbsmasterABB_1" )
      P_Trig( "memRisSteperror_MPP04-1" )
      wire#w1
      Move(in := "dbTags_master_ABB_1"."step", out1 => "memStep_errorMPP04-1")
   END_RUNG
   RUNG wire#w1
      { S7_GenerateENO := "TRUE" } Move(in := "dbTags_master_ABB_1".modbusMaster.errorStatus, out1 => "db10datablock".RTU_MPP04_1errorStatus)
   END_RUNG
   RUNG wire#w1
      R_Coil( "dbTags_master_ABB_1".modbusMaster.req )
   END_RUNG
   // the same network as SCL:
   #_w1 := NOT "FirstScan" AND "setErrorModbsmasterABB_1";
   #_w2 := #_w1 AND NOT "memRisSteperror_MPP04-1";   // rising edge
   "memRisSteperror_MPP04-1" := #_w1;
   IF #_w2 THEN
       "memStep_errorMPP04-1" := "dbTags_master_ABB_1"."step";
       "db10datablock".RTU_MPP04_1errorStatus := "dbTags_master_ABB_1".modbusMaster.errorStatus;
       "dbTags_master_ABB_1".modbusMaster.req := FALSE;
   END_IF;
END_REGION

REGION Network 13: Obsługa błędów Modbaus
   // Inicjacja pętli modbus dla następnego urządzenia
   // Ustawienie kroku pętli na stan awaria [27]
   // Uwolnienie linni modbus
   RUNG wire#powerrail
      I_Contact( "FirstScan" )
      { S7_Templates := "SrcType := Word" } NE_Contact(in1 := "dbTags_master_Fal_1".modbusMaster.errorStatus, in2 := 0)
      Contact( "setErrorModbsmasterFal" )
      P_Trig( "memRisErrorModbusmaster" )
      wire#w1
      { S7_GenerateENO := "TRUE" } Move(in := 1, out1 => "dbTags_master_ABB_1"."step")
   END_RUNG
   RUNG wire#w1
      { S7_GenerateENO := "TRUE" } Move(in := 27, out1 => "dbTags_master_Fal_1"."step")
   END_RUNG
   // the same network as SCL:
   #_w1 := NOT "FirstScan" AND ("dbTags_master_Fal_1".modbusMaster.errorStatus <> 0) AND "setErrorModbsmasterFal";
   #_w2 := #_w1 AND NOT "memRisErrorModbusmaster";   // rising edge
   "memRisErrorModbusmaster" := #_w1;
   IF #_w2 THEN
       "dbTags_master_ABB_1"."step" := 1;
       "dbTags_master_Fal_1"."step" := 27;
   END_IF;
END_REGION

REGION Network 14: Obsługa błędów Modbaus
   // Inicjacja pętli modbus dla następnego urządzenia
   // Ustawienie kroku pętli na stan awaria [27]
   // Uwolnienie linni modbus
   RUNG wire#powerrail
      I_Contact( "FirstScan" )
      { S7_Templates := "SrcType := Word" } NE_Contact(in1 := "dbTags_master_ABB_1".modbusMaster.errorStatus, in2 := 0)
      Contact( "setErrorModbsmasterABB_1" )
      P_Trig( "memRisErrorModbusMPP04_1" )
      wire#w1
      { S7_GenerateENO := "TRUE" } Move(in := 1, out1 => "dbTags_master_Fal_1"."step")
   END_RUNG
   RUNG wire#w1
      { S7_GenerateENO := "TRUE" } Move(in := 27, out1 => "dbTags_master_ABB_1"."step")
   END_RUNG
   RUNG wire#w1
      R_Coil( "dbTags_master_ABB_1".modbusMaster.req )
   END_RUNG
   // the same network as SCL:
   #_w1 := NOT "FirstScan" AND ("dbTags_master_ABB_1".modbusMaster.errorStatus <> 0) AND "setErrorModbsmasterABB_1";
   #_w2 := #_w1 AND NOT "memRisErrorModbusMPP04_1";   // rising edge
   "memRisErrorModbusMPP04_1" := #_w1;
   IF #_w2 THEN
       "dbTags_master_Fal_1"."step" := 1;
       "dbTags_master_ABB_1"."step" := 27;
       "dbTags_master_ABB_1".modbusMaster.req := FALSE;
   END_IF;
END_REGION

REGION Network 15: Start loop Falownik
   RUNG wire#powerrail
      { S7_Templates := "SrcType := USInt" } EQ_Contact(in1 := "dbTags_master_ABB_1"."step", in2 := 25)
      wire#w1
      P_Trig( "memReisModbus_Loop1" )
      { S7_GenerateENO := "TRUE" } Move(in := 1, out1 => "dbTags_master_Fal_1"."step")
   END_RUNG
   RUNG wire#w1
      R_Coil( "setErrorModbsmasterFal" )
   END_RUNG
   // the same network as SCL:
   #_w1 := "dbTags_master_ABB_1"."step" = 25;
   #_w2 := #_w1 AND NOT "memReisModbus_Loop1";   // rising edge
   "memReisModbus_Loop1" := #_w1;
   IF #_w2 THEN "dbTags_master_Fal_1"."step" := 1; END_IF;
   IF #_w1 THEN "setErrorModbsmasterFal" := FALSE; END_IF;
END_REGION

REGION Network 16: Reset error mdbus staus
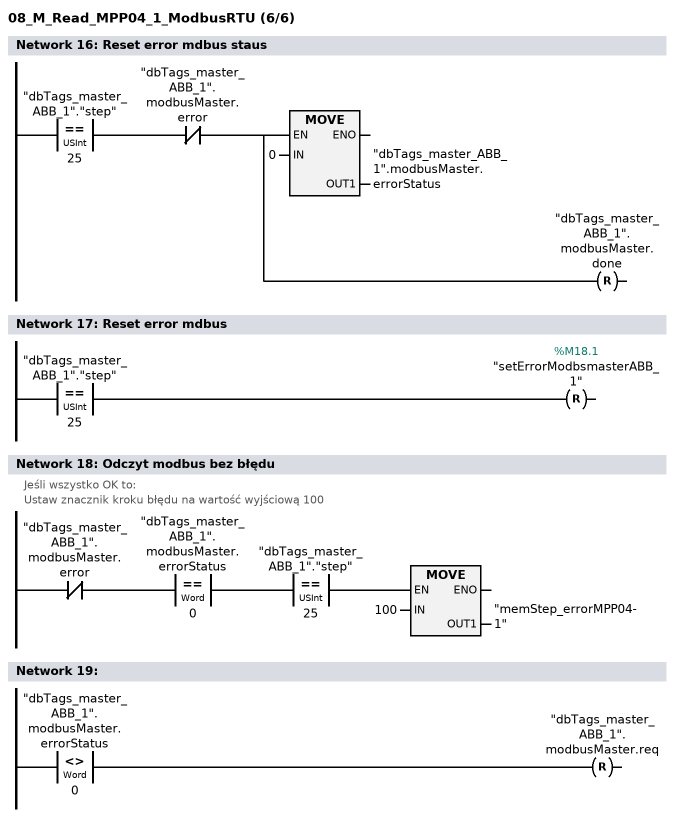
   RUNG wire#powerrail
      { S7_Templates := "SrcType := USInt" } EQ_Contact(in1 := "dbTags_master_ABB_1"."step", in2 := 25)
      I_Contact( "dbTags_master_ABB_1".modbusMaster.error )
      wire#w1
      { S7_GenerateENO := "TRUE" } Move(in := 0, out1 => "dbTags_master_ABB_1".modbusMaster.errorStatus)
   END_RUNG
   RUNG wire#w1
      R_Coil( "dbTags_master_ABB_1".modbusMaster.done )
   END_RUNG
   // the same network as SCL:
   IF ("dbTags_master_ABB_1"."step" = 25) AND NOT "dbTags_master_ABB_1".modbusMaster.error THEN
       "dbTags_master_ABB_1".modbusMaster.errorStatus := 0;
       "dbTags_master_ABB_1".modbusMaster.done := FALSE;
   END_IF;
END_REGION

REGION Network 17: Reset error mdbus
   RUNG wire#powerrail
      { S7_Templates := "SrcType := USInt" } EQ_Contact(in1 := "dbTags_master_ABB_1"."step", in2 := 25)
      R_Coil( "setErrorModbsmasterABB_1" )
   END_RUNG
   // the same network as SCL:
   IF "dbTags_master_ABB_1"."step" = 25 THEN "setErrorModbsmasterABB_1" := FALSE; END_IF;
END_REGION

REGION Network 18: Odczyt modbus bez błędu
   // Jeśli wszystko OK to:
   // Ustaw znacznik kroku błędu na wartość wyjściową 100
   RUNG wire#powerrail
      I_Contact( "dbTags_master_ABB_1".modbusMaster.error )
      { S7_Templates := "SrcType := Word" } EQ_Contact(in1 := "dbTags_master_ABB_1".modbusMaster.errorStatus, in2 := 0)
      { S7_Templates := "SrcType := USInt" } EQ_Contact(in1 := "dbTags_master_ABB_1"."step", in2 := 25)
      { S7_GenerateENO := "TRUE" } Move(in := 100, out1 => "memStep_errorMPP04-1")
   END_RUNG
   // the same network as SCL:
   IF NOT "dbTags_master_ABB_1".modbusMaster.error AND ("dbTags_master_ABB_1".modbusMaster.errorStatus = 0) AND ("dbTags_master_ABB_1"."step" = 25) THEN
       "memStep_errorMPP04-1" := 100;
   END_IF;
END_REGION

REGION Network 19
   RUNG wire#powerrail
      { S7_Templates := "SrcType := Word" } NE_Contact(in1 := "dbTags_master_ABB_1".modbusMaster.errorStatus, in2 := 0)
      R_Coil( "dbTags_master_ABB_1".modbusMaster.req )
   END_RUNG
   // the same network as SCL:
   IF "dbTags_master_ABB_1".modbusMaster.errorStatus <> 0 THEN
       "dbTags_master_ABB_1".modbusMaster.req := FALSE;
   END_IF;
END_REGION
END_FUNCTION

FUNCTION "09_W_Work counter block" : Void   // FC8, LAD
TITLE = Wywołanie funkcji liczników pracy
{ S7_Optimized_Access := 'TRUE' }
AUTHOR : RTecmer
VERSION : 0.1
// Funkcja wywołuje liczniki pracy napędów
// stored: AutoNumber true, IsIECCheckEnabled false, SetENOAutomatically false, UDAEnableTagReadback false
BEGIN

REGION Network 1: Pompa P1
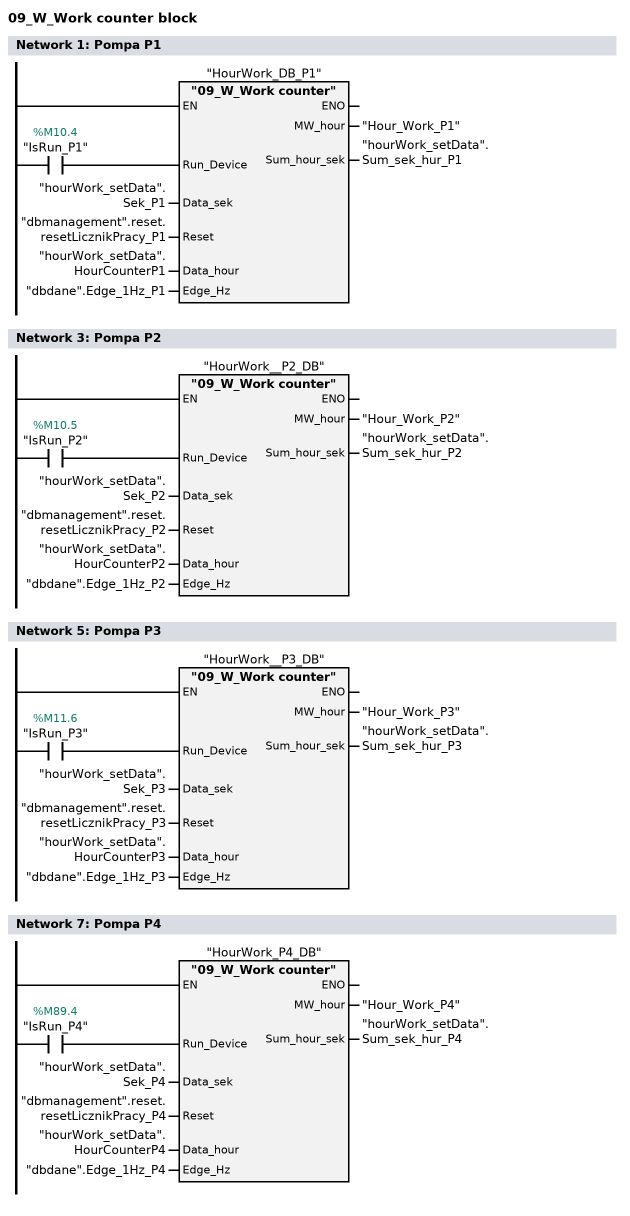
   RUNG wire#powerrail
      "HourWork_DB_P1"(Run_Device := wire#w1, Data_sek := "hourWork_setData".Sek_P1, Reset := "dbmanagement".reset.resetLicznikPracy_P1, Data_hour := "hourWork_setData".HourCounterP1, Edge_Hz := "dbdane".Edge_1Hz_P1, MW_hour => "Hour_Work_P1", Sum_hour_sek => "hourWork_setData".Sum_sek_hur_P1)
   END_RUNG
   RUNG wire#powerrail
      Contact( "IsRun_P1" )
   END_RUNG wire#w1
   // the same network as SCL:
   "HourWork_DB_P1"(Run_Device := "IsRun_P1",   // "09_W_Work counter"
                    Data_sek := "hourWork_setData".Sek_P1,
                    Reset := "dbmanagement".reset.resetLicznikPracy_P1,
                    Data_hour := "hourWork_setData".HourCounterP1,
                    Edge_Hz := "dbdane".Edge_1Hz_P1,
                    MW_hour => "Hour_Work_P1",
                    Sum_hour_sek => "hourWork_setData".Sum_sek_hur_P1);
END_REGION

REGION Network 2 (SCL)
   "db10datablock".HourCounterP1 := "hourWork_setData".HourCounterP1;
END_REGION

REGION Network 3: Pompa P2
   RUNG wire#powerrail
      "HourWork__P2_DB"(Run_Device := wire#w1, Data_sek := "hourWork_setData".Sek_P2, Reset := "dbmanagement".reset.resetLicznikPracy_P2, Data_hour := "hourWork_setData".HourCounterP2, Edge_Hz := "dbdane".Edge_1Hz_P2, MW_hour => "Hour_Work_P2", Sum_hour_sek => "hourWork_setData".Sum_sek_hur_P2)
   END_RUNG
   RUNG wire#powerrail
      Contact( "IsRun_P2" )
   END_RUNG wire#w1
   // the same network as SCL:
   "HourWork__P2_DB"(Run_Device := "IsRun_P2",   // "09_W_Work counter"
                     Data_sek := "hourWork_setData".Sek_P2,
                     Reset := "dbmanagement".reset.resetLicznikPracy_P2,
                     Data_hour := "hourWork_setData".HourCounterP2,
                     Edge_Hz := "dbdane".Edge_1Hz_P2,
                     MW_hour => "Hour_Work_P2",
                     Sum_hour_sek => "hourWork_setData".Sum_sek_hur_P2);
END_REGION

REGION Network 4 (SCL)
   "db10datablock".HourCounterP2 := "hourWork_setData".HourCounterP2;
END_REGION

REGION Network 5: Pompa P3
   RUNG wire#powerrail
      "HourWork__P3_DB"(Run_Device := wire#w1, Data_sek := "hourWork_setData".Sek_P3, Reset := "dbmanagement".reset.resetLicznikPracy_P3, Data_hour := "hourWork_setData".HourCounterP3, Edge_Hz := "dbdane".Edge_1Hz_P3, MW_hour => "Hour_Work_P3", Sum_hour_sek => "hourWork_setData".Sum_sek_hur_P3)
   END_RUNG
   RUNG wire#powerrail
      Contact( "IsRun_P3" )
   END_RUNG wire#w1
   // the same network as SCL:
   "HourWork__P3_DB"(Run_Device := "IsRun_P3",   // "09_W_Work counter"
                     Data_sek := "hourWork_setData".Sek_P3,
                     Reset := "dbmanagement".reset.resetLicznikPracy_P3,
                     Data_hour := "hourWork_setData".HourCounterP3,
                     Edge_Hz := "dbdane".Edge_1Hz_P3,
                     MW_hour => "Hour_Work_P3",
                     Sum_hour_sek => "hourWork_setData".Sum_sek_hur_P3);
END_REGION

REGION Network 6 (SCL)
   "db10datablock".HourCounterP3:= "hourWork_setData".HourCounterP3;
END_REGION

REGION Network 7: Pompa P4
   RUNG wire#powerrail
      "HourWork_P4_DB"(Run_Device := wire#w1, Data_sek := "hourWork_setData".Sek_P4, Reset := "dbmanagement".reset.resetLicznikPracy_P4, Data_hour := "hourWork_setData".HourCounterP4, Edge_Hz := "dbdane".Edge_1Hz_P4, MW_hour => "Hour_Work_P4", Sum_hour_sek => "hourWork_setData".Sum_sek_hur_P4)
   END_RUNG
   RUNG wire#powerrail
      Contact( "IsRun_P4" )
   END_RUNG wire#w1
   // the same network as SCL:
   "HourWork_P4_DB"(Run_Device := "IsRun_P4",   // "09_W_Work counter"
                    Data_sek := "hourWork_setData".Sek_P4,
                    Reset := "dbmanagement".reset.resetLicznikPracy_P4,
                    Data_hour := "hourWork_setData".HourCounterP4,
                    Edge_Hz := "dbdane".Edge_1Hz_P4,
                    MW_hour => "Hour_Work_P4",
                    Sum_hour_sek => "hourWork_setData".Sum_sek_hur_P4);
END_REGION

REGION Network 8 (SCL)
   "db10datablock".HourCounterP4:=  "hourWork_setData".HourCounterP4;
END_REGION
END_FUNCTION

FUNCTION_BLOCK "09_W_Work counter"   // FB2, LAD
{ S7_Optimized_Access := 'TRUE' }
AUTHOR : RTecmer
FAMILY : XMHour
VERSION : 0.1
// Licznik czasu pracy
// stored: AutoNumber true, IsIECCheckEnabled false, IsRetainMemResEnabled false, MemoryReserve 500, SetENOAutomatically false, UDAEnableTagReadback false
   VAR_INPUT
      Run_Device : Bool;
   END_VAR
   VAR_OUTPUT
      MW_hour : DWord;
      Sum_hour_sek : Real;   // Licznik sumator godzin i sekund na potrzeby wyznaczania dumchawy do pracy
   END_VAR
   VAR_IN_OUT
      Data_sek : Int;
      Reset { ExternalAccessible := 'False'; ExternalVisible := 'False'; ExternalWritable := 'False'} : Bool;
      Data_hour : DWord;
      Edge_Hz { ExternalAccessible := 'False'; ExternalVisible := 'False'; ExternalWritable := 'False'} : Bool;
   END_VAR
   VAR
      sek_real { ExternalAccessible := 'False'; ExternalVisible := 'False'; ExternalWritable := 'False'} : Real;   // pomocnicza konwerski sekund
      actSekReal { ExternalAccessible := 'False'; ExternalVisible := 'False'; ExternalWritable := 'False'} : Real;   // aktualne sekundy po konwersji
      hour_sek { ExternalAccessible := 'False'; ExternalVisible := 'False'; ExternalWritable := 'False'} : Real;
   END_VAR
   VAR_TEMP   // added for the SCL form of the ladder/FBD networks
      _w1 : Bool;
      _w2 : Bool;
   END_VAR
BEGIN

REGION Network 1
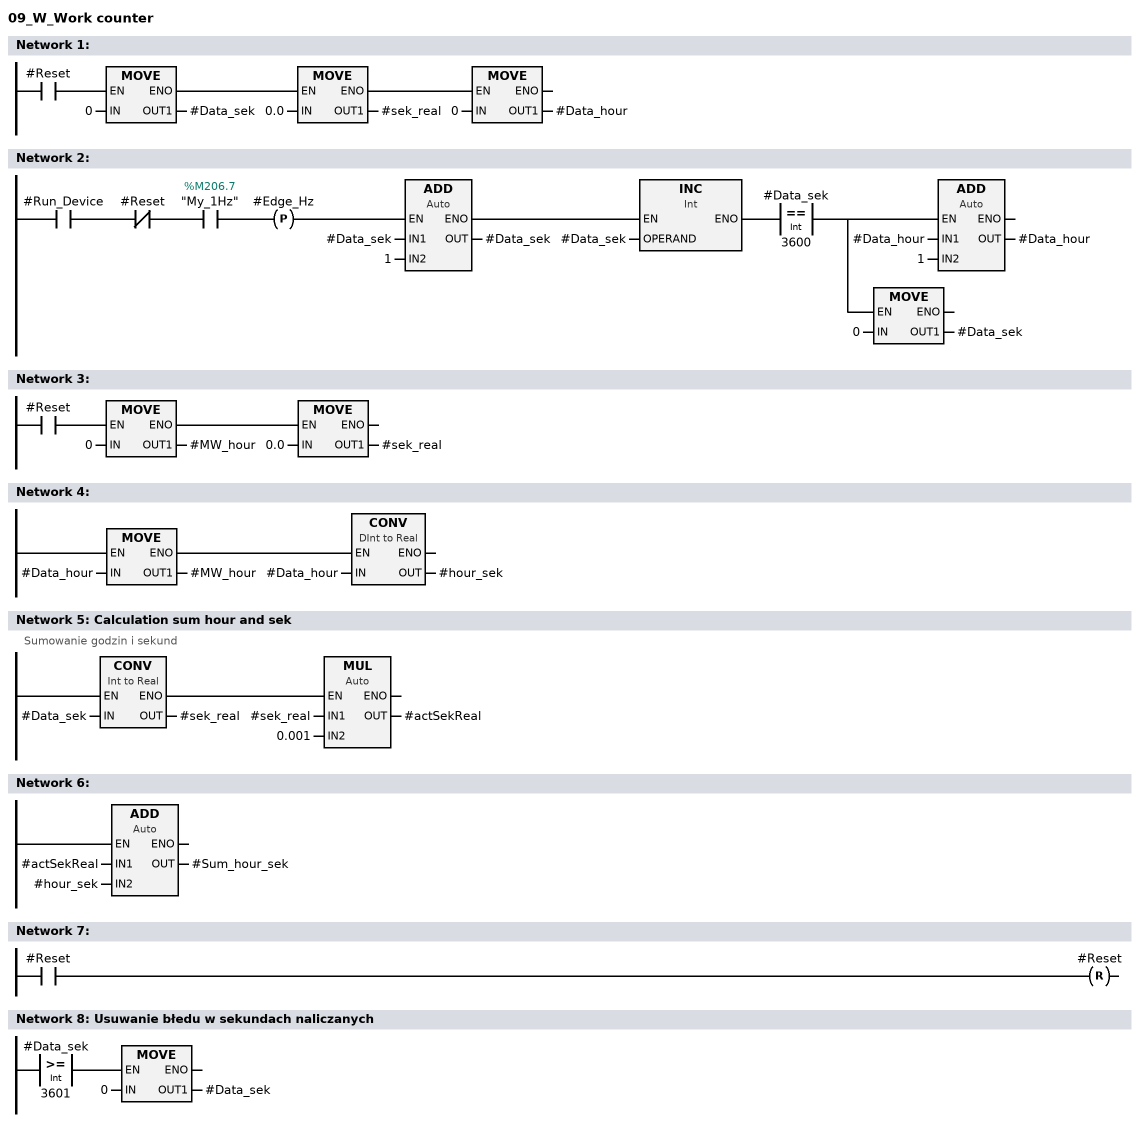
   RUNG wire#powerrail
      Contact( #Reset )
      { S7_GenerateENO := "TRUE" } Move(in := 0, out1 => #Data_sek)
      { S7_GenerateENO := "TRUE" } Move(in := 0.0, out1 => #sek_real)
      { S7_GenerateENO := "TRUE" } Move(in := 0, out1 => #Data_hour)
   END_RUNG
   // the same network as SCL:
   // ENO of a box is taken as its EN; it also drops when the box reports an error
   IF #Reset THEN
       #Data_sek := 0;
       #sek_real := 0.0;
       #Data_hour := 0;
   END_IF;
END_REGION

REGION Network 2
   RUNG wire#powerrail
      Contact( #Run_Device )
      I_Contact( #Reset )
      Contact( "My_1Hz" )
      P_Trig( #Edge_Hz )
      { S7_GenerateENO := "TRUE" } Add(in1 := #Data_sek, in2 := 1, out => #Data_sek)
      { S7_Templates := "DestType := Int"; S7_GenerateENO := "TRUE" } Inc( #Data_sek )
      { S7_Templates := "SrcType := Int" } EQ_Contact(in1 := #Data_sek, in2 := 3600)
      wire#w1
      { S7_GenerateENO := "TRUE" } Add(in1 := #Data_hour, in2 := 1, out => #Data_hour)
   END_RUNG
   RUNG wire#w1
      { S7_GenerateENO := "TRUE" } Move(in := 0, out1 => #Data_sek)
   END_RUNG
   // the same network as SCL:
   // ENO of a box is taken as its EN; it also drops when the box reports an error
   #_w1 := #Run_Device AND NOT #Reset AND "My_1Hz";
   #_w2 := #_w1 AND NOT #Edge_Hz;   // rising edge
   #Edge_Hz := #_w1;
   IF #_w2 THEN
       #Data_sek := #Data_sek + 1;
       #Data_sek := #Data_sek + 1;
   END_IF;
   IF #_w2 AND (#Data_sek = 3600) THEN
       #Data_hour := #Data_hour + 1;
       #Data_sek := 0;
   END_IF;
END_REGION

REGION Network 3
   RUNG wire#powerrail
      Contact( #Reset )
      { S7_GenerateENO := "TRUE" } Move(in := 0, out1 => #MW_hour)
      { S7_GenerateENO := "TRUE" } Move(in := 0.0, out1 => #sek_real)
   END_RUNG
   // the same network as SCL:
   // ENO of a box is taken as its EN; it also drops when the box reports an error
   IF #Reset THEN
       #MW_hour := 0;
       #sek_real := 0.0;
   END_IF;
END_REGION

REGION Network 4
   RUNG wire#powerrail
      { S7_GenerateENO := "TRUE" } Move(in := #Data_hour, out1 => #MW_hour)
      { S7_Templates := "[SrcType := DInt, DestType := Real]" } Convert(in := #Data_hour, out => #hour_sek)
   END_RUNG
   // the same network as SCL:
   // ENO of a box is taken as its EN; it also drops when the box reports an error
   #MW_hour := #Data_hour;
   #hour_sek := DINT_TO_REAL(#Data_hour);
END_REGION

REGION Network 5: Calculation sum hour and sek
   // Sumowanie godzin i sekund
   RUNG wire#powerrail
      { S7_Templates := "[SrcType := Int, DestType := Real]" } Convert(in := #Data_sek, out => #sek_real)
      Mul(in1 := #sek_real, in2 := 0.001, out => #actSekReal)
   END_RUNG
   // the same network as SCL:
   #sek_real := INT_TO_REAL(#Data_sek);
   #actSekReal := #sek_real * 0.001;
END_REGION

REGION Network 6
   RUNG wire#powerrail
      Add(in1 := #actSekReal, in2 := #hour_sek, out => #Sum_hour_sek)
   END_RUNG
   // the same network as SCL:
   #Sum_hour_sek := #actSekReal + #hour_sek;
END_REGION

REGION Network 7
   RUNG wire#powerrail
      Contact( #Reset )
      R_Coil( #Reset )
   END_RUNG
   // the same network as SCL:
   IF #Reset THEN #Reset := FALSE; END_IF;
END_REGION

REGION Network 8: Usuwanie błedu w sekundach naliczanych
   RUNG wire#powerrail
      { S7_Templates := "SrcType := Int" } GE_Contact(in1 := #Data_sek, in2 := 3601)
      { S7_GenerateENO := "TRUE" } Move(in := 0, out1 => #Data_sek)
   END_RUNG
   // the same network as SCL:
   IF #Data_sek >= 3601 THEN #Data_sek := 0; END_IF;
END_REGION
END_FUNCTION_BLOCK

FUNCTION_BLOCK "06_S_MainControlSetPump"
TITLE = MainControlSetPump
{ S7_Optimized_Access := 'TRUE' }
AUTHOR : vrtecmer
VERSION : 0.1
//Główna funkcja wustawiająca aktywną pompę w oparciu o liczniki pracy
   VAR_IN_OUT 
      chosenPump : Int;   // wybrana wiodąca
   END_VAR


BEGIN
	(*
	//=============================================================================
	//(JZWiK S.A Radosław Tecmer)
	//(c)Copyright (2021) All Rights Reserved
	//-----------------------------------------------------------------------------
	//Testowane z:   (system docelowy z  FW 4.4)
	//Pakiet inżynierski:   TIA Portal (V14 Sp1 Update 9)
	//Ograniczenia:  ( - )
	//Wymagania:  (minimalne S7-1200 CPU 1215C FW 4.2 .)
	//Funkcjonalnośc: (Główna funkcja aktywująca znacznik Set_HWork_Px 
	//                 odpowiedniej pompyustawiając ją jako wiodąca)
	//-----------------------------------------------------------------------------
	//Zmainy wprowadzone:
	//Wersja  Data       Osoba wprowadzająca zmiany - ekspert
	//01.00.00 23.09.2023 (Tecmer Radosław - twórca) Pieresza wersja 01.00.00
	//=============================================================================
	*)
	
	// Znajdź pompę o najmniejszym stanie licznika pracy
	"FindPumpWithMinWorkTime_DB_1"(chosenPump:= #chosenPump);
	
	IF #chosenPump > 0 THEN
	  // Ustaw wybraną pompę do pracy
	  "SetActivePump_DB_1"(ActivePump:="dbdane".ActivePump,
	                       pumpNum:="dbdane".pumpNum);
	 
	  
	END_IF;
END_FUNCTION_BLOCK

FUNCTION "08_M_ClearError_Modbus" : Void
{ S7_Optimized_Access := 'TRUE' }
AUTHOR : rtecmer
VERSION : 0.1
   VAR_TEMP 
      set_error_RTU : Bool;
   END_VAR


BEGIN
	
	(*
	//=============================================================================
	//(JZWiK S.A Radosław Tecmer)
	//(c)Copyright (2021) All Rights Reserved
	//-----------------------------------------------------------------------------
	//Testowane z:   (system docelowy z  FW 4.4)
	//Pakiet inżynierski:   TIA Portal (V14 Sp1 Update 9)
	//Ograniczenia:  ( - )
	//Wymagania:  (minimalne S7-1200 CPU 1215C FW 4.2 .)
	//Funkcjonalnośc: (Obsługa błedów na magistrali Modbus RTU, inicjacja pętli po konfliktach )
	//-----------------------------------------------------------------------------
	//Zmainy wprowadzone:
	//Wersja  Data       Osoba wprowadzająca zmiany - ekspert
	//01.00.00 17.11.2021 (Tecmer Radosław - twórca) Pieresza wersja 01.00.00
	//=============================================================================
	*)
	
